Omron CX-Programmer project 新工程 (CX-Programmer 9.61)

# PLC 后氦检24L: CJ2M CPU33
I/O table (CPU CJ2M-CPU33): rack 0 slot 0 CJ1W-NC213; rack 0 slot 1 CJ1W-SCU21-V1; rack 0 slot 2 CJ1W-SCU21-V1; rack 0 slot 3 CJ1W-AD041-V1; rack 0 slot 4 CJ1W-ID261; rack 0 slot 5 CJ1W-ID261; rack 0 slot 6 CJ1W-OD261; rack 0 slot 7 CJ1W-MD231; rack 0 slot 11 CJ2M-EIP21

## Global symbols (name address type ; comment)
0 CHANNEL  ; 料盒#6电池屏蔽信号
0.00 BOOL  ; $?St$Bk?_#[1162] / 数字压力表 / $?St$Bk?_#[1162]
0.01 BOOL  ; 扫码位电池感应
0.02 BOOL  ; 抓料位有托盘感应
0.03 BOOL  ; 抓电池处有电池感应
0.04 BOOL  ; 腔体1有料感应
0.05 BOOL  ; 缺相保护信号
0.06 BOOL  ; 出料起始位有料感应
0.07 BOOL  ; 输送带有料感应
0.08 BOOL  ; NG放料位有料感应(常闭)
0.09 BOOL  ; NG通道料满感应
0.10 BOOL  ; 上料柔性报警
0.11 BOOL  ; 下料柔性报警延时
0.12 BOOL  ; 入盘升降柔性报警
0.13 BOOL  ; 料盒#12电池有料感应
0.14 BOOL  ; 料盒#11电池有料信号
0.15 BOOL  ; 料盒#10电池有料信号
10.00 BOOL  ; #2破真空阀
10.01 BOOL  ; #2吹气阀
10.02 BOOL  ; #2上顶升气缸
10.03 BOOL  ; #1上顶升气缸
10.04 BOOL  ; #2下顶升气缸
10.05 BOOL  ; #1下顶升气缸
10.06 BOOL  ; 料盒上阻挡气缸
10.07 BOOL  ; 料盒下阻挡气缸
10.08 BOOL  ; 料盒定位气缸
10.09 BOOL  ; 拉带左脱离气缸
10.10 BOOL  ; 拉带右脱离气缸
10.11 BOOL  ; 出料NG拨料气缸
10.12 BOOL  ; 上空料盘电机
10.13 BOOL  ; 下有料盘电机
10.14 BOOL  ; 有料盘缓存电机
10.15 BOOL  ; 出料输送带
11.01 BOOL  ; 真空泵
11.02 BOOL  ; 氦检仪启动
11.03 BOOL  ; 启动指示灯
11.04 BOOL  ; 停止指示灯
11.05 BOOL  ; 复位指示灯
11.06 BOOL  ; 蜂鸣器
11.07 BOOL  ; 三色红灯
11.08 BOOL  ; 三色绿灯
11.09 BOOL  ; 三色黄灯
11.10 BOOL  ; 料盒升降伺服Serv_ON
11.11 BOOL  ; 料盒升降伺服Alarm_Clr
11.12 BOOL  ; 入盘升降气缸
11.13 BOOL  ; 入盘夹爪气缸
11.14 BOOL  ; 龙门升降伺服刹车
11.15 BOOL  ; 料盒升降伺服刹车
12.03 BOOL  ; NG有料感应
12.07 BOOL  ; 腔体2有料感应
13.00 BOOL  ; 上料NG伸出位
13.01 BOOL  ; 上料NG缩回位
13.02 BOOL  ; 上料NG满感应
13.03 BOOL  ; 上料缓存NG有料感应
13.04 BOOL  ; 右按钮上气缸顶升请求（上料叉车到位）
13.05 BOOL  ; 左按钮气缸顶升请求（下料叉车到位）
13.07 BOOL  ; 腔体2有料感应
13.08 BOOL  ; 上料盒位有料盒感应
1534.15 BOOL  ; 单元1的串口1协议宏执行标志
1544.15 BOOL  ; 单元1的串口2协议宏执行标志
1559.15 BOOL  ; 单元2串口1协议宏执行标志
19.00 BOOL  ; 真空泵缺相报警
19.01 BOOL  ; PC系统异常
1.00 BOOL  ; 料盒#9电池有料信号
1.01 BOOL  ; 料盒#8电池有料信号
1.02 BOOL  ; 料盒#7电池有料信号
1.03 BOOL  ; 料盒#6电池有料信号
1.04 BOOL  ; 料盒#5电池有料信号
1.05 BOOL  ; 料盒#4电池有料信号
1.06 BOOL  ; 料盒#3电池有料信号
1.07 BOOL  ; 料盒#2电池有料信号
1.08 BOOL  ; 料盒#1电池有料信号
1.09 BOOL  ; 料盒#24电池有料信号
1.10 BOOL  ; 料盒#23电池有料信号
1.11 BOOL  ; 料盒#22电池有料信号
1.12 BOOL  ; 料盒#21电池有料信号
1.13 BOOL  ; 料盒#20电池有料信号
1.14 BOOL  ; 料盒#19电池有料信号
1.15 BOOL  ; 料盒#18电池有料信号
2000.03 BOOL  ; 绝对定位
2000.06 BOOL  ; 前后位回原
2000.09 BOOL  ; 龙门前后伺服脉冲
2000.10 BOOL  ; 龙门前后伺服方向
2000.12 BOOL  ; NC-X轴错误复位
2000.15 BOOL  ; 入盘Y轴停止
2002.03 BOOL  ; 料盘绝对运动
2002.06 BOOL  ; 料盘回原
2002.09 BOOL  ; 料盘升降脉冲
2002.10 BOOL  ; 料盘运动方向
2002.12 BOOL  ; NC-Y轴复位
2002.15 BOOL  ; 料盘伺服减速2停止
2004.06 BOOL  ; Y轴原点标志
2004.12 BOOL  ; NC
2004.13 BOOL  ; 伺服忙标志位
2007.06 BOOL  ; 料盘升降原点标志
2007.13 BOOL  ; 料盘伺服忙标志位
2010 CHANNEL  ; #1真空计度读出值CHO
2011 CHANNEL  ; #1真空计读出值CH1
2012 CHANNEL  ; #2真空计读出值CH2
20.01 BOOL  ; #2电池扫码信号
20.04 BOOL  ; 两扫码NG
20.09 BOOL  ; 放右NG缩回
21.00 BOOL  ; 上料机械手回左上料位
21.01 BOOL  ; 上料机械手回右上料位
21.05 BOOL  ; 上料右夹爪夹紧
21.09 BOOL  ; 上料右夹爪松开
21.10 BOOL  ; 上料提升气缸缩回
21.11 BOOL  ; 上料提升气缸/左夹爪升降气缸伸出
21.14 BOOL  ; 上料右夹爪夹紧
21.15 BOOL  ; 上料机械手去#1腔体放料
22.02 BOOL  ; 上料提升气缸取OK料后缩回(A)
22.10 BOOL  ; 上料提升气缸伸出(抓NG料)(A)
22.12 BOOL  ; 上料提升气缸伸出(放扫码NG料)(A)
22.13 BOOL  ; #1，#2夹爪张开(放扫码NG料)(A)
22.14 BOOL  ; 上料提升气缸缩回(放扫码NG料)(A)
22.15 BOOL  ; 扫码NG气缸缩回
25.13 BOOL  ; 出料机械手归零后回NG位置
25.15 BOOL  ; 机械手放料条件
26.00 BOOL  ; 出料旋转回#1待料位
26.02 BOOL  ; 下料升降气缸输出
26.06 BOOL  ; 下料升降/提升气缸输出
26.13 BOOL  ; 下料旋转回#2待料角度
26.14 BOOL  ; 下料旋转回出料角度
27.00 BOOL  ; 下料旋转归零后回下料角度
28.00 BOOL  ; 电池从扫码位到抓料超时
28.01 BOOL  ; 扫码阻挡气缸缩回位异常
28.02 BOOL  ; 扫码阻挡气缸伸出位异常
28.03 BOOL  ; 抓料阻挡气缸缩回位异常
28.04 BOOL  ; 抓料阻挡气缸伸出位异常
28.09 BOOL  ; 出料机械手回#1腔体位置
28.10 BOOL  ; 出料机械手回#2腔体位置
28.11 BOOL  ; 出料机械手回OK位置
28.12 BOOL  ; 出料机械手回放爪2位置
28.13 BOOL  ; 出料机械手回NG位置
2906.06 BOOL  ; 进料机械手左极限
2906.07 BOOL  ; 进料机械手右极限
2906.08 BOOL  ; 出料机械手左极限
2906.09 BOOL  ; 出料机械手右极限
2960.06 BOOL  ; 进料机械手左限位
2960.07 BOOL  ; 进料机械手右限位
2960.08 BOOL  ; 出料机械手左限位
2960.09 BOOL  ; 出料机械手右限位
2962.00 BOOL  ; 入盘升降原点
2962.06 BOOL  ; 龙门升降伺服上限位
2962.07 BOOL  ; 龙门升降伺服下限位
2962.08 BOOL  ; 龙门左右伺服左限位
2962.09 BOOL  ; 龙门左右伺服右限位
29.00 BOOL  ; 扫码NG拨料气缸缩回位报警
29.01 BOOL  ; 扫码NG拨料气缸伸出报警
29.02 BOOL  ; 上料提升气缸缩回报警
29.03 BOOL  ; 上料提升气缸伸出报警
29.04 BOOL  ; 上料左夹爪升降缩回报警
29.05 BOOL  ; 上料左夹爪升降气缸伸出报警
29.06 BOOL  ; 上料右夹爪升降气缸缩回报警
29.07 BOOL  ; 上料右夹爪升降气缸缩回报警
29.08 BOOL  ; 上料左夹爪张开位报警
29.09 BOOL  ; 上料左夹爪夹紧报警
29.10 BOOL  ; 上料夹爪2张开报警
29.11 BOOL  ; 上料夹爪2夹紧报警
29.12 BOOL  ; 上料机构柔性报警
29.13 BOOL  ; 进料机械手报警
2.00 BOOL  ; 料盒#17电池有料信号
2.01 BOOL  ; 料盒#16电池有料信号
2.02 BOOL  ; 料盒#15电池有料信号
2.03 BOOL  ; 料盒#14电池有料信号
2.04 BOOL  ; 料盒#13电池有料信号
2.05 BOOL  ; 扫码阻挡缩回位
2.06 BOOL  ; 扫码阻挡气缸伸出位
2.07 BOOL  ; 扫码定位气缸缩回位
2.08 BOOL  ; 扫码定位气缸伸出位
2.09 BOOL  ; 抓料阻挡气缸缩回位
2.10 BOOL  ; 抓料阻挡气缸伸出位
2.11 BOOL  ; 上料提升气缸缩回位
2.12 BOOL  ; 上料提升气缸伸出位
2.13 BOOL  ; 上料左夹爪升降气缸缩回位
2.14 BOOL  ; 上料左夹爪升降气缸伸出位
2.15 BOOL  ; 上料右夹爪升降气缸缩回位
32.00 BOOL  ; 读检漏仪状态
32.01 BOOL  ; 读氦检仪状态完成
32.02 BOOL  ; 读检漏口压力
32.03 BOOL  ; 读检漏口压力完成
32.05 BOOL  ; 读漏率
32.06 BOOL  ; 读漏率完成
32.07 BOOL  ; 读漏率失败
32.08 BOOL  ; 读氦检仪状态失败
32.09 BOOL  ; 读检漏口压力失败
3304.10 BOOL  ; 氦检仪报警
33.00 BOOL  ; #1腔体复位破真空
33.01 BOOL  ; #1合模气缸复位缩回
33.02 BOOL  ; 进料机械手有料
33.03 BOOL  ; 出料机械手有料
33.04 BOOL  ; #1合模气缸复位
33.05 BOOL  ; 下料夹爪有料
34.00 BOOL  ; 氦检仪当前为检漏状态
34.01 BOOL  ; 氦检仪当前为待机状态
34.02 BOOL  ; 氦检仪当前为启动状态
34.03 BOOL  ; 氦检仪当前为定标状态
34.04 BOOL  ; 氦检仪当前为错误状态
34.05 BOOL  ; 氦检仪当前为暂停状态
35.00 BOOL  ; #2腔体复位破真空
35.01 BOOL  ; #2合模气缸缩回
35.02 BOOL  ; #2合模气缸复位
35.05 BOOL  ; 扫码气缸自动伸出
39.00 BOOL  ; 合模气缸1缩回报警
39.01 BOOL  ; 合模气缸1伸出报警
39.02 BOOL  ; 合模气缸2缩回报警
39.03 BOOL  ; 合模气缸2伸出报警
39.04 BOOL  ; 氦检仪没启动
39.05 BOOL  ; 读氦漏率失败
39.06 BOOL  ; 读氦检仪状态失败
39.07 BOOL  ; 读检漏口压力失败
39.08 BOOL  ; 氦检仪通信异常
39.09 BOOL  ; 扫码枪通信异常
39.10 BOOL  ; #1真空计断线报警
39.11 BOOL  ; #2真空计断线报警
39.12 BOOL  ; （I：0.04）#1腔体有料感应异常
39.13 BOOL  ; （I：13.07）#2腔体有料感应异常
3.00 BOOL  ; 上料右夹爪升降气缸伸出位
3.01 BOOL  ; 上料左夹爪张开位
3.02 BOOL  ; 上料左夹爪夹紧位
3.03 BOOL  ; 上料右夹爪张开位
3.04 BOOL  ; 上料右夹爪夹紧位
3.05 BOOL  ; 下料提升气缸缩回位
3.06 BOOL  ; 下料提升气缸伸出位
3.07 BOOL  ; 下料夹爪升降气缸缩回位
3.08 BOOL  ; 下料夹爪升降气缸伸出位
3.09 BOOL  ; 下料左夹爪张开位
3.10 BOOL  ; 下料左夹爪夹紧位
3.11 BOOL  ; 下料右夹爪张开位
3.12 BOOL  ; 下料右夹爪夹紧位
3.13 BOOL  ; #1合模气缸缩回位
3.14 BOOL  ; #1合模气缸伸出位
3.15 BOOL  ; #2合模气缸缩回位
46.00 BOOL  ; #1夹爪放料完成
46.01 BOOL  ; #2夹爪放料完成
48.00 BOOL  ; 出料机械手位置异常
48.01 BOOL  ; 下料旋转托盘位置异常
48.02 BOOL  ; 下料缓存有料异常
48.03 BOOL  ; #1合模气缸不在缩回位
48.04 BOOL  ; #2合模气缸不在缩回位
48.05 BOOL  ; 出料夹爪不在张开位
48.06 BOOL  ; 出料提升气缸不在伸出位
48.07 BOOL  ; 出料提升气缸不在缩回位
48.08 BOOL  ; 出料机械手没归零
48.09 BOOL  ; 出料机械手到达左极限
48.10 BOOL  ; 出料机械手到达右极限
48.11 BOOL  ; 进料机械手位置避让异常
48.12 BOOL  ; 进料机械手位置避让异常
49.00 BOOL  ; 下料提升气缸缩回报警
49.01 BOOL  ; 下料提升气缸伸出报警
49.02 BOOL  ; 下料夹爪升降气缸缩回报警
49.03 BOOL  ; 下料夹爪升降气缸伸出报警
49.04 BOOL  ; 下料夹爪1张开报警
49.05 BOOL  ; 下料夹爪夹1紧报警
49.06 BOOL  ; 下料夹爪2张开位延时报警
49.07 BOOL  ; 下料夹爪2夹紧位报警
49.08 BOOL  ; 出料NG拨料气缸伸出位报警
49.09 BOOL  ; 出料NG拨料气缸缩回位报警
49.10 BOOL  ; 出料机械手报警
49.11 BOOL  ; 下料机构柔性报警
49.12 BOOL  ; （0.06）出料起始位有料感应异常
49.13 BOOL  ; （10.05）出料拉带运行异常
49.14 BOOL  ; （0.07）出料拉带末端感应异常
4.00 BOOL  ; #2合模气缸伸出位
4.01 BOOL  ; 出料NG拨料气缸缩回位
4.02 BOOL  ; 出料NG拨料气缸伸出位
4.03 BOOL  ; 料盒定位气缸缩回位
4.04 BOOL  ; 料盒定位气缸伸出位
4.05 BOOL  ; 料盒上阻挡气缸缩回位
4.06 BOOL  ; 料盒上阻挡气缸伸出位
4.07 BOOL  ; 料盒下阻挡气缸缩回位
4.08 BOOL  ; 料盒下阻挡气缸伸出位
4.09 BOOL  ; #2上顶升左气缸缩回位
4.10 BOOL  ; #2上顶升左气缸伸出位
4.11 BOOL  ; #2上顶升右气缸缩回位
4.12 BOOL  ; #2上顶升右气缸伸出位
4.13 BOOL  ; #1上顶升左气缸缩回位
4.14 BOOL  ; #1上顶升左气缸伸出位
4.15 BOOL  ; #1上顶升右气缸缩回位
54.00 BOOL  ; 放料准备-拉带对接测试按钮(T)
54.02 BOOL  ; 放料可移动-拉带对接测试按钮(T)
54.03 BOOL  ; 取料准备-拉带对接测试按钮(T)
54.05 BOOL  ; 取料可移动-拉带对接测试按钮(T)
54.06 BOOL  ; 设备故障-拉带对接测试按钮(T)
54.10 BOOL  ; 可取料-拉带对接测试按钮(T)
5.00 BOOL  ; #1上顶升右气缸伸出位
5.01 BOOL  ; #2下顶升左气缸缩回位
5.02 BOOL  ; #2下顶升左气缸伸出位
5.03 BOOL  ; #2下顶升右气缸缩回位
5.04 BOOL  ; #2下顶升右气缸伸出位
5.05 BOOL  ; #1下顶升左气缸缩回位
5.06 BOOL  ; #1下顶升左气缸伸出位
5.07 BOOL  ; #1下顶升右气缸缩回位
5.08 BOOL  ; #1下顶升右气缸伸出位
5.09 BOOL  ; 龙门左拉带脱离气缸缩回位
5.10 BOOL  ; 龙门左拉带脱离气缸伸出位
5.11 BOOL  ; 龙门右拉带脱离气缸缩回位
5.12 BOOL  ; 龙门右拉带脱离气缸伸出位
5.13 BOOL  ; 上料伺服Ready信号
5.14 BOOL  ; 上料伺服Alarm信号
5.15 BOOL  ; 下料伺服Ready信号
68.00 BOOL  ; 料盒定位气缸缩回位报警
68.01 BOOL  ; 料盒定位气缸伸出位报警
68.02 BOOL  ; 料盒上阻挡气缸缩回位报警
68.03 BOOL  ; 料盒上阻挡气缸伸出位报警
68.04 BOOL  ; #1上顶升左气缸缩回位报警
68.05 BOOL  ; #1上顶升左气缸伸出位报警
68.06 BOOL  ; #1上顶升右气缸缩回位报警
68.07 BOOL  ; #1上顶升右气缸伸出位报警
68.08 BOOL  ; #2上顶升左气缸缩回位报警
68.09 BOOL  ; #2上顶升左气缸伸出位报警
68.10 BOOL  ; #2上顶升右气缸缩回位报警
68.11 BOOL  ; #2上顶升右气缸伸出位报警
68.12 BOOL  ; #1下顶升左气缸缩回位报警
68.13 BOOL  ; #1下顶升左气缸伸出位报警
68.14 BOOL  ; #1下料顶升右气缸缩回位报警
68.15 BOOL  ; #1下顶升右气缸伸出位报警
69.00 BOOL  ; #2下顶升左气缸缩回位报警
69.01 BOOL  ; #2下顶升左气缸伸出位报警
69.02 BOOL  ; #2下料顶升右气缸缩回位报警
69.03 BOOL  ; #2下顶升右气缸伸出位报警
69.04 BOOL  ; 入盘左拉带脱离气缸缩回位报警
69.05 BOOL  ; 入盘左拉带脱离气缸伸出位报警
69.06 BOOL  ; 入盘右拉带脱离气缸缩回位报警
69.07 BOOL  ; 入盘右拉带脱离气缸伸出位报警
69.08 BOOL  ; 入盘升降气缸缩回位延时报警
69.09 BOOL  ; 入盘升降气缸伸出位延时报警
69.10 BOOL  ; 入盘夹爪气缸松开延时报警
69.11 BOOL  ; 入盘夹爪气缸夹紧延时报警
69.12 BOOL  ; 入盘机械手柔性报警
69.13 BOOL  ; 此位置有电池不能入盘
6.00 BOOL  ; 下料伺服Alarm信号
6.01 BOOL  ; 入盘升降伺服Ready信号
6.02 BOOL  ; 入盘升降伺服Alarm信号
6.03 BOOL  ; 龙门左右伺服Ready信号
6.04 BOOL  ; 龙门左右伺服Alarm信号
6.05 BOOL  ; 龙门前后伺服Ready信号
6.06 BOOL  ; 龙门前后伺服Alarm信号
6.07 BOOL  ; 氦检仪器报警
6.08 BOOL  ; 启动按钮
6.09 BOOL  ; 停止按钮
6.10 BOOL  ; 复位按钮
6.11 BOOL  ; 急停按钮
6.12 BOOL  ; 前门磁开关
6.13 BOOL  ; 后门磁开关
6.14 BOOL  ; 左门禁开关
6.15 BOOL  ; 右门禁开关
70.01 BOOL  ; I:7.01空托盘感应感应异常
70.02 BOOL  ; I:7.00空托盘感应感应异常
70.03 BOOL  ; （7.02）空托盘到位感应或拉带异常
70.04 BOOL  ; (7.05)#3空托盘感应或拉带异常
70.05 BOOL  ; 空托盘到位感应、#3空托盘感应或拉带异常
70.06 BOOL  ; 空托盘到位感应
70.07 BOOL  ; 空盘升降机架上有空托盘记忆异常
70.08 BOOL  ; （7.05）上空托盘位感应异常
70.09 BOOL  ; （7.14）下满料托盘感应1异常
70.10 BOOL  ; （7.04）下满料托盘到位感应#2异常
70.11 BOOL  ; （13.08）电池入盘位有托盘感应异常
70.12 BOOL  ; （7.03）缓存#1托盘到位感应异常
70.13 BOOL  ; （7.04）缓存#2托盘到位感应异常
71.00 BOOL  ; 上空托盘感应异常
7.00 BOOL  ; #2下感应有空料盒（外面）
7.01 BOOL  ; #1下感应有空料盒
7.02 BOOL  ; 料盒到位感应
7.03 BOOL  ; 缓存1有料到位感应
7.04 BOOL  ; 缓存2有料到位感应
7.05 BOOL  ; #3下料盒有料感应
7.06 BOOL  ; 料盒升降伺服Ready
7.07 BOOL  ; 料盒升降伺服Alarm
7.08 BOOL  ; $?St$Bk?_#[1163] / 龙门升降气缸缩回位 / $?St$Bk?_#[1163]
7.09 BOOL  ; $?St$Bk?_#[1164] / 龙门升降气缸伸出位 / $?St$Bk?_#[1164]
7.10 BOOL  ; $?St$Bk?_#[1165] / 龙门夹爪气缸张开位 / $?St$Bk?_#[1165]
7.11 BOOL  ; 龙门夹爪气缸夹紧
7.12 BOOL  ; $?St$Bk?_#[1166] / 上层货架叉车感应 / $?St$Bk?_#[1166]
7.13 BOOL  ; $?St$Bk?_#[1167] / 下层货架叉车感应 / $?St$Bk?_#[1167]
7.14 BOOL  ; 上有料盒感应1
7.15 BOOL  ; 缓存2有料感应
81.00 BOOL  ; 扫码NG缓存有料
82.02 BOOL  ; #3上料夹爪有料
82.03 BOOL  ; #4上料夹爪有料
83.02 BOOL  ; #3下料夹爪有料
83.03 BOOL  ; #4下料夹爪有料
84.11 BOOL  ; #2扫码失败
84.12 BOOL  ; #2扫码OK
8.00 BOOL  ; $?St$Bk?_#[1168] / 上料伺服Serv_On / $?St$Bk?_#[1168]
8.01 BOOL  ; $?St$Bk?_#[1169] / 上料伺服Alarm_Clr / $?St$Bk?_#[1169]
8.02 BOOL  ; $?St$Bk?_#[1170] / 下料伺服Serv_On / $?St$Bk?_#[1170]
8.03 BOOL  ; $?St$Bk?_#[1171] / 下料伺服Alarm_Clr / $?St$Bk?_#[1171]
8.04 BOOL  ; $?St$Bk?_#[1172] / 龙门升降伺服Serv_On / $?St$Bk?_#[1172]
8.05 BOOL  ; 龙门升降伺服Alarm_Clr
8.06 BOOL  ; 龙门左右伺服Serv_ON
8.07 BOOL  ; 龙门左右伺服Alarm_Clr
8.08 BOOL  ; 龙门前后伺服Serv_ON
8.09 BOOL  ; $?St$Bk?_#[1173] / 龙门前后伺服Alarm_Clr / $?St$Bk?_#[1173]
8.10 BOOL  ; 扫码阻挡气缸
8.11 BOOL  ; 抓料阻挡气缸
8.12 BOOL  ; 上料NG气缸
8.13 BOOL  ; 上料提升气缸
8.14 BOOL  ; 上料左夹爪升降气缸
8.15 BOOL  ; 上料右夹爪升降气缸
9.00 BOOL  ; $?St$Bk?_#[1174] / 上料左夹爪气缸 / $?St$Bk?_#[1174]
9.01 BOOL  ; 上料右夹爪
9.02 BOOL  ; 下料提升气缸
9.03 BOOL  ; 下料夹爪升降气缸
9.04 BOOL  ; 下料左夹爪气缸
9.05 BOOL  ; 下料右夹爪气缸
9.06 BOOL  ; #1合模气缸关闭
9.07 BOOL  ; #1合模气缸打开
9.08 BOOL  ; $?St$Bk?_#[1175] / #1腔体抽气阀 / $?St$Bk?_#[1175]
9.09 BOOL  ; $?St$Bk?_#[1176] / #1腔体氦检阀 / $?St$Bk?_#[1176]
9.10 BOOL  ; $?St$Bk?_#[1177] / #1腔体破真空阀 / $?St$Bk?_#[1177]
9.11 BOOL  ; $?St$Bk?_#[1178] / #1腔体吹气阀 / $?St$Bk?_#[1178]
9.12 BOOL  ; #2合模气缸关闭
9.13 BOOL  ; #2合模气缸打开
9.14 BOOL  ; #2抽气阀
9.15 BOOL  ; #2氦检阀
A202.01 BOOL  ; 通信端口1允许标志
A202.02 BOOL  ; 通信端口2允许标志
A276 CHANNEL  ; 前机械手当前脉冲
A278 CHANNEL  ; 后机械手当前脉冲
A280.04 BOOL  ; 上料机械手脉冲输出中
A280.05 BOOL  ; 上料机械手原点标志
A281.04 BOOL  ; 后机械手脉冲输出中
A281.05 BOOL  ; 下料机械手原点标志
A322 CHANNEL  ; 上料旋转当前位置脉冲
A324 CHANNEL  ; 下料旋转当前位置脉冲
A326.04 BOOL  ; 入盘升降脉冲输出中
A326.05 BOOL  ; 入盘升降原点标志
A327.04 BOOL  ; 入盘X轴脉冲标志
A327.05 BOOL  ; 入盘X轴原点标志
A351 CHANNEL  ; 系统时间(分秒)
A352 CHANNEL  ; 系统时间(日时)
A353 CHANNEL  ; 系统时间(年月)
A501.01 BOOL  ; #1通信模块复位
A501.02 BOOL  ; #2通信模块复位
A540.08 BOOL  ; 进料机械手CW
A540.09 BOOL  ; 进料机械手CCW
A541.08 BOOL  ; 出料机械手CW
A541.09 BOOL  ; 出料机械手CCW
A542.08 BOOL  ; 龙门升降伺服下限位
A542.09 BOOL  ; 龙门升降伺服上限位
A543.08 BOOL  ; 龙门左右伺服右限位
A543.09 BOOL  ; 龙门左右伺服左限位
D0.00 BOOL  ; CF113
D10 CHANNEL  ; 报警画面跳转
D100 CHANNEL  ; 扫码阻挡气缸缩回位延时
D1000 CHANNEL  ; #1腔体检漏口压力(浮点)
D1002 CHANNEL  ; #1腔体漏率(浮点)
D1004 CHANNEL  ; #1腔体测试完成时的检漏口压力
D1006 CHANNEL  ; #1腔体测试完成时的漏率
D1008 CHANNEL  ; #1腔抽残气压力
D101 CHANNEL  ; 扫码阻挡气缸伸出位延时
D102 CHANNEL  ; 扫码定位气缸缩回位延时
D1020 CHANNEL  ; #2腔体检漏口压力(浮点)
D1022 CHANNEL  ; #2腔体漏率(浮点)
D1024 CHANNEL  ; #2腔体测试完成时检漏口压力
D1026 CHANNEL  ; #2腔体测试完成时的漏率
D1028 CHANNEL  ; #2腔抽残气压力
D103 CHANNEL  ; 扫码定位气缸伸出位延时
D104 CHANNEL  ; 抓料阻挡气缸缩回位延时
D105 CHANNEL  ; 抓料阻挡气缸伸出位延时
D106 CHANNEL  ; 上料提升气缸缩回位延时
D107 CHANNEL  ; 上料提升气缩回位延时
D108 CHANNEL  ; 上料左夹爪升降气缸缩回位延时
D109 CHANNEL  ; 上料左夹爪升降气缸伸出位延时
D110 CHANNEL  ; 上料右夹爪升降气缸缩回位延时
D111 CHANNEL  ; 上料右夹爪升降气缸伸出位延时
D112 CHANNEL  ; 上料左夹爪张开位延时
D113 CHANNEL  ; 上料左夹爪夹紧位延时
D114 CHANNEL  ; 上料右夹爪张开位延时
D115 CHANNEL  ; 上料右夹爪夹紧位延时
D116 CHANNEL  ; 下料提升气缸缩回位延时
D1160 CHANNEL  ; 正向行程
D1164 CHANNEL  ; 反向行程（浮点）
D1168 CHANNEL  ; 反向行程
D117 CHANNEL  ; 下料提升气缸伸出位延时
D118 CHANNEL  ; 下料夹爪升降气缸缩回位延时
D119 CHANNEL  ; 下料夹爪升降气缸伸出位延时
D120 CHANNEL  ; 下料左夹爪张开位延时
D1204 CHANNEL  ; 检漏口压力设定值
D1206 CHANNEL  ; 漏率设定值
D121 CHANNEL  ; 下料左夹爪夹紧位延时
D122 CHANNEL  ; 下料右夹爪张开位延时
D123 CHANNEL  ; 下料右夹爪夹紧位延时
D124 CHANNEL  ; #1合模气缸缩回位延时
D125 CHANNEL  ; #1合模气缸伸出位延时
D126 CHANNEL  ; #2合模气缸缩回位延时
D1260 CHANNEL  ; 检漏口压力底数转换
D1264 CHANNEL  ; 漏率底数转换
D127 CHANNEL  ; #2合模气缸伸出位延时
D128 CHANNEL  ; 扫码NG拨料气缸缩回位延时
D129 CHANNEL  ; 扫码NG拨料气缸伸出位延时
D130 CHANNEL  ; 料盒定位气缸缩回位延时
D131 CHANNEL  ; 料盒定位气缸伸出位延时
D132 CHANNEL  ; 料盒上阻挡气缸缩回位延时
D133 CHANNEL  ; 料盒上阻挡气缸伸出位延时
D134 CHANNEL  ; 料盒下阻挡气缸缩回位延时
D135 CHANNEL  ; 料盒下阻挡气缸伸出位延时
D136 CHANNEL  ; #1上顶升左气缸缩回位延时
D137 CHANNEL  ; #1上顶升左气缸伸出位延时
D138 CHANNEL  ; #1上顶升右气缸缩回位延时
D139 CHANNEL  ; #1上顶升右气缸伸出位延时
D140 CHANNEL  ; #2上顶升左气缸缩回位延时
D141 CHANNEL  ; #2上顶升左气缸伸出位延时
D142 CHANNEL  ; #2上顶升右气缸缩回位延时
D143 CHANNEL  ; #2上顶升右气缸伸出位延时
D144 CHANNEL  ; #1下顶升左气缸缩回位延时
D145 CHANNEL  ; #1下顶升左气缸伸出位延时
D146 CHANNEL  ; #1下顶升右气缸缩回位延时
D147 CHANNEL  ; #1下顶升右气缸伸出位延时
D148 CHANNEL  ; #2下顶升左气缸延时缩回位
D149 CHANNEL  ; #2下顶升左气缸伸出位延时
D150 CHANNEL  ; #2下顶升右气缸缩回位延时
D151 CHANNEL  ; #2下顶升右气缸伸出位延时
D152 CHANNEL  ; 龙门左拉带脱离气缸缩回位延时
D153 CHANNEL  ; 龙门左拉带脱离气缸伸出位延时
D154 CHANNEL  ; 龙门右拉带脱离气缸缩回位延时
D155 CHANNEL  ; 龙门右拉带脱离气缸伸出位延时
D160 CHANNEL  ; 上料旋转步进当前脉冲
D1600 CHANNEL  ; #1条码下料机械手#1
D1606 CHANNEL  ; （龙门）抓料机械手当前位置(mm)
D1610 CHANNEL  ; #2条码下料机械手#2
D162 CHANNEL  ; 上料旋转步进当前脉冲(浮点）
D1620 CHANNEL  ; 产品检漏口压力在下料机械手#1
D1630 CHANNEL  ; 产品检漏口压力在下料机械手#2
D164 CHANNEL  ; 旋转脉冲当量(浮点)
D1640 CHANNEL  ; #1腔体测试完成时的漏率在下料机械手#1
D1650 CHANNEL  ; #1腔体测试完成时的漏率在下料机械手#2
D166 CHANNEL  ; 上料旋转步进当前位置(mm)
D1660 CHANNEL  ; 产品测试结果在下料机械手#1
D1670 CHANNEL  ; 产品测试结果在下料机械手#2
D168 CHANNEL  ; 旋转脉冲当量
D1690 CHANNEL  ; 1夹爪-1为腔体1-2为腔体2
D1692 CHANNEL  ; 2夹爪-1为腔体1-2为腔体2
D170 CHANNEL  ; 下料旋转步进当前脉冲
D1700 CHANNEL  ; 下料机械手#1条码
D1710 CHANNEL  ; 下料机械手#2条码
D172 CHANNEL  ; 下料旋转步进当前脉冲(浮点)
D1730 CHANNEL  ; OK拉带电池条码
D1750 CHANNEL  ; 龙门夹爪电池条码
D176 CHANNEL  ; 下料旋转步进当前角度(mm)
D1800 CHANNEL  ; 故障代码
D1802 CHANNEL  ; 设备状态
D1803 CHANNEL  ; 设备状态(存储)
D1804 CHANNEL  ; 设备状态变更
D181 CHANNEL  ; 入盘升降气缸缩回位延时
D1810 CHANNEL  ; #1爪电池抽真空时间
D1812 CHANNEL  ; #1爪电池真空达到阀值
D1814 CHANNEL  ; #1爪电池抽残气压力
D1816 CHANNEL  ; #1爪电池氦检消耗时长
D1818 CHANNEL  ; #1爪电池破真空阀值
D182 CHANNEL  ; 入盘升降气缸伸出位延时
D183 CHANNEL  ; 入盘夹爪气缸松开延时
D1830 CHANNEL  ; #2爪电池抽真空时间
D1832 CHANNEL  ; #2爪电池真空达到阀值
D1834 CHANNEL  ; #2爪电池抽残气压力
D1836 CHANNEL  ; #2爪电池氦检消耗时长
D1838 CHANNEL  ; #2爪电池破真空阀值
D184 CHANNEL  ; 龙门夹爪气缸夹紧延时
D185 CHANNEL  ; #1上料盒到位感应延时
D1856 CHANNEL  ; #1爪电池抽残气压力
D1858 CHANNEL  ; 下料机械手#1产品检漏口压力
D186 CHANNEL  ; #2上料盒到位感应延时
D1860 CHANNEL  ; 下料机械手#1产品漏率
D1862 CHANNEL  ; 产品测试结果在下料机械手#1
D1864 CHANNEL  ; #1爪电池抽真空时间
D1866 CHANNEL  ; #2爪电池抽残气压力
D1868 CHANNEL  ; 下料机械手#2产品检漏口压力
D187 CHANNEL  ; 料盒到位感应延时
D1870 CHANNEL  ; 下料机械手#2产品漏率
D1872 CHANNEL  ; 产品测试结果在下料机械手#2
D1874 CHANNEL  ; #2爪电池抽真空时间
D1876 CHANNEL  ; 托盘电池位置
D188 CHANNEL  ; #1下料盒到位感应延时
D1880 CHANNEL  ; 托盘放料信号--->PC
D189 CHANNEL  ; #2下料盒到位感应延时
D190 CHANNEL  ; #3下料盒到位感应延时
D1900 CHANNEL  ; 1为腔体1-2为腔体2
D1902 CHANNEL  ; 1为腔体1-2为腔体2
D1904 CHANNEL  ; PC返回夹1-OK
D1905 CHANNEL  ; PC返回夹2-OK
D1906 CHANNEL  ; 托盘扫码OK-->PC
D1908 CHANNEL  ; 托盘码注册OK PC-->PLC
D191 CHANNEL  ; 出料NG气伸出位屏蔽延时
D1910 CHANNEL  ; 出料夹爪电池时间
D192 CHANNEL  ; 出料NG气缩回位屏蔽延时
D1920 CHANNEL  ; 系统时间(年)
D1922 CHANNEL  ; 系统时间(日)
D1924 CHANNEL  ; 系统时间(分)
D1930 CHANNEL  ; #1腔体电池时间
D1940 CHANNEL  ; #2腔体电池时间
D196 CHANNEL  ; 传感器延迟时间
D197 CHANNEL  ; 报警信号延时
D198 CHANNEL  ; 上下料机械手距各自原点的总距离
D2000 CHANNEL  ; 进料机械手手动速度mm/s
D2002 CHANNEL  ; 进料机械手自动速度mm/s
D2004 CHANNEL  ; 异常报警状态2
D2006 CHANNEL  ; 异常报警状态3
D20068 CHANNEL  ; 运动位置
D20070 CHANNEL  ; NC-速度
D2008 CHANNEL  ; 异常报警状态4
D20080 CHANNEL  ; 运动位置
D20092 CHANNEL  ; 入盘（前后）机械手当前脉冲
D20096 CHANNEL  ; 料盘当前脉冲
D2010 CHANNEL  ; 进料机械手左进料位置(浮点)
D20100 CHANNEL  ; #1,#2路模拟量使用设置
D20101 CHANNEL  ; #1,#2路模拟量输入范围位0--10v
D20118 CHANNEL  ; #1,#2路模拟量分辨率8000，普通模式
D2012 CHANNEL  ; 进料机械手右进料位
D2014 CHANNEL  ; 进料机械手腔体1位置(浮点)
D2016 CHANNEL  ; 进料机械手腔体2位置(浮点)
D2018 CHANNEL  ; 进NG左位置-HMI
D20180 CHANNEL  ; 上料Z轴输出脉冲-读取值（二进制）
D2020 CHANNEL  ; 进NG右位置-HMI
D2104 CHANNEL  ; 伺服脉冲当量
D2106 CHANNEL  ; 伺服脉冲当量(浮点)
D2110 CHANNEL  ; 进料机械手当前脉冲
D2112 CHANNEL  ; 进料机械手当前脉冲(浮点)
D2116 CHANNEL  ; 进料机械手当前位置(mm)
D2200 CHANNEL  ; 进料机械手手动速度puls/s
D2202 CHANNEL  ; 进料机械手自动速度puls/s
D2300 CHANNEL  ; 上料机械手自动状态加速度
D2301 CHANNEL  ; 上料机械手自动状态减速度
D2302 CHANNEL  ; 进料机械手自动速度puls/s
D2304 CHANNEL  ; 进料机械手自动位移量
D2306 CHANNEL  ; 上料机械手自动状态起动速度
D2310 CHANNEL  ; 上料机械手手动状态加速度
D2311 CHANNEL  ; 上料机械手手动状态减速度
D2312 CHANNEL  ; 进料机械手手动速度puls/s
D2314 CHANNEL  ; 进料机械手手动位移量
D2316 CHANNEL  ; 上料机械手手动状态起动速度
D234 CHANNEL  ; #1腔体状态 0-停用；1-待料；2-测试中；3-测试完成
D236 CHANNEL  ; #1腔体状态 0-停用；1-待料；2-测试中；3-测试完成
D240 CHANNEL  ; 接收检漏仪状态的起始字
D241 CHANNEL  ; 接收的检漏口压力(ASCII)
D2450 CHANNEL  ; 氦捡仪稳定时间设定值(BCD)
D2452 CHANNEL  ; #1氦检阀打开抽气阀关闭延时
D2454 CHANNEL  ; #2氦检阀打开抽气阀关闭延时
D250 CHANNEL  ; 接收检漏口压力的起始字
D2500 CHANNEL  ; 出料结束手动速度(度/s)
D2502 CHANNEL  ; 出料机械手自动速度(度/s)
D251 CHANNEL  ; 接收的检漏口压力(ASCII)
D2510 CHANNEL  ; 出料机械手腔体1位置(浮点)
D2512 CHANNEL  ; 出料机械手腔体2位置(mm)
D2514 CHANNEL  ; 出料机械手OK左放料位置(mm)
D2516 CHANNEL  ; 出料机械手OK右位置(mm)
D2518 CHANNEL  ; 下料机械手NG位置(浮点)
D260 CHANNEL  ; 接收漏率起始字
D261 CHANNEL  ; 接收的漏率(ASCII)
D2610 CHANNEL  ; 出料机械手当前脉冲
D2612 CHANNEL  ; 出料机械手当前脉冲(浮点)
D2616 CHANNEL  ; 出料机械手当前位置(mm)
D2620 CHANNEL  ; 进、出料机械手正向行程脉冲
D2624 CHANNEL  ; 进、出料机械手反向行程
D2628 CHANNEL  ; 进、出料机械手反向行程脉冲
D270 CHANNEL  ; 进,出料机械手原点间距离
D2700 CHANNEL  ; 出料机械手手动速度puls/s
D2702 CHANNEL  ; 出料机械手自动速度puls/s
D272 CHANNEL  ; 机械手治具宽度
D274 CHANNEL  ; 进,出料机械手间的距离
D280 CHANNEL  ; 两轴原点间距离
D2810 CHANNEL  ; 出料机械手手动状态加速度
D2811 CHANNEL  ; 出料机械手手动状态减速度
D2812 CHANNEL  ; 出料机械手手动速度puls/s
D2814 CHANNEL  ; 出料机械手手动位移量
D2816 CHANNEL  ; 出料机械手手动状态起动速度
D282 CHANNEL  ; 最小间距
D2820 CHANNEL  ; 出料机械手自动状态加速度
D2821 CHANNEL  ; 出料机械手自动状态减速度
D2822 CHANNEL  ; 出料机械手自动速度puls/s
D2824 CHANNEL  ; 出料机械手自动位移量
D2826 CHANNEL  ; 出料机械手自动状体起动速度
D2998 CHANNEL  ; 轴控制预留
D30 CHANNEL  ; 一排有料状态
D300 CHANNEL  ; 扫码阻挡气缸缩回位延时
D3000 CHANNEL  ; 腔体真空达到阀值
D3002 CHANNEL  ; 腔体抽气时间
D3004 CHANNEL  ; 抽残气后压力设置值
D3008 CHANNEL  ; 腔体破真空设定值
D301 CHANNEL  ; 扫码阻挡气缸伸出位延时
D302 CHANNEL  ; 抓料阻挡气缸缩回位延时
D3020 CHANNEL  ; 腔体自检真空阀值
D3022 CHANNEL  ; 腔体自检抽气时间
D3024 CHANNEL  ; 腔体自检泄漏量设置值
D303 CHANNEL  ; 抓料阻挡气缸伸出位延时
D3030 CHANNEL  ; 腔体自检保压前设定时间
D3032 CHANNEL  ; 腔体自检保压设定时间
D3034 CHANNEL  ; 腔体自检破真空设定值
D304 CHANNEL  ; 抓料阻挡气缸缩回位延时
D305 CHANNEL  ; 抓料阻挡气缸伸出位延时
D306 CHANNEL  ; 上料提升气缸缩回位延时
D307 CHANNEL  ; 上料提升气缸伸出位延时
D308 CHANNEL  ; 上料左夹爪升降气缸缩回位延时
D309 CHANNEL  ; 上料左夹爪升降气缸伸出位延时
D31 CHANNEL  ; 二排有状态
D310 CHANNEL  ; 上料右夹爪升降气缸缩回位延时
D3100 CHANNEL  ; #1腔体真空值
D3104 CHANNEL  ; #1腔体抽气时间
D3108 CHANNEL  ; #1腔体测试结果
D311 CHANNEL  ; 上料右夹爪升降气缸伸出位延时
D3110 CHANNEL  ; #1腔体手动抽气时间
D3111 CHANNEL  ; #1腔体保压前时间
D3112 CHANNEL  ; #1腔体保压时间
D312 CHANNEL  ; 上料左夹爪张开位延时
D3120 CHANNEL  ; #1腔体保压前真空值
D3122 CHANNEL  ; #1腔体保压后真空值
D3124 CHANNEL  ; #1腔体自检泄漏量
D313 CHANNEL  ; 上料左夹爪夹紧位延时
D314 CHANNEL  ; 上料右夹爪张开位延时
D315 CHANNEL  ; 上料右夹爪夹紧位延时
D316 CHANNEL  ; 下料提升气缸缩回位延时
D317 CHANNEL  ; 下料提升气缸伸出位延时
D318 CHANNEL  ; 下料夹爪升降气缸缩回位延时
D319 CHANNEL  ; 下料夹爪升降气缸伸出位延时
D320 CHANNEL  ; 下料左夹爪张开位延时
D3200 CHANNEL  ; #2腔体真空值
D3204 CHANNEL  ; #2腔体抽气时间
D3208 CHANNEL  ; #2腔体测试结果
D321 CHANNEL  ; 下料左夹爪夹紧位延时
D3210 CHANNEL  ; #2腔体自检抽气时间
D3211 CHANNEL  ; #2腔体进入保压前时间
D3212 CHANNEL  ; #2腔体保压时间
D322 CHANNEL  ; 下料右夹爪张开位延时
D3220 CHANNEL  ; #2腔体保压前真空值
D3222 CHANNEL  ; #1腔体保压后真空值
D3224 CHANNEL  ; #1腔体自检泄漏量
D323 CHANNEL  ; 下料右夹爪夹紧位延时
D324 CHANNEL  ; #1合模气缸缩回位延时
D325 CHANNEL  ; #1合模气缸伸出位延时
D326 CHANNEL  ; #2合模气缸缩回位延时
D327 CHANNEL  ; #2合模气缸伸出位延时
D328 CHANNEL  ; 扫码NG拨料气缸缩回位延时
D329 CHANNEL  ; 扫码NG拨料气缸伸出位延时
D330 CHANNEL  ; 料盒定位气缸缩回位延时
D3300 CHANNEL  ; 真空值1转存
D3302 CHANNEL  ; #1真空值运算1
D3304 CHANNEL  ; #1真空值运算2
D3306 CHANNEL  ; #1真空值运算3
D3308 CHANNEL  ; #1真空值运算4
D331 CHANNEL  ; 料盒定位气缸伸出位延时
D332 CHANNEL  ; 料盒上阻挡气缸缩回位位延时
D333 CHANNEL  ; 料盒上阻挡气缸伸出位延时
D334 CHANNEL  ; 料盒下阻挡气缸缩回位延时
D335 CHANNEL  ; 料盒下阻挡气缸伸出位延时
D336 CHANNEL  ; #1上顶升左气缸缩回位延时
D337 CHANNEL  ; #2上顶升左气缸伸出位延时
D338 CHANNEL  ; #2上顶升右气缸缩回位延时
D339 CHANNEL  ; #2上顶升右气缸伸出位延时
D340 CHANNEL  ; #1上顶升左气缸缩回位延时
D3400 CHANNEL  ; 真空值2转存
D3402 CHANNEL  ; #2真空值运算1
D3404 CHANNEL  ; #2真空值运算2
D3406 CHANNEL  ; #2真空值运算3
D3408 CHANNEL  ; #2真空值运算4
D341 CHANNEL  ; #1上顶升左气缸伸出位延时
D342 CHANNEL  ; #1上顶升右气缸缩回位延时
D343 CHANNEL  ; #1上顶升右气缸伸出位延时
D344 CHANNEL  ; #2下顶升左气缸缩回位延时
D345 CHANNEL  ; #2下顶升左气缸伸出位延时
D346 CHANNEL  ; #2下顶升右气缸缩回位延时
D347 CHANNEL  ; #2下顶升右气缸伸出位延时
D348 CHANNEL  ; #2下顶升左气缸延时缩回位
D349 CHANNEL  ; #1下顶升左气缸伸出位延时
D35 CHANNEL  ; 入盘状态
D350 CHANNEL  ; #1下顶升右气缸缩回位延时
D351 CHANNEL  ; #1下顶升右气缸伸出位延时
D352 CHANNEL  ; 龙门左拉带脱离气缸缩回位延时
D353 CHANNEL  ; 龙门左拉带脱离气缸伸出位延时
D354 CHANNEL  ; 龙门右拉带脱离气缸缩回位延时
D355 CHANNEL  ; 龙门右拉带脱离气缸伸出位延时
D356 CHANNEL  ; 出料NG气伸出位延时
D357 CHANNEL  ; 出料NG气缩回位延时
D36 CHANNEL  ; #1排位置
D370 CHANNEL  ; 氦检仪状态
D4000 CHANNEL  ; （龙门）左右机械手手动速度
D4010 CHANNEL  ; 左右取料点位
D4030 CHANNEL  ; 入盘（左右）X轴手动速度puls/s（浮点）
D4032 CHANNEL  ; 入盘（左右）X轴自动速度（浮点）
D4100 CHANNEL  ; （龙门）左右#1号点位置
D4102 CHANNEL  ; #2号点位置
D4104 CHANNEL  ; #3点位置
D4106 CHANNEL  ; #4点位置
D4108 CHANNEL  ; #5点位置
D4110 CHANNEL  ; #6点位置
D4112 CHANNEL  ; #7点位置
D4114 CHANNEL  ; #8点位置
D4116 CHANNEL  ; #9点位置
D4118 CHANNEL  ; #10点位置
D4120 CHANNEL  ; #11点位置
D4122 CHANNEL  ; #12点位置
D4124 CHANNEL  ; （龙门）左右#13号点位置
D4126 CHANNEL  ; #14号点位置
D4128 CHANNEL  ; （龙门）左右#15号点位置
D4130 CHANNEL  ; （龙门）左右#16号点位置
D4132 CHANNEL  ; （龙门）左右#17号点位置
D4134 CHANNEL  ; #18点位置
D4136 CHANNEL  ; （龙门）左右#19号点位置
D4138 CHANNEL  ; （龙门）左右#20号点位置
D4140 CHANNEL  ; （龙门）左右#21号点位置
D4142 CHANNEL  ; （龙门）左右#22号点位置
D4144 CHANNEL  ; （龙门）左右#23号点位置
D4146 CHANNEL  ; （龙门）左右#24号点位置
D4200 CHANNEL  ; 入盘（左右）X轴#1号位置脉冲(浮点)
D4202 CHANNEL  ; 入盘（左右）X轴#2号位置脉冲(浮点)
D4204 CHANNEL  ; 入盘（左右）X轴#3号位置脉冲(浮点)
D4206 CHANNEL  ; 入盘（左右）X轴#4号位置脉冲(浮点)
D4208 CHANNEL  ; 入盘（左右）X轴#5号位置脉冲(浮点)
D4210 CHANNEL  ; 入盘（左右）X轴#6号位置脉冲(浮点)
D4212 CHANNEL  ; 入盘（左右）X轴#18号位置脉冲(浮点)
D4214 CHANNEL  ; 入盘（左右）X轴#8号位置脉冲(浮点)
D4216 CHANNEL  ; 入盘（左右）X轴#9号位置脉冲(浮点)
D4218 CHANNEL  ; 入盘（左右）X轴#10号位置脉冲(浮点)
D4220 CHANNEL  ; 入盘（左右）X轴#11号位置脉冲(浮点)
D4222 CHANNEL  ; 入盘（左右）X轴#12号位置脉冲(浮点)
D4250 CHANNEL  ; 入盘（左右）X轴#1号位置脉冲
D4252 CHANNEL  ; 入盘（左右）X轴#2号位置脉冲
D4254 CHANNEL  ; 入盘（左右）X轴#3号位置脉冲)
D4256 CHANNEL  ; 入盘（左右）X轴#4号位置脉冲
D4258 CHANNEL  ; 入盘（左右）X轴#5号位置脉冲
D4260 CHANNEL  ; 入盘（左右）X轴#6号位置脉冲
D4262 CHANNEL  ; 入盘（左右）X轴#7号位置脉冲
D4264 CHANNEL  ; 入盘（左右）X轴#8号位置脉冲
D4266 CHANNEL  ; 入盘（左右）X轴#9号位置脉冲
D4268 CHANNEL  ; 入盘（左右）X轴#10号位置脉冲
D4270 CHANNEL  ; 入盘（左右）X轴#11号位置脉冲
D4272 CHANNEL  ; 入盘（左右）X轴#12号位置脉冲
D4280 CHANNEL  ; 入盘（左右）X轴取料位置脉冲（浮点）
D4282 CHANNEL  ; 入盘（左右）X轴取料位置脉冲
D4300 CHANNEL  ; 入盘（左右）X轴#13号位置脉冲(浮点)
D4302 CHANNEL  ; 入盘（左右）X轴#14号位置脉冲(浮点)
D4304 CHANNEL  ; 入盘（左右）X轴#15号位置脉冲(浮点)
D4306 CHANNEL  ; 入盘（左右）X轴#16号位置脉冲(浮点)
D4308 CHANNEL  ; 入盘（左右）X轴#17号位置脉冲(浮点)
D4310 CHANNEL  ; 入盘（左右）X轴#18号位置脉冲(浮点)
D4312 CHANNEL  ; 入盘（左右）X轴#19号位置
D4314 CHANNEL  ; 入盘（左右）X轴#20号位置脉冲(浮点)
D4316 CHANNEL  ; 入盘（左右）X轴#21号位置脉冲(浮点)
D4318 CHANNEL  ; 入盘（左右）X轴#22号位置脉冲(浮点)
D4320 CHANNEL  ; 入盘（左右）X轴#23号位置脉冲(浮点)
D4322 CHANNEL  ; 入盘（左右）X轴#24号位置脉冲(浮点)
D4350 CHANNEL  ; 入盘（左右）X轴#13号位置脉冲
D4352 CHANNEL  ; 入盘（左右）X轴#14号位置脉冲
D4354 CHANNEL  ; 入盘（左右）X轴#15号位置
D4356 CHANNEL  ; 入盘（左右）X轴#16号位置
D4358 CHANNEL  ; 入盘（左右）X轴#17号位置脉冲
D4360 CHANNEL  ; 入盘（左右）X轴#18号位置
D4362 CHANNEL  ; 入盘（左右）X轴#19号位置
D4364 CHANNEL  ; 入盘（左右）X轴#20号位置
D4366 CHANNEL  ; 入盘（左右）X轴#21号位置
D4368 CHANNEL  ; 入盘（左右）X轴#22号位置
D4370 CHANNEL  ; 入盘（左右）X轴#23号位置
D4372 CHANNEL  ; 入盘（左右）X轴#24号位置
D440 CHANNEL  ; 上料旋转步进自动状态加速度
D441 CHANNEL  ; 上料旋转步进自动状体减速度
D4414 CHANNEL  ; 入盘X轴脉冲_距离转换系数（二进制）
D4416 CHANNEL  ; 入盘X轴脉冲_距离转换系数（浮点）
D442 CHANNEL  ; 上料旋转步进自动速度puls/s
D4424 CHANNEL  ; 入盘X轴脉冲_距离（二进制）
D4426 CHANNEL  ; 入盘X轴脉冲_距离（浮点）
D4428 CHANNEL  ; （龙门)左右料机械手位置(mm)
D444 CHANNEL  ; 上料旋转自动位移量
D4440 CHANNEL  ; 左右机械手正向行程脉冲
D4444 CHANNEL  ; 左右机械手反向行程
D4448 CHANNEL  ; 左右机械手反向行程脉冲
D446 CHANNEL  ; 上料旋转步进自动状态起动速度
D4480 CHANNEL  ; 入盘（左右）X轴手动状态加速度
D4481 CHANNEL  ; 入盘（左右）X轴手动状态减速度
D4482 CHANNEL  ; 入盘（左右）X轴手动速度脉冲puls/s
D4484 CHANNEL  ; 入盘（左右）X轴手动位移量
D4486 CHANNEL  ; 入盘（左右）X轴手动状态启动速度
D4490 CHANNEL  ; 入盘（左右）X轴自动状态加速度
D4491 CHANNEL  ; 入盘（左右）X轴自动状态减速度
D4492 CHANNEL  ; 入盘（左右）X轴自动速度脉冲puls/s
D4494 CHANNEL  ; 入盘（左右）X轴自动位移量
D4496 CHANNEL  ; 入盘（左右）X轴自动状态启动速度
D450 CHANNEL  ; 上料旋转步进手动状态加速度
D4500 CHANNEL  ; 入盘（前后）机械手手动速度mm/s
D4502 CHANNEL  ; 入盘（前后）机械手自动速度
D451 CHANNEL  ; 上料旋转步进手动状态减速度
D4510 CHANNEL  ; #1排位置
D4512 CHANNEL  ; #2排位置
D4514 CHANNEL  ; （龙门）前后机械手取料位置
D452 CHANNEL  ; 上料旋转步进手动速度puls/s
D4530 CHANNEL  ; 入盘（前后）Y轴手动速度puls/s（浮点）
D4532 CHANNEL  ; 入盘（前后）Y轴手动速度脉冲puls/s
D4534 CHANNEL  ; 入盘（前后）Y轴自动速度puls/s（浮点）
D4536 CHANNEL  ; 入盘（前后）Y轴自动速度脉冲puls/s
D454 CHANNEL  ; 进料旋转手动位移量
D4540 CHANNEL  ; （龙门）前后机械手#1排位置脉冲(浮点)
D4542 CHANNEL  ; （龙门）前后机械手#1排位置脉冲
D4544 CHANNEL  ; （龙门）前后机械手取料位置脉冲（浮点）
D4546 CHANNEL  ; （龙门）前后机械手#1排位置脉冲
D4550 CHANNEL  ; （龙门）前后机械手#2排位）前后机械手取料位(浮点)
D4552 CHANNEL  ; （龙门）前后机械手取料位置脉冲
D456 CHANNEL  ; 上料旋转步进手动状态起动速度
D46 CHANNEL  ; 氦检设定时间
D460 CHANNEL  ; 下料旋转步进自动状态加速度
D461 CHANNEL  ; 下料旋转步进自动状态减速度
D4614 CHANNEL  ; 入盘Y轴脉冲_距离（二进制）
D4616 CHANNEL  ; 入盘前后Y轴脉冲_距离转换系数（浮点）
D462 CHANNEL  ; 下料旋转步进自动速度puls/s
D4624 CHANNEL  ; 入盘（前后）Y轴当前脉冲
D4626 CHANNEL  ; 入盘（前后）Y轴当前脉冲（浮点）
D4628 CHANNEL  ; 入盘（前后）Y轴当前位置
D464 CHANNEL  ; 下料旋转自动位移量
D4640 CHANNEL  ; 前后料机械手行程
D4644 CHANNEL  ; 前后机械手反向行程
D4648 CHANNEL  ; 前后机械手反向行程
D466 CHANNEL  ; 下料旋转步进自动状态起动速度
D470 CHANNEL  ; 下料旋转步进手动状态加速度
D4700 CHANNEL  ; （龙门）上下料机械手上手动速度
D4702 CHANNEL  ; （龙门）上下料机械手自动速度
D471 CHANNEL  ; 下料旋转步进手动状态减速度
D4710 CHANNEL  ; （龙门）抓料机械手进料位置
D4712 CHANNEL  ; （龙门）抓料机械手OK位置
D472 CHANNEL  ; 下料旋转步进手动速度puls/s
D4730 CHANNEL  ; 入盘（升降）Z轴手动速度puls/s
D4734 CHANNEL  ; 入盘（升降）Z轴自动速度puls/s
D4736 CHANNEL  ; 入盘（升降）Z轴自动速度puls/s
D474 CHANNEL  ; 下料旋转手动位移量
D4740 CHANNEL  ; （龙门）抓料机械手进料位置脉冲(浮点)
D4742 CHANNEL  ; （龙门）抓料机械手进料位置脉冲
D4744 CHANNEL  ; （龙门）抓料机械手OK位置脉冲(浮点)
D4746 CHANNEL  ; （龙门）抓料机械手OK位置脉冲
D476 CHANNEL  ; 下料旋转步进手动状态起动速度
D4814 CHANNEL  ; 入盘升降轴脉冲_距离转换系数（二进制）
D4816 CHANNEL  ; 入盘升降轴脉冲_距离转换系数（浮点）
D4824 CHANNEL  ; 入盘升降脉冲
D4826 CHANNEL  ; （龙门）入盘升降脉冲当前脉冲(浮点)
D4828 CHANNEL  ; （龙门）入盘升降脉冲当前位置(mm)
D4840 CHANNEL  ; 抓料机械手正向行程脉冲
D4844 CHANNEL  ; 前后 抓料机械手反向行程
D4848 CHANNEL  ; 前后 抓料机械手反向行程脉冲
D4870 CHANNEL  ; 入盘（升降）Z轴手动状态加速度
D4871 CHANNEL  ; 入盘（升降）Z轴手动状态减速度
D4872 CHANNEL  ; 入盘（升降）Z轴手动速度脉冲puls/s
D4874 CHANNEL  ; 入盘（升降）Z轴手动行程脉冲
D4876 CHANNEL  ; 入盘（升降）Z轴手动状态启动速度
D4880 CHANNEL  ; 入盘（升降）Z轴自动状态加速度
D4881 CHANNEL  ; 入盘（升降）Z轴自动状态减速度
D4882 CHANNEL  ; 入盘（升降）Z轴自动速度脉冲puls/s
D4884 CHANNEL  ; 抓料机械手手动位移量
D4886 CHANNEL  ; 入盘（升降）Z轴自动状态启动速度
D4900 CHANNEL  ; 料盘手动速度
D4902 CHANNEL  ; 运行速度
D4910 CHANNEL  ; 上料盒位置
D4912 CHANNEL  ; 放料盒位置
D4924 CHANNEL  ; 料盘当前脉冲
D4926 CHANNEL  ; 料盘当前脉冲（浮点）
D4928 CHANNEL  ; 料盘当前位置
D4934 CHANNEL  ; 料盒升降轴脉冲_距离转换系数（二进制）
D4936 CHANNEL  ; 料盒升降轴脉冲_距离转换系数（浮点）
D4940 CHANNEL  ; 料盘手动速度puls/s（浮点）
D4942 CHANNEL  ; 料盘手动速度脉冲
D4944 CHANNEL  ; 料盘自动速度puls/s（浮点）
D4946 CHANNEL  ; 料盘自动速度脉冲
D4950 CHANNEL  ; （龙门）料盘机到上料位置脉冲(浮点)
D4952 CHANNEL  ; （龙门）料盘机到上料位置脉冲
D4954 CHANNEL  ; （龙门）料盘机到放料位置脉冲(浮点)
D4956 CHANNEL  ; （龙门）料盘机到放料位置脉冲
D50 CHANNEL  ; 检漏口压力指数
D502 CHANNEL  ; 进料机械手自动速度mm/s
D52 CHANNEL  ; 检漏口压力底数
D520 CHANNEL  ; 上料旋转步进自动速度puls/s
D524 CHANNEL  ; 上料旋转步进手动速度puls/s
D530 CHANNEL  ; 下料旋转步进自动速度puls/s
D534 CHANNEL  ; 下料旋转步进手动速度puls/s
D54 CHANNEL  ; 漏率指数
D540 CHANNEL  ; 下料机械手电池数量
D56 CHANNEL  ; 漏率底数
D600 CHANNEL  ; 进料机械手左进料位置脉冲(浮点)
D6000 CHANNEL  ; #1扫码长度
D604 CHANNEL  ; 上料机械手左取料位置脉冲
D610 CHANNEL  ; 进料机械手腔体1位置脉冲(浮点)
D614 CHANNEL  ; 上料机械手腔体1位置脉冲
D620 CHANNEL  ; 进料机械手腔体2位置(浮点)
D624 CHANNEL  ; 上料机械手腔体2位置脉冲
D640 CHANNEL  ; 进料机械手右进料位置(浮点)
D644 CHANNEL  ; 上料机械手右进料位置脉冲
D650 CHANNEL  ; 出料机械手腔体1位置(浮点)
D654 CHANNEL  ; 出料机械手腔体1位置脉冲
D66 CHANNEL  ; 条码设置长度
D660 CHANNEL  ; 出料机械手腔体2位置(浮点)
D664 CHANNEL  ; 出料机械手腔体2位置脉冲
D670 CHANNEL  ; 出料机械手OK左位置(浮点)
D674 CHANNEL  ; 出料机械手OK左位置脉冲
D680 CHANNEL  ; 出料机械手OK右位置(浮点)
D684 CHANNEL  ; 出料机械手OK右位置脉冲
D688 CHANNEL  ; 上料旋转进料反向位置脉冲
D690 CHANNEL  ; 下料机械手NG位置(浮点)
D692 CHANNEL  ; 上料升降轴输出脉冲-读取值（浮点数）
D694 CHANNEL  ; 下料机械手NG位置脉冲
D696 CHANNEL  ; 上料升降轴脉冲_距离转换系数（浮点）
D698 CHANNEL  ; 上料升降轴当前位置（浮点）
D7 CHANNEL  ; #2排位置
D700 CHANNEL  ; 下料旋转进料位置(浮点)
D7000 CHANNEL  ; 扫码长度
D7001 CHANNEL  ; 电池条码
D7020 CHANNEL  ; 条码在爪子1
D704 CHANNEL  ; 下料旋转进料位置脉冲
D7040 CHANNEL  ; 电池条码在爪子2
D7060 CHANNEL  ; #3条码缓存
D710 CHANNEL  ; 旋转步进正向行程脉冲
D7101 CHANNEL  ; #2电池条码
D7120 CHANNEL  ; #1腔体#1条码
D714 CHANNEL  ; 旋转步进反向行程
D7140 CHANNEL  ; #1腔体#2条码
D7160 CHANNEL  ; #1腔体#3条码
D718 CHANNEL  ; 旋转步进反向行程脉冲
D7180 CHANNEL  ; #1腔体#4条码
D72 CHANNEL  ; 托盘条码长度
D7200 CHANNEL  ; 托盘码长度
D7220 CHANNEL  ; #2腔体#1条码
D7240 CHANNEL  ; #2腔体#2条码
D7260 CHANNEL  ; #2腔体#3条码
D7280 CHANNEL  ; #2腔体#4条码
D7360 CHANNEL  ; 下料机械手#3条码
D7380 CHANNEL  ; 下料机械手#4条码
D74 CHANNEL  ; 托盘条码字节数
D76 CHANNEL  ; 托盘条码字符串字节数
D800 CHANNEL  ; 进NG左位置-HMI
D8000 CHANNEL  ; 检漏状态第一字节
D8001 CHANNEL  ; 检漏状态第二字节
D8002 CHANNEL  ; 检漏状态结束字节
D8010 CHANNEL  ; 待机状态第一字节
D8011 CHANNEL  ; 待机状态第二字节
D8012 CHANNEL  ; 待机状态结束字节
D802 CHANNEL  ; （龙门）上下料机械手手动速度mm/s
D8020 CHANNEL  ; 定标状态第一字节
D8021 CHANNEL  ; 定标状态第二字节
D8022 CHANNEL  ; 定标状态结束字节
D8030 CHANNEL  ; 启动状态第一字节
D8031 CHANNEL  ; 启动状态第二字节
D8032 CHANNEL  ; 启动状态结束字节
D804 CHANNEL  ; 进NG左位置-HMI
D8040 CHANNEL  ; 错误状态第一字节
D8041 CHANNEL  ; 错误状态第二字节
D8042 CHANNEL  ; 错误状态结束字节
D8050 CHANNEL  ; 暂停状态第一字节
D8051 CHANNEL  ; 暂停状态第二字节
D8052 CHANNEL  ; 暂停状态结束字节
D810 CHANNEL  ; 进NG右位置-HMI
D8100 CHANNEL  ; 氦检仪状态(1-检漏,2-待机,3-启动,4-定标,5-错误,6-暂停)
D814 CHANNEL  ; 进NG右位置-HMI
D9000 CHANNEL  ; PC通信标志
D9003 CHANNEL  ; PC交互
D9100 CHANNEL  ; MES进站结果 1-0K 2-NG
D9102 CHANNEL  ; #1腔体数据处理完成
D9103 CHANNEL  ; #3腔体数据处理完成
D9300 CHANNEL  ; 条码状态 0-EMS已读取 <>0 触发扫码
D9302 CHANNEL  ; 条码结果 0-OK，1-NG
D9303 CHANNEL  ; #2条码结果 0-OK, 1-NG
H0.00 BOOL  ; #1腔体屏蔽-HMI
H0.01 BOOL  ; #2腔体屏蔽-HMI
H0.02 BOOL  ; 扫码屏蔽-HMI
H0.03 BOOL  ; 电脑屏蔽-HMI
H0.04 BOOL  ; 门磁开关屏蔽-HMI
H0.05 BOOL  ; 空跑程序-HMI
H0.06 BOOL  ; MES屏蔽-HMI
H0.07 BOOL  ; 托盘扫码屏蔽-HMI
H0.08 BOOL  ; 氦检仪屏蔽
H0.09 BOOL  ; 入盘启用0ff/屏蔽on
H0.10 BOOL  ; 单个测试
H11.00 BOOL  ; 上料机械手归零完成
H11.01 BOOL  ; 下料机械手归零完成
H11.02 BOOL  ; 入盘升降归零完成
H11.03 BOOL  ; 入盘X轴归零完成
H11.04 BOOL  ; 入盘Y轴归零完成
H11.05 BOOL  ; 料盘升降归零完成
H16.04 BOOL  ; 下料夹爪3手动松开
H16.11 BOOL  ; 出料输送带手动
H1.00 BOOL  ; 扫码阻挡气缸缩回位-HMI
H1.01 BOOL  ; 扫码阻挡气缸伸出位-HMI
H1.02 BOOL  ; 扫码定位气缸缩回位-HMI
H1.03 BOOL  ; 扫码定位气缸伸出位-HMI
H1.04 BOOL  ; 抓料阻挡气缸缩回位-HMI
H1.05 BOOL  ; 抓料阻挡气缸伸出位-HMI
H1.06 BOOL  ; 上料提升气缸缩回位-HMI
H1.07 BOOL  ; 上料提升气缸伸出位-HMI
H1.08 BOOL  ; 上料左夹爪升降气缸缩回位-HMI
H1.09 BOOL  ; 上料左夹爪升降气缸伸出位-HMI
H1.10 BOOL  ; 上料右夹爪升降气缸缩回位-HMI
H1.11 BOOL  ; 上料右夹爪升降气缸伸出位-HMI
H1.12 BOOL  ; 上料左夹爪张开位-HMI
H1.13 BOOL  ; 上料左夹爪夹紧位-HMI
H1.14 BOOL  ; 上料右夹爪张开位-HMI
H1.15 BOOL  ; 上料右夹爪夹紧位-HMI
H20.00 BOOL  ; 扫码OK
H20.01 BOOL  ; 扫码OK在抓电池位
H20.05 BOOL  ; 在扫码位与抓料位有电池
H20.10 BOOL  ; 扫码NG
H20.11 BOOL  ; 扫码NG在抓电池位
H21.02 BOOL  ; 上料夹爪1手动夹紧
H21.03 BOOL  ; 上料夹爪2手动夹紧
H22 CHANNEL  ; 进料机械手状态
H22.00 BOOL  ; 左上料夹爪有料
H22.02 BOOL  ; 左夹爪有OK料
H22.03 BOOL  ; 右夹爪电池OK
H22.04 BOOL  ; 左夹爪有NG料
H22.05 BOOL  ; NG槽有料
H22.06 BOOL  ; 扫码NG拨料完成
H22.10 BOOL  ; 上料机械手夹爪1抓OK料完成
H22.11 BOOL  ; 夹爪1有NG料
H22.12 BOOL  ; 右上料夹爪有料_OK
H22.13 BOOL  ; 夹爪2有NG料
H22.14 BOOL  ; 上料机械手抓料完成
H23 CHANNEL  ; #3腔体保持状态
H23.01 BOOL  ; 1#上料夹爪夹紧(A)
H23.02 BOOL  ; 2#上料夹爪夹紧(A)
H23.03 BOOL  ; 上料机械手抓扫码NG料完成
H23.11 BOOL  ; #1上料夹爪有料
H23.12 BOOL  ; .#2上料夹爪有料
H24 CHANNEL  ; #4腔体保持状态
H25 CHANNEL  ; 出料机械手状态
H25.00 BOOL  ; 下料机械手有料
H25.01 BOOL  ; 下料夹爪产品NG
H25.02 BOOL  ; NG产品放料完成
H25.03 BOOL  ; OK产品放料完成
H25.04 BOOL  ; NG拨料完成
H25.05 BOOL  ; 机械手#1腔体取料
H25.06 BOOL  ; 机械手#2腔体取料
H25.12 BOOL  ; 出料托盘#3位置有料
H25.13 BOOL  ; 出料托盘#4位置有料
H26.00 BOOL  ; 下料夹爪夹紧
H26.01 BOOL  ; 1腔有料
H26.02 BOOL  ; 2腔有料
H26.05 BOOL  ; #1腔位置3有料
H26.06 BOOL  ; #1腔位置4有料
H26.09 BOOL  ; #2腔位置3有料
H26.10 BOOL  ; #2腔位置4有料
H2.00 BOOL  ; 下料提升气缸缩回位-HMI
H2.01 BOOL  ; 下料提升气缸伸出位-HMI
H2.02 BOOL  ; 下料夹爪升降气缸缩回位-HMI
H2.03 BOOL  ; 下料夹爪升降气缸伸出位-HMI
H2.04 BOOL  ; 下料左夹爪张开位-HMI
H2.05 BOOL  ; 下料左夹爪夹紧位-HMI
H2.06 BOOL  ; 下料右夹爪张开位-HMI
H2.07 BOOL  ; 下料右夹爪夹紧位-HMI
H2.08 BOOL  ; #1合模气缸缩回位-HMI
H2.09 BOOL  ; #1合模气缸伸出位-HMI
H2.10 BOOL  ; #2合模气缸缩回位-HMI
H2.11 BOOL  ; #2合模气缸伸出位-HMI
H2.12 BOOL  ; 扫码NG拨料气缸缩回位-HMI
H2.13 BOOL  ; 扫码NG拨料气缸伸出位-HMI
H2.14 BOOL  ; 料盒定位气缸缩回位-HMI
H2.15 BOOL  ; 料盒定位气缸伸出位-HMI
H31.01 BOOL  ; #1腔体自检OK
H31.02 BOOL  ; #2腔体自检OK
H31.03 BOOL  ; 4#下料夹爪夹紧(A)
H32.10 BOOL  ; 1#上料夹爪夹紧(NG料)(A)
H32.11 BOOL  ; 2#上料夹爪夹紧(NG料)(A)
H33.00 BOOL  ; #1腔体放料完成
H33.01 BOOL  ; #1腔体#1位有电池
H33.02 BOOL  ; #1腔体产品NG
H33.03 BOOL  ; #1腔体测试中
H33.04 BOOL  ; #1腔位置1有料
H33.05 BOOL  ; #1腔位置2有料
H34.00 BOOL  ; #2腔体放料完成
H34.01 BOOL  ; #2腔体#1位有电池
H34.02 BOOL  ; #2腔体产品NG
H34.03 BOOL  ; #2腔体测试中
H34.04 BOOL  ; #2腔位置1有料
H34.05 BOOL  ; #2腔位置2有料
H3.00 BOOL  ; 料盒上阻挡气缸缩回位-HMI
H3.01 BOOL  ; 料盒上阻挡气缸伸出位-HMI
H3.02 BOOL  ; 料盒下阻挡气缸缩回位-HMI
H3.03 BOOL  ; 料盒下阻挡气缸伸出位-HMI
H3.04 BOOL  ; #1上顶升左气缸缩回位-HMI
H3.05 BOOL  ; #2上顶升左气缸伸出位-HMI
H3.06 BOOL  ; #1上顶升右气缸缩回位-HMI
H3.07 BOOL  ; #2上顶升右气缸伸出位-HMI
H3.08 BOOL  ; #1上顶升左气缸缩回位-HMI
H3.09 BOOL  ; #1上顶升左气缸伸出位-HMI
H3.10 BOOL  ; #2上顶升右气缸缩回位-HMI
H3.11 BOOL  ; #1上顶升右气缸伸出位-HMI
H3.12 BOOL  ; #2下顶升左气缸缩回位-HMI
H3.13 BOOL  ; #2下顶升左气缸伸出位-HMI
H3.14 BOOL  ; #2下顶升右气缸缩回位-HMI
H3.15 BOOL  ; #2下顶升右气缸伸出位-HMI
H44.01 BOOL  ; 1#下料夹爪夹紧(A)
H44.02 BOOL  ; 2#下料夹爪夹紧(A)
H44.11 BOOL  ; #1下料夹爪有料
H44.12 BOOL  ; #2下料夹爪有料
H44.13 BOOL  ; #2下料夹爪无料
H45.01 BOOL  ; 下料夹爪1手动松开
H45.02 BOOL  ; 下料夹爪2手动松开
H4.00 BOOL  ; #2下顶升左气缸缩回位-HMI
H4.01 BOOL  ; #2下顶升左气缸伸出位-HMI
H4.02 BOOL  ; #2下顶升右气缸缩回位-HMI
H4.03 BOOL  ; #2下顶升右气缸伸出位-HMI
H4.04 BOOL  ; 龙门左拉带脱离气缸缩回位-HMI
H4.05 BOOL  ; 龙门左拉带脱离气缸伸出位-HMI
H4.06 BOOL  ; 龙门右拉带脱离气缸伸出位-HMI
H4.07 BOOL  ; 腔体有料信号-HMI
H4.08 BOOL  ; 料盒#1电池有料信号-HMI
H4.09 BOOL  ; 料盒#2电池有料信号-HMI
H4.10 BOOL  ; 料盒#3电池有料信号-HMI
H4.11 BOOL  ; 料盒#4电池有料屏蔽-HMI
H4.12 BOOL  ; 料盒#5电池有料屏蔽-HMI
H4.13 BOOL  ; 料盒#6电池有料屏蔽-HMI
H4.14 BOOL  ; 料盒#7电池有料屏蔽-HMI
H4.15 BOOL  ; 料盒#8电池有料信号屏蔽-HMI
H51.10 BOOL  ; 料盘有料感应屏蔽
H55.01 BOOL  ; 入盘夹爪气缸张开位
H55.02 BOOL  ; 入盘夹爪夹紧
H55.03 BOOL  ; 出料输出带有料
H55.10 BOOL  ; 输送带有#1-OK料
H55.11 BOOL  ; 输送带有#2-OK料
H55.12 BOOL  ; 龙门料抓有料
H55.13 BOOL  ; 放有料1
H55.14 BOOL  ; 放有料2
H58.01 BOOL  ; #1位有电池(记忆)
H58.02 BOOL  ; #2位有电池(记忆)
H58.03 BOOL  ; #3位有电池(记忆)
H58.04 BOOL  ; #4位有电池(记忆)
H58.05 BOOL  ; #5位有电池(记忆)
H58.06 BOOL  ; #6位有电池(记忆)
H58.07 BOOL  ; #7位有电池(记忆)
H58.08 BOOL  ; #8位有电池(记忆)
H58.09 BOOL  ; #9位有电池(记忆)
H58.10 BOOL  ; #10位有电池(记忆)
H58.11 BOOL  ; #11位有电池(记忆)
H58.12 BOOL  ; #12位有电池(记忆)
H59.01 BOOL  ; #13位有电池(记忆)
H59.02 BOOL  ; #14位有电池(记忆)
H59.03 BOOL  ; #15位有电池(记忆)
H59.04 BOOL  ; #16位有电池(记忆)
H59.05 BOOL  ; #17位有电池(记忆)
H59.06 BOOL  ; #18位有电池(记忆)
H59.07 BOOL  ; #19位有电池(记忆)
H59.08 BOOL  ; #20位有电池(记忆)
H59.09 BOOL  ; #21位有电池(记忆)
H59.10 BOOL  ; #22位有电池(记忆)
H59.11 BOOL  ; #23位有电池(记忆)
H59.12 BOOL  ; #24位有电池(记忆)
H5.01 BOOL  ; 拉带对接信号屏蔽
H5.02 BOOL  ; 料盒#11电池有料屏蔽-HMI
H5.03 BOOL  ; 料盒#12电池有料屏蔽-HMI
H5.04 BOOL  ; 料盒#13电池有料屏蔽-HMI
H5.06 BOOL  ; 料盒#15电池有料屏蔽-HMI
H5.07 BOOL  ; 料盒#16电池有料屏蔽-HMI
H5.08 BOOL  ; 料盒#17电池有料屏蔽-HMI
H5.09 BOOL  ; 料盒#18电池有料屏蔽-HMI
H5.10 BOOL  ; 料盒#19电池有料屏蔽-HMI
H5.11 BOOL  ; 料盒#20电池有料屏蔽-HMI
H5.12 BOOL  ; 料盒#21电池有料屏蔽-HMI
H5.13 BOOL  ; 料盒#22电池有料屏蔽
H5.14 BOOL  ; 料盒#23电池有料屏蔽-HMI
H5.15 BOOL  ; 料盒#24电池有料屏蔽-HMI
H6.00 BOOL  ; 机台方向选择(0:左进右出,1:右进左出)
H6.10 BOOL  ; 出料NG气伸出位屏蔽
H6.11 BOOL  ; 出料NG气缸缩回位屏蔽
H6.12 BOOL  ; 上料柔性报警屏蔽
H6.13 BOOL  ; 下料柔性报警屏蔽
H6.14 BOOL  ; 入盘柔性报警屏蔽
H73.01 BOOL  ; 下#1有空料盒
H73.02 BOOL  ; 下#2有空料盒
H73.03 BOOL  ; 下输送带有料
H73.04 BOOL  ; 料盒升降架上有空料盒
H73.05 BOOL  ; 料盒在入电池位
H73.06 BOOL  ; 下料输送带有满料
H73.07 BOOL  ; 满料在缓存输送带
H73.08 BOOL  ; 下#1位有料满电池
H73.09 BOOL  ; 下电池#2有满料盒
H8.00 BOOL  ; 龙门升降气缸缩回位 HIM屏蔽
H8.01 BOOL  ; 龙门升降气缸伸出位 HIM屏蔽
H8.02 BOOL  ; 龙门夹爪气缸夹紧HIM屏蔽
H8.03 BOOL  ; 龙门夹爪气缸松开HIM屏蔽
H8.04 BOOL  ; #1上料盒到位感应屏蔽HIM
H8.05 BOOL  ; #2上料盒到位感应 HIM
H8.06 BOOL  ; 料盒到位感应
H8.07 BOOL  ; #1下料盒到位感应HIM'
H8.08 BOOL  ; #2下料盒到位感应HIM'
H8.09 BOOL  ; #3下料盒到位感应HIM
T0000 BOOL  ; 扫码阻挡气缸缩回位延时
T0001 BOOL  ; 扫码阻挡气缸伸出位延时
T0002 BOOL  ; 抓料阻挡气缸缩回位延时
T0003 BOOL  ; 抓料阻挡气缸伸出位延时
T0004 BOOL  ; 下料提升气缸伸出位延时
T0005 BOOL  ; 上料提升气缸缩回位延时
T0006 BOOL  ; 上料提升气缸伸出位延时
T0007 BOOL  ; 上料左升降气缸缩回位
T0008 BOOL  ; 上料左夹爪升降气缸伸出位延时
T0009 BOOL  ; 上料右升降气缸缩回位
T0010 BOOL  ; 上料右夹爪升降气缸伸出位延时
T0011 BOOL  ; 上料夹爪1张开位延时
T0012 BOOL  ; 上料左夹爪夹紧位延时
T0013 BOOL  ; 上料右夹爪张开位延时
T0014 BOOL  ; 上料右夹爪夹紧位延时
T0015 BOOL  ; 扫码NG拨料气缸缩回位延时
T0016 BOOL  ; 扫码NG拨料气缸伸出位延时
T0017 BOOL  ; #1合模气缸缩回位延时
T0018 BOOL  ; #1合模气缸伸出位延时
T0019 BOOL  ; #2合模气缸缩回位延时
T0020 BOOL  ; #2合模气缸伸出位延时
T0021 BOOL  ; 下料提升气缸缩回位延时
T0022 BOOL  ; 下料提升气缸伸出位延时
T0023 BOOL  ; 下料升降气缸缩回位延时
T0024 BOOL  ; 下料夹爪升降气缸伸出位延时
T0025 BOOL  ; 下料夹爪1张开位延时
T0026 BOOL  ; 下料左夹爪夹紧位延时
T0027 BOOL  ; 下料夹爪2张开位延时
T0028 BOOL  ; 下料右夹爪夹紧位延时
T0029 BOOL  ; 出料NG拨料气缸缩回位延时
T0030 BOOL  ; 出料NG拨料气缸伸出位延时
T0031 BOOL  ; 料盒定位气缸缩回位延时
T0032 BOOL  ; 料盒定位气缸伸出位延时
T0033 BOOL  ; 料盒上阻挡气缸缩回位延时
T0034 BOOL  ; 料盒上阻挡气缸伸出位延时
T0035 BOOL  ; 料盒下阻挡气缸缩回位延时
T0036 BOOL  ; 料盒下阻挡气缸伸出位延时
T0037 BOOL  ; #1上顶升左气缸缩回位延时
T0038 BOOL  ; #2上顶升左气缸伸出位延时
T0039 BOOL  ; #2上顶升右气缸缩回位延时
T0040 BOOL  ; #2上顶升右气缸伸出位延时
T0041 BOOL  ; #1上顶升左气缸缩回位延时
T0042 BOOL  ; #1上顶升左气缸伸出位延时
T0043 BOOL  ; #1上顶升右气缸缩回位延时
T0044 BOOL  ; #1上顶升右气缸伸出位延时
T0045 BOOL  ; #2下顶升左气缸缩回位延时
T0046 BOOL  ; #2下顶升左气缸伸出位延时
T0047 BOOL  ; #2下料顶升右气缸缩回位延时
T0048 BOOL  ; #2下顶升右气缸伸出位延时
T0049 BOOL  ; #2下顶升左气缸缩回位延时
T0050 BOOL  ; #1下顶升左气缸伸出位延时
T0051 BOOL  ; #1下顶升右气缸缩回位延时
T0052 BOOL  ; #1下顶升右气缸伸出位延时
T0053 BOOL  ; 龙门左拉带脱离气缸缩回位延时
T0054 BOOL  ; 入盘左拉带脱离气缸伸出位
T0055 BOOL  ; 龙门右拉带脱离气缸缩回位延时
T0056 BOOL  ; 入盘右拉带脱离气缸伸出位延时
T0057 BOOL  ; 入盘升降气缸缩回位延时
T0058 BOOL  ; 入盘升降气缸伸出位延时
T0059 BOOL  ; 入盘夹爪气缸松开延时
T0060 BOOL  ; 龙门夹爪气缸夹紧延时
T0061 BOOL  ; #1上料盒到位感应延时报警
T0062 BOOL  ; #2上料盒有料感应报警
T0063 BOOL  ; 料盒到位感应延时
T0064 BOOL  ; #1下料盒到位感应延时
T0065 BOOL  ; #2下料盒到位感应延时
T0066 BOOL  ; #3下料盒有料感应
T0067 BOOL  ; 出料夹爪1张开报警
T0068 BOOL  ; 出料夹爪1夹紧报警
T0069 BOOL  ; 出料夹爪2张开报警
T0070 BOOL  ; 清料延时
T0107 BOOL  ; 延时关复位
T0110 BOOL  ; PC运行标志断开时间
T0111 BOOL  ; PC通信正常持续时间
T0112 BOOL  ; 氦检仪通信异常时间
T0113 BOOL  ; 扫码通信异常
T0114 BOOL  ; #1真空计断线延时
T0115 BOOL  ; #2真空计断线延时
T0116 BOOL  ; 报警延时关
T0118 BOOL  ; 系统运行延时
T0160 BOOL  ; 进料旋转回#1待料角度延时
T0161 BOOL  ; 进料旋转回#2待料位置延时
T0162 BOOL  ; 进料旋转回进料角度延时
T0200 BOOL  ; 扫码位有电感应延时
T0201 BOOL  ; 扫码位无电感应延时
T0202 BOOL  ; 抓料位有托盘感应延时
T0203 BOOL  ; 抓料位无托盘感应延时
T0204 BOOL  ; 抓料位有电池感应延时
T0205 BOOL  ; 抓料位无电池感应延时
T0207 BOOL  ; 空跑延时给信号
T0209 BOOL  ; 电池流出延时
T0210 BOOL  ; 扫码后判断延时
T0211 BOOL  ; 扫描缺料持续时间
T0212 BOOL  ; 隔离阻挡气缸延时放开
T0220 BOOL  ; 进料机械手左取料位置延时
T0221 BOOL  ; 进料机械手右取料位置延时
T0222 BOOL  ; 进料机械手回#1腔体位置
T0223 BOOL  ; 进料机械手回#2腔体位置
T0224 BOOL  ; 进料机械手手动回左NG位延时
T0225 BOOL  ; 进料机械手手动回右NG位延时
T0226 BOOL  ; 上料爪1打开延时时
T0227 BOOL  ; 上料爪2打开延时时
T0230 BOOL  ; #1合模气缸不在缩回位异常信息持续时间
T0231 BOOL  ; 进料夹爪不在张开位异常信息持续时间
T0232 BOOL  ; #2合模气缸不在缩回位异常信息持续时间
T0233 BOOL  ; 进料夹爪不在张开位异常信息持续时间
T0234 BOOL  ; 进料提升气缸不在缩回位异常信息持续时间
T0235 BOOL  ; 进料机械手没归零异常信息持续时间
T0236 BOOL  ; 进料机械手到达左极限信息持续时间
T0237 BOOL  ; 进料机械手到达右极限信息持续时间
T0238 BOOL  ; 出料机械手避让位置异常信息持续时间
T0239 BOOL  ; 出料机械手避让位置异常信息持续时间
T0250 BOOL  ; 进料机械手回进料位置延时
T0251 BOOL  ; 进料机械手回右进料位置延时
T0252 BOOL  ; 进料机械手回#1腔体位置延时
T0253 BOOL  ; 进料机械手回#2腔体位置延时
T0261 BOOL  ; 上料机械伺服复位时间
T0262 BOOL  ; 上料机械手报警信号持续时间
T0300 BOOL  ; 氦捡仪稳定时间
T0301 BOOL  ; 氦检仪状体判断延时
T0302 BOOL  ; 上料旋转回进料位置延时
T0303 BOOL  ; 检漏口压力判断延时
T0304 BOOL  ; 漏率判断延时
T0305 BOOL  ; 氦捡仪稳定时间
T0310 BOOL  ; 真空泵打开延时
T0311 BOOL  ; 真空泵断开延时
T0312 BOOL  ; #1腔体抽气时间
T0314 BOOL  ; #1腔体自检保压前延时
T0315 BOOL  ; #1腔体自检保压延时
T0316 BOOL  ; 破真空阀打开延时
T0320 BOOL  ; 进料提升气缸不在原位信息持续时间
T0321 BOOL  ; 出料提升气缸不在原位信息持续时间
T0322 BOOL  ; #1腔体真空值大于破真空设定值信息持续事假
T0323 BOOL  ; #1抽气阀打开异常信息持续时间
T0324 BOOL  ; #1氦检阀打开异常信息持续时间
T0325 BOOL  ; #1破真空阀打开异常信息持续时间
T0326 BOOL  ; #1吹气阀打开异常信息持续时间
T0327 BOOL  ; #1腔体复位破真空延时
T0328 BOOL  ; #1腔体达到破真空持续时间
T0330 BOOL  ; #1抽气阀打开延时(A)
T0331 BOOL  ; #1腔体抽气时间
T0332 BOOL  ; #1氦检阀打开延时
T0333 BOOL  ; 氦检持续时间
T0334 BOOL  ; #1氦检阀打开抽气阀关闭延时
T0335 BOOL  ; #1腔体数据传输延时
T0336 BOOL  ; 测试结束后抽残气延时
T0337 BOOL  ; 抽残气时间
T0338 BOOL  ; #1腔体破真空延时
T0339 BOOL  ; #1腔体破真空值到达
T0340 BOOL  ; #1腔氦检阀关闭延时
T0350 BOOL  ; #2腔体复位破真空延时
T0351 BOOL  ; #2腔体达到破真空持续时间
T0360 BOOL  ; #2腔体抽气时间
T0362 BOOL  ; #2腔体自检保压前延时
T0363 BOOL  ; #2腔体自检保压延时
T0364 BOOL  ; 破真空阀打开延时
T0370 BOOL  ; 进料提升气缸不在原位异常信息持续时间
T0371 BOOL  ; 出料提升气缸不在原位异常信息持续时间
T0372 BOOL  ; #2腔体真空值大于破真空设定值信息持续时间
T0373 BOOL  ; #2抽气阀异常信息持续时间
T0374 BOOL  ; #2氦检阀异常信息持续时间
T0375 BOOL  ; #2破真空阀异常信息持续时间
T0376 BOOL  ; #2吹气阀异常信息持续时间
T0380 BOOL  ; #2抽气阀打开延时(A)
T0381 BOOL  ; #2腔体抽气时间
T0382 BOOL  ; #2氦检阀打开延时
T0383 BOOL  ; 氦检持续时间
T0384 BOOL  ; #2氦检阀打开抽气阀关闭延时
T0385 BOOL  ; #2腔体数据传输延时
T0386 BOOL  ; 测试结束后抽残气延时
T0387 BOOL  ; 抽残气时间
T0388 BOOL  ; #2腔体破真空延时
T0389 BOOL  ; #2腔体破真空值到达
T0390 BOOL  ; #2腔氦检阀关闭延时
T0400 BOOL  ; 出料机械手回左OK位置延时
T0401 BOOL  ; 出料机械手回右OK位置延时
T0402 BOOL  ; 出料机械手回NG位置延时
T0403 BOOL  ; 出料机械手回#1腔体位置延时
T0404 BOOL  ; 出料机械手回#2腔体位置延时
T0407 BOOL  ; 下料机械手Alarm_Clr输出时间
T0410 BOOL  ; 出料机械手位置异常信息持续时间
T0411 BOOL  ; 下料旋转气缸位置异常信息持续时间
T0412 BOOL  ; 下料缓存有料异常信息持续时间
T0413 BOOL  ; #1合模气缸不在缩回位异常信息持续时间
T0414 BOOL  ; #2合模气缸不在缩回位异常信息持续时间
T0415 BOOL  ; 出料夹爪不在张开位异常信息持续时间
T0416 BOOL  ; 出料提升气缸不在伸出位异常信息持续时间
T0417 BOOL  ; 出料提升气缸不在缩回位异常信息持续时间
T0418 BOOL  ; 出料机械手没归零异常信息持续时间
T0419 BOOL  ; 出料机械手到达左极限异常信息持续时间
T0420 BOOL  ; 出料机械手到达右极限异常信息持续时间
T0421 BOOL  ; 进料机械手位置避让异常信息持续时间
T0422 BOOL  ; 进料机械手位置避让异常信息持续时间
T0425 BOOL  ; 出料机械手报警信号持续时间
T0426 BOOL  ; 出料爪1打开延时
T0427 BOOL  ; 出料爪2打开延时
T0430 BOOL  ; 出料机械手回#1腔体位置延时
T0431 BOOL  ; 出料机械手回#2腔体位置延时
T0432 BOOL  ; 出料机械手回OK位置延时
T0433 BOOL  ; 爪2-OK延时
T0434 BOOL  ; 出料机械手回NG位置延时
T0440 BOOL  ; （0.06）出料起始位有料感应异常延时
T0441 BOOL  ; （10.05）出料拉带运行异常延时
T0442 BOOL  ; （0.07）出料拉带末端感应异常延时
T0469 BOOL  ; $?St$Bk?_#[1179] / 上料伺服Alarm_Clr输出延时 / $?St$Bk?_#[1179]
T0501 BOOL  ; （龙门）左右机械手手动#1位置延时
T0502 BOOL  ; （龙门）左右机械手手动#2位置延时
T0503 BOOL  ; （龙门）左右机械手手动#3位置延时
T0504 BOOL  ; （龙门）左右机械手手动#4位置延时
T0505 BOOL  ; （龙门）左右机械手手动#5位置延时
T0506 BOOL  ; （龙门）左右机械手手动#6位置延时
T0507 BOOL  ; （龙门）左右机械手手动#7位置延时
T0508 BOOL  ; （龙门）左右机械手手动#8位置延时
T0509 BOOL  ; （龙门）左右机械手手动#9位置延时
T0510 BOOL  ; （龙门）左右机械手手动#10位置延时
T0511 BOOL  ; （龙门）左右机械手手动#11位置延时
T0512 BOOL  ; （龙门）左右机械手手动#12位置延时
T0513 BOOL  ; 取料点位延时
T0514 BOOL  ; 左右自动速度
T0520 BOOL  ; 到取料料位置延时
T0521 BOOL  ; （龙门）左右机械手手动#13位置延时
T0522 BOOL  ; （龙门）左右机械手手动#14位置延时
T0523 BOOL  ; （龙门）左右机械手手动#15位置延时
T0524 BOOL  ; （龙门）左右机械手手动#16位置延时
T0525 BOOL  ; （龙门）左右机械手手动#17位置延时
T0526 BOOL  ; （龙门）左右机械手手动#18位置延时
T0527 BOOL  ; （龙门）左右机械手手动#19位置延时
T0528 BOOL  ; （龙门）左右机械手手动#20位置延时
T0529 BOOL  ; （龙门）左右机械手手动#21位置延时
T0530 BOOL  ; （龙门）左右机械手手动#22位置延时
T0531 BOOL  ; （龙门）左右机械手手动#23位置延时
T0532 BOOL  ; （龙门）左右机械手手动#24位置延时
T0533 BOOL  ; 前后伺服正转脉冲
T0534 BOOL  ; 前后伺服反转脉冲
T0535 BOOL  ; 到#1排放料位置延时
T0536 BOOL  ; 到#2排放料位置延时
T0537 BOOL  ; 入盘爪打开延时
T0538 BOOL  ; 延时复位伺服
T0565 BOOL  ; 空跑延时
T0566 BOOL  ; 输送带有料感应延时
T0567 BOOL  ; 输送带无料感应延时
T0568 BOOL  ; 有料延时上升
T0569 BOOL  ; 去放料延时
T0570 BOOL  ; 延时松夹
T0571 BOOL  ; 入盘机械手延时上升
T0572 BOOL  ; 出料带电池取走持续时间
T0573 BOOL  ; 输送带没料持续时间
T0574 BOOL  ; 入盘延时复位
T0575 BOOL  ; 延时复位W66.10
T0576 BOOL  ; 出料带末端有料持续时间
T0577 BOOL  ; 出料末端料已取走持续时间
T0600 BOOL  ; 龙门升降机械手Alarm_Clr输出时间
T0601 BOOL  ; 龙门左右机械手Alarm_Clr输出时间
T0602 BOOL  ; 龙门前后机械手Alarm_Clr输出时间
T0603 BOOL  ; 抓料机械手手动到取料位
T0650 BOOL  ; 入盘机械手左右伺服没归零延时报警
T0651 BOOL  ; 入盘机械手前后伺服没归零延时报警
T0652 BOOL  ; 入盘机械手升降伺服没归零延时报警
T0653 BOOL  ; 入盘升降气缸只能在取料位升降延时
T0654 BOOL  ; 入盘夹爪气缸张开异常延时
T0655 BOOL  ; 入盘升降只能在入电池位下降
T0656 BOOL  ; 入盘放料时夹爪气缸张开异常延时
T0657 BOOL  ; 在取料位才能下降取料异常延时
T0661 BOOL  ; #1有空托盘感应异常延时
T0662 BOOL  ; #2有空托盘感应异常延时
T0663 BOOL  ; 空托盘到位感应或拉带异常延时
T0664 BOOL  ; #3空托盘感应或拉带异常延时
T0665 BOOL  ; 空托盘到位感应、#3空托盘感应或拉带异常延时
T0666 BOOL  ; 空托盘到位感应异常延时
T0667 BOOL  ; 空盘升降机架上有空托盘记忆异常延时
T0668 BOOL  ; （7.05）上空托盘位感应异常延时
T0669 BOOL  ; （7.14）下满料托盘感应1异常延时
T0670 BOOL  ; （7.04）下满料托盘到位感应#2异常延时
T0671 BOOL  ; （13.08）电池入盘位有托盘感应异常延时
T0672 BOOL  ; （7.03）缓存#1托盘到位感应异常延时
T0673 BOOL  ; （7.04）缓存#2托盘到位感应异常延时
T0701 BOOL  ; 料盘上升
T0702 BOOL  ; 料盘下降
T0703 BOOL  ; （龙门）料盘机到上料延时
T0704 BOOL  ; （龙门）料盘机到放料位置延时
T0710 BOOL  ; 料盘Alarm_Clr输出时间
T0711 BOOL  ; 刹车释放延时
T0720 BOOL  ; #1无料盒感应延时下降
T0721 BOOL  ; #2无料盒感应延时下降
T0722 BOOL  ; 下顶升气缸延时缩回
T0728 BOOL  ; 料盒定位气缸缩回延时
T0729 BOOL  ; 缓存电机延时停止
T0730 BOOL  ; 延时停下料电机
T0732 BOOL  ; 料盒定位气缸延时
T0733 BOOL  ; 缓存2有料顶升延时
T0734 BOOL  ; 缓存2有料延时
T0735 BOOL  ; 顶升气缸延时下降
T0736 BOOL  ; 顶升#2无料延时下
T0737 BOOL  ; 顶升#1无料延时下
T0738 BOOL  ; 料盒到位延时
T0750 BOOL  ; 料盒升降伺服没归零延时
T0751 BOOL  ; 有料盒脱离气缸没伸出不能上升延时
T0752 BOOL  ; 有料盒定位气缸没缩回不能上升延时
T0753 BOOL  ; 下面有料盒感应异常不下行延时
T0754 BOOL  ; 有料盒时定位气缸没缩回不能下降延时
T0800 BOOL  ; 腔体1有料感应延时
T0801 BOOL  ; 腔体1无料感应延时
T0802 BOOL  ; 上料柔性报警延时
T0803 BOOL  ; 下料柔性报警延时
T0804 BOOL  ; 入盘升降柔性报警
T0805 BOOL  ; 料盒#1电池有料屏蔽
T0806 BOOL  ; 料盒#2电池有料屏蔽
T0807 BOOL  ; 料盒#3电池有料信号屏蔽
T0808 BOOL  ; 料盒#4电池有料信号屏蔽
T0809 BOOL  ; 气源压力信号屏蔽
T0810 BOOL  ; 料盒#6电池屏蔽信号
T0811 BOOL  ; 进料缓存有料信号延时
T0812 BOOL  ; 出料缓存有料信号屏蔽
T0813 BOOL  ; 腔体有料信号
T0814 BOOL  ; 料盒#9电池有料信号屏蔽
T0815 BOOL  ; 料盒#10电池有料信号屏蔽
T0816 BOOL  ; 进料横移气缸缩回位延时
T0817 BOOL  ; 进料横移气缸伸出位延时
T0818 BOOL  ; 料盒#13电池有料信号屏蔽
T0819 BOOL  ; 料盒#14电池有料屏蔽
T0820 BOOL  ; 进料升降气缸缩回位时间
T0821 BOOL  ; 料盒#16电池有料信号屏蔽
T0822 BOOL  ; 进料夹爪1张开位延时
T0823 BOOL  ; 料盒#18电池有料信号屏蔽
T0824 BOOL  ; 进料夹爪2张开位延时
T0825 BOOL  ; 料盒#20电池有料信号屏蔽
T0826 BOOL  ; 进料移栽气缸缩回位时间
T0827 BOOL  ; 料盒#22电池有料信号屏蔽
T0828 BOOL  ; 上料夹爪1张开位时间
T0829 BOOL  ; 上料夹爪1夹紧位延时
T0830 BOOL  ; NG无料感应延时
T0831 BOOL  ; NG有料感应延时
T0832 BOOL  ; 腔体2无料感应延时
T0833 BOOL  ; 腔体2有料感应延时
T0900 BOOL  ; 扫码阻挡气缸缩回报警
T0901 BOOL  ; 扫码阻挡气缸伸出报警
T0902 BOOL  ; 抓料阻挡气缸缩回报警
T0903 BOOL  ; 抓料阻挡气缸伸出报警
T0904 BOOL  ; 扫码NG拨料气缸缩回位延时报警
T0905 BOOL  ; 扫码NG拨料气缸伸出报警
T0906 BOOL  ; 上料提升气缸缩回报警
T0907 BOOL  ; 上料提升气缸伸出报警
T0908 BOOL  ; 上料左夹爪升降气缸缩回报警
T0909 BOOL  ; 上料左夹爪升降气缸伸出报警
T0910 BOOL  ; 上料右夹爪升降气缸缩回报警
T0911 BOOL  ; 上料右夹爪升降气缸伸出报警
T0912 BOOL  ; 上料左夹爪张开位报警
T0913 BOOL  ; 上料左夹爪夹紧报警
T0914 BOOL  ; 上料夹爪2张开报警
T0915 BOOL  ; 上料夹爪2夹紧报警
T0916 BOOL  ; 下料提升气缸缩回报警
T0917 BOOL  ; 下料提升气缸伸出位延时报警
T0918 BOOL  ; 下料夹爪升降气缸缩回报警
T0919 BOOL  ; 下料夹爪升降气缸伸出报警
T0920 BOOL  ; 下料夹爪1张开报警
T0921 BOOL  ; 下料夹爪夹1紧报警
T0922 BOOL  ; 下料夹爪2张开位延时报警
T0923 BOOL  ; 下料夹爪2夹紧位延时报警
T0924 BOOL  ; 合模气缸1缩回延时报警
T0925 BOOL  ; #1合模气缸伸出位延时报警
T0926 BOOL  ; #2合模气缸缩回位延时报警
T0927 BOOL  ; #2合模气缸伸出位延时#2合模气缸伸出位延时报警
T0928 BOOL  ; 出料NG拨料气缸伸出位延时报警
T0929 BOOL  ; 出料NG拨料气缸缩回位延时报警
T0930 BOOL  ; 料盒定位气缸缩回位延时报警
T0931 BOOL  ; 料盒定位气缸伸出位延时报警
T0932 BOOL  ; 料盒上阻挡气缸缩回位延时报警
T0933 BOOL  ; 料盒上阻挡气缸伸出位延时报警
T0934 BOOL  ; 备份
T0935 BOOL  ; 备份
T0936 BOOL  ; #1上顶升左气缸缩回位延时报警
T0937 BOOL  ; #1上顶升左气缸伸出位延时报警
T0938 BOOL  ; #1上顶升右气缸缩回位延时报警
T0939 BOOL  ; #1上顶升右气缸伸出位延时报警
T0940 BOOL  ; #2上顶升左气缸缩回位延时报警
T0941 BOOL  ; #2上顶升左气缸伸出位延时
T0942 BOOL  ; #2上顶升右气缸缩回位延时报警
T0943 BOOL  ; #2上顶升右气缸伸出位延时报警
T0944 BOOL  ; #1下顶升左气缸缩回位延时报警
T0945 BOOL  ; #1下顶升左气缸伸出位延时报警
T0946 BOOL  ; #1下料顶升右气缸缩回位延时报警
T0947 BOOL  ; #1下顶升右气缸伸出位延时报警
T0948 BOOL  ; #2下顶升左气缸缩回位延时报警
T0949 BOOL  ; #2下顶升左气缸伸出位延时报警
T0950 BOOL  ; #2下料顶升右气缸缩回位延时报警
T0951 BOOL  ; #2下顶升右气缸伸出位延时报警
T0952 BOOL  ; 龙门左拉带脱离气缸缩回位延时
T0953 BOOL  ; 龙门左拉带脱离气缸伸出位
T0954 BOOL  ; 龙门右拉带脱离气缸缩回位延时
T0955 BOOL  ; 入盘右拉带脱离气缸伸出位延时
T0956 BOOL  ; 入盘升降气缸缩回位延时
T0957 BOOL  ; 入盘升降气缸伸出位延时
T0958 BOOL  ; 入盘夹爪气缸松开延时报警
T0959 BOOL  ; 龙门夹爪气缸夹紧延时报警
T0960 BOOL  ; 入盘扫码后判断
T0961 BOOL  ; 托盘重新扫码持续时间
T0962 BOOL  ; 托盘更新确认持续时间
T1099 BOOL  ; 出料夹爪2夹紧报警
T1287 BOOL  ; 料盘自动上
T1288 BOOL  ; 自动下
W0.00 BOOL  ; 自动状态-HMI
W0.01 BOOL  ; 启动按钮-HMI
W0.03 BOOL  ; 自动状态
W0.04 BOOL  ; 强制清零
W0.05 BOOL  ; 整机复位
W0.06 BOOL  ; 上料夹爪复位-HMI
W0.07 BOOL  ; 托盘重新扫码-HMI
W0.08 BOOL  ; 托盘更换确认-HMI
W0.09 BOOL  ; #1腔体复位-HMI
W0.10 BOOL  ; #2腔体复位-HMI
W0.11 BOOL  ; 出料机械手复位-HMI
W0.12 BOOL  ; 入盘机构复位
W0.13 BOOL  ; 出料夹爪复位-HMI
W0.14 BOOL  ; 复位按钮-HMI
W0.15 BOOL  ; 报警返回-HMI
W1 CHANNEL  ; 上料手动按钮-HMI
W10 CHANNEL  ; 上料手动气缸寄存器复位
W104.06 BOOL  ; 料盘定位气缸打开 HIM
W107.00 BOOL  ; 入盘（前后）Y轴取料位置
W107.01 BOOL  ; 入盘（前后）Y轴#1排位置
W107.02 BOOL  ; 入盘（前后）Y轴#2排位置
W107.03 BOOL  ; 料盘机到入电池位置
W107.04 BOOL  ; 料盘机上空料盒位置
W107.05 BOOL  ; 入盘（升降）Z轴取料位置
W107.06 BOOL  ; 入盘（升降）Z轴放料位置
W107.07 BOOL  ; 入盘（左右）X轴#1号点位置ok
W107.08 BOOL  ; 入盘（左右）X轴#2号点位置OK
W107.09 BOOL  ; 入盘（左右）X轴#3号点位置OK
W107.10 BOOL  ; 入盘（左右）X轴#4号点位置OK
W107.11 BOOL  ; 入盘（左右）X轴#5号点位置OK
W107.12 BOOL  ; 入盘（左右）X轴#6号点位置OK
W107.13 BOOL  ; 入盘（左右）X轴#7号点位置OK
W107.14 BOOL  ; 入盘（左右）X轴#8号点位置OK
W107.15 BOOL  ; 入盘（左右）X轴#9号点位置OK
W108.00 BOOL  ; 入盘（左右）X轴#10号点位置OK
W108.01 BOOL  ; 入盘（左右）X轴#11号点位置OK
W108.02 BOOL  ; 入盘（左右）X轴#12号点位置OK
W108.03 BOOL  ; 入盘（左右）X轴#13号点位置OK
W108.04 BOOL  ; 入盘（左右）X轴#14号点位置OK
W108.05 BOOL  ; 入盘（左右）X轴#15号点位置OK
W108.06 BOOL  ; 入盘（左右）X轴#16号点位置OK
W108.07 BOOL  ; 入盘（左右）X轴#17号点位置OK
W108.08 BOOL  ; 入盘（左右）X轴#18号点位置OK
W108.09 BOOL  ; 入盘（左右）X轴#19号点位置OK
W108.10 BOOL  ; 入盘（左右）X轴#20号点位置OK
W108.11 BOOL  ; 入盘（左右）X轴#21号点位置OK
W108.12 BOOL  ; 入盘（左右）X轴#22号点位置OK
W108.13 BOOL  ; 入盘（左右）X轴#23号点位置OK
W108.14 BOOL  ; 入盘（左右）X轴#24号点位置OK
W108.15 BOOL  ; 入盘（左右）X轴左右取料位
W109.00 BOOL  ; 入盘（左右）X轴前后左右到去料点位置
W10.00 BOOL  ; 机械手手动停止距离
W10.01 BOOL  ; 上料机械手到#1腔体安全条件
W10.02 BOOL  ; 上料机械手回#2腔体安全条件
W10.03 BOOL  ; 进料机械手回NG位时出料机械手条件
W10.04 BOOL  ; 出料机械手回#1腔体时进料机械手条件
W10.05 BOOL  ; 出料机械手回#2腔体时进料机械手条件
W10.06 BOOL  ; 手动可行走
W10.09 BOOL  ; 进料旋转手动归零
W10.10 BOOL  ; 进料旋转手动左转
W10.11 BOOL  ; 进料旋转手动右转
W10.12 BOOL  ; 进料手动旋转到#1待料角度
W10.13 BOOL  ; 进料手动旋转到#2待料角度
W10.14 BOOL  ; 进料手动旋转到进料角度
W11 CHANNEL  ; 下料手动气缸寄存器复位
W114.01 BOOL  ; 入盘机械手取料位
W11.09 BOOL  ; 上料机械手手动归零
W11.10 BOOL  ; 上料机械手手动左移
W11.11 BOOL  ; 上料机械手手动右移
W11.12 BOOL  ; 上料机械手手动左上料位
W11.13 BOOL  ; 上料机械手手动右上料位
W11.14 BOOL  ; 上料机械手手动#1腔体
W12 CHANNEL  ; 腔体手动寄存器复位1
W12.00 BOOL  ; 真空泵手动打开
W13 CHANNEL  ; 腔体手动寄存器复位2
W14 CHANNEL  ; 腔体手动寄存器复位3
W140.00 BOOL  ; 取料点位
W15 CHANNEL  ; 上料机械手手动寄存器复位
W151.06 BOOL  ; 入盘夹爪松开
W15.00 BOOL  ; 空跑程序-抓料
W15.01 BOOL  ; 重新扫码按钮(T)(A)
W15.02 BOOL  ; 电池扫码完成
W15.03 BOOL  ; 扫码失败
W15.04 BOOL  ; 扫码OK
W15.05 BOOL  ; 隔离阻挡气缸输出
W16 CHANNEL  ; 下料机械手手动寄存器复位
W166.10 BOOL  ; 上阻挡气缸
W16.08 BOOL  ; 下料NG手动拔料
W170.08 BOOL  ; .
W18.00 BOOL  ; 上料爪1打开
W18.01 BOOL  ; 上料爪2打开
W18.02 BOOL  ; 出料爪1打开
W18.03 BOOL  ; 出料爪2打开
W18.04 BOOL  ; 入盘夹爪打开-HMI
W19.00 BOOL  ; 门磁条件
W19.01 BOOL  ; PC系统条件
W19.02 BOOL  ; 自动状态不能进手动操作
W19.03 BOOL  ; 上料机构气缸状态
W19.04 BOOL  ; 出料机构气缸状态条件
W19.06 BOOL  ; 复位
W19.07 BOOL  ; 初始或复位后启动条件
W19.08 BOOL  ; 初始或复位后状态
W19.09 BOOL  ; 设备启动条件
W19.10 BOOL  ; 启动状态
W19.11 BOOL  ; 腔体真空泵启动
W19.13 BOOL  ; 手动转自动状态
W19.14 BOOL  ; 氦检仪启动条件
W19.15 BOOL  ; 氦检仪启动
W1.00 BOOL  ; 停止按钮-HMI
W1.01 BOOL  ; 启动按钮-HMI
W1.02 BOOL  ; 复位按钮-HMI
W1.03 BOOL  ; 清料按钮-HMI
W1.08 BOOL  ; HMI-蜂鸣器屏蔽
W2 CHANNEL  ; 下料手动按钮-HMI
W200.00 BOOL  ; 调试
W200.15 BOOL  ; 调试
W20.00 BOOL  ; 手动阻挡气缸
W20.01 BOOL  ; 手动阻挡气缸（抓料位）
W20.02 BOOL  ; 手动扫描-HMI
W20.05 BOOL  ; 扫码位阻挡气缸手动输出
W20.06 BOOL  ; 抓料位阻挡气缸手动输出
W20.09 BOOL  ; 电池扫码信号
W20.10 BOOL  ; 扫码阻挡气缸缩回
W20.11 BOOL  ; 电池已到抓紧料位
W20.12 BOOL  ; 抓紧料位阻挡气缸缩回
W21 CHANNEL  ; 上料机构寄存器
W21.00 BOOL  ; 机械手归零-HMI
W21.01 BOOL  ; 上料机械手左移按钮-HMI
W21.02 BOOL  ; 上料机械手机械手右移按钮-HMI
W21.03 BOOL  ; 上料左取料位-HMI
W21.04 BOOL  ; 上料右取料位-HMI
W21.05 BOOL  ; 腔体1位置-HMI
W21.06 BOOL  ; 腔体2位置-HMI
W21.07 BOOL  ; 左NG位
W21.08 BOOL  ; 右NG位
W21.09 BOOL  ; 进料提升气缸-HMI
W21.10 BOOL  ; 左爪升降
W21.11 BOOL  ; 右爪升降
W21.12 BOOL  ; #1进料夹爪-HMI
W21.13 BOOL  ; #2进料夹爪-HMI
W21.14 BOOL  ; NG手动拔料
W22 CHANNEL  ; 进料机械手寄存器
W23 CHANNEL  ; 上料机械手动作
W23.00 BOOL  ; 上料提升气缸伸出条件
W23.01 BOOL  ; 手动复位
W23.02 BOOL  ; 上料复位
W23.03 BOOL  ; 进料机械手回左取料位置
W23.04 BOOL  ; 进料机械手归回右取料位置
W23.05 BOOL  ; 上料提升气缸伸出
W23.06 BOOL  ; 升降1下
W23.07 BOOL  ; 上料夹爪2下
W23.08 BOOL  ; 进料机械手回#1腔体
W23.09 BOOL  ; 进料机械手回#2腔体
W23.10 BOOL  ; 上料提升气缸伸出
W23.11 BOOL  ; 上料夹爪松开
W23.12 BOOL  ; 进料提升气缸缩回
W24 CHANNEL  ; #4腔体状态1
W24.01 BOOL  ; 放左NG料
W24.02 BOOL  ; 放右NG料
W24.03 BOOL  ; 放NG缩回
W24.04 BOOL  ; 自动拔NG料
W24.05 BOOL  ; 清料了不去右取料
W24.06 BOOL  ; 自动扫码NG拨料缩回
W24.07 BOOL  ; 扫码NG拨料完成
W25.00 BOOL  ; 上料机械手手动归零
W25.01 BOOL  ; 上料机械手手动左移
W25.02 BOOL  ; 上料机械手手动右移
W25.03 BOOL  ; 上料机械手手动到上料左取料位
W25.04 BOOL  ; 手动到上料右取料位
W25.05 BOOL  ; 进料机械手手动到腔体1位置
W25.06 BOOL  ; 进料机械手手动到腔体2位置
W25.07 BOOL  ; 上料机械手手动回左NG位置
W25.08 BOOL  ; 上料机械手手动回右NG位置
W25.09 BOOL  ; 上料提升气缸手动伸出
W25.10 BOOL  ; 上料左爪升降手动伸出
W25.11 BOOL  ; 上料右爪升降手动伸出
W25.14 BOOL  ; NG手动拔料
W28.00 BOOL  ; #1合模气缸不在缩回位
W28.01 BOOL  ; 上料夹爪有料腔体有料不能下降
W28.02 BOOL  ; #2合模气缸不在缩回位
W28.03 BOOL  ; 进料夹爪不在张开位
W28.04 BOOL  ; 进料提升气缸不在缩回位
W28.05 BOOL  ; 进料机械手没归零
W28.06 BOOL  ; 进料机械手到达左极限
W28.07 BOOL  ; 进料机械手到达右极限
W28.08 BOOL  ; 出料机械手避让位置异常
W28.09 BOOL  ; 出料机械手避让位置异常
W28.10 BOOL  ; 上料提升气缸要先下到位才能操作
W29.00 BOOL  ; 上料机械手有报警输出
W3 CHANNEL  ; 腔体按钮-HMI
W303.00 BOOL  ; 异常
W303.01 BOOL  ; 设备暂停
W30.00 BOOL  ; #1合模气缸-HMI
W30.01 BOOL  ; #1抽气阀-HMI
W30.02 BOOL  ; #1氦检阀-HMI
W30.03 BOOL  ; #1破真空阀-HMI
W30.04 BOOL  ; #1吹气阀-HMI
W30.05 BOOL  ; #1腔体自检-HMI
W30.08 BOOL  ; #2合模气缸-HMI
W30.09 BOOL  ; #2抽气阀-HMI
W30.10 BOOL  ; #2氦检阀-HMI
W30.11 BOOL  ; #2破真空阀-HMI
W30.12 BOOL  ; #2吹气阀-HMI
W30.13 BOOL  ; #2腔体自检-HMI
W311.00 BOOL  ; 异常报警
W31.00 BOOL  ; #1合模气缸手动伸出
W31.01 BOOL  ; #1抽气阀手动打开
W31.02 BOOL  ; #1氦检阀手动打开
W31.03 BOOL  ; #1破真空阀手动打开
W31.04 BOOL  ; #1吹气阀手动打开
W31.06 BOOL  ; #1合模气缸手动缩回
W31.08 BOOL  ; #2合模气缸手动伸出
W31.09 BOOL  ; #2抽气阀手动打开
W31.10 BOOL  ; #2氦检阀手动打开
W31.11 BOOL  ; #2破真空阀手动打开
W31.12 BOOL  ; #2吹气阀手动打开
W31.14 BOOL  ; #2合模气缸手动缩回
W32.00 BOOL  ; 腔体1合模条件
W32.01 BOOL  ; #1腔体自检条件
W32.02 BOOL  ; #1腔体自检中
W32.03 BOOL  ; #1合模气缸自检伸出
W32.04 BOOL  ; #1抽气阀自检输出
W32.05 BOOL  ; #1腔体自检进入保压前状态
W32.06 BOOL  ; #1腔体自检进入保压状态
W32.07 BOOL  ; #1腔体保压结束
W32.08 BOOL  ; #1腔体自检破真空阀打开
W32.09 BOOL  ; #1腔体自检破真空结束
W32.10 BOOL  ; #1合模气缸缩回
W32.11 BOOL  ; #1腔体自检吹气阀打开
W32.12 BOOL  ; #1腔体自检结束
W33.00 BOOL  ; 合模气缸1伸出条件
W33.01 BOOL  ; 合模气缸1伸出
W33.02 BOOL  ; #1抽气阀打开
W33.03 BOOL  ; #1抽气结束
W33.04 BOOL  ; #1抽气阀关闭
W33.05 BOOL  ; #1氦检阀打开
W33.06 BOOL  ; #1氦检正常结束
W33.07 BOOL  ; #1抽气异常结束
W33.08 BOOL  ; #1抽气阀打开(抽残气)
W33.09 BOOL  ; #1抽残气结束
W33.10 BOOL  ; #1腔体破真空阀打开
W33.11 BOOL  ; #1腔体破真空结束
W33.12 BOOL  ; #1腔体吹气阀打开
W33.13 BOOL  ; #1合模气缸缩回
W34.00 BOOL  ; 腔体2合模条件
W34.01 BOOL  ; #2腔体自检条件
W34.02 BOOL  ; #2腔体自检中
W34.03 BOOL  ; #2合模气缸自检伸出
W34.04 BOOL  ; #2抽气阀自检输出
W34.05 BOOL  ; #2腔体自检进入保压前状体
W34.06 BOOL  ; #2腔体自检进入保压状态
W34.07 BOOL  ; #2腔体保压结束
W34.08 BOOL  ; #2腔体自检破真空阀打开
W34.09 BOOL  ; #2腔体自检破真空结束
W34.10 BOOL  ; #2合模气缸缩回
W34.11 BOOL  ; #2腔体自检吹气阀打开
W34.12 BOOL  ; #2腔体自检结束
W35.00 BOOL  ; 合模气缸2伸出条件
W35.01 BOOL  ; 合模气缸2伸出
W35.02 BOOL  ; #2抽气阀打开
W35.03 BOOL  ; #2抽气结束
W35.04 BOOL  ; #2抽气阀关闭
W35.05 BOOL  ; #2氦检阀打开
W35.06 BOOL  ; #2氦检正常结束
W35.07 BOOL  ; #2抽气异常结束
W35.08 BOOL  ; #2抽气阀打开(抽残气)
W35.09 BOOL  ; #2抽残气结束
W35.10 BOOL  ; #2腔体破真空阀打开
W35.11 BOOL  ; #2腔体破真空结束
W35.12 BOOL  ; #2腔体吹气阀打开
W35.13 BOOL  ; #2合模气缸缩回
W38.00 BOOL  ; 产品测试NG后蜂鸣器报警
W38.01 BOOL  ; 进料机械手要复位
W38.02 BOOL  ; 出料机械手要复位
W38.03 BOOL  ; #1腔体真空值大于破真空设定值异常
W38.04 BOOL  ; #1抽气阀打开异常
W38.05 BOOL  ; #1氦检阀打开异常
W38.06 BOOL  ; #1破真空阀打开异常
W38.07 BOOL  ; #1吹气阀打开异常
W38.08 BOOL  ; 上料机械手要复位
W38.09 BOOL  ; 出料机械手要复位
W38.10 BOOL  ; #2腔体真空值大于破真空设定值异常
W38.11 BOOL  ; #2抽气阀打开异常
W38.12 BOOL  ; #2氦检阀打开异常
W38.13 BOOL  ; #2破真空阀打开异常
W38.14 BOOL  ; #2吹气阀打开异常
W39.00 BOOL  ; 腔体有报警输出
W39.01 BOOL  ; 下料机械手在原点位
W4 CHANNEL  ; 上料机械手按钮-HMI
W400.00 BOOL  ; 料盘上
W400.01 BOOL  ; 料盘上方向
W400.02 BOOL  ; 料盘上
W400.03 BOOL  ; 料盘下方向
W400.04 BOOL  ; 前后伺服正转脉冲
W400.05 BOOL  ; 前后伺服正转方向
W400.06 BOOL  ; 前后伺服反转脉冲
W400.07 BOOL  ; 前后伺服反转方向
W40.00 BOOL  ; 机械手归零-HMI
W40.01 BOOL  ; 下料机械手左移按钮-HMI
W40.02 BOOL  ; 下料机械手右移按钮-HMI
W40.03 BOOL  ; 左OK下料位置-HMI
W40.04 BOOL  ; 右OK下料位置-HMI
W40.05 BOOL  ; NG下料位置-HMI
W40.06 BOOL  ; 腔体1位置-HMI
W40.07 BOOL  ; 腔体2位置-HMI
W40.08 BOOL  ; 出料输送带手动
W40.10 BOOL  ; 出料提升气缸-HMI
W40.11 BOOL  ; 出料升降气缸手动
W40.12 BOOL  ; #1出料夹爪-HMI
W40.13 BOOL  ; #2出料夹爪-HMI
W40.14 BOOL  ; 下料NG拔料
W42.00 BOOL  ; 出料提升气缸伸出条件
W42.01 BOOL  ; 左下料夹爪松开条件
W42.02 BOOL  ; 右下料夹爪松开条件
W43.01 BOOL  ; 腔体位出料提升缩回条件
W44.00 BOOL  ; 出料机械手回#1腔体位置
W44.01 BOOL  ; 出料机械手回#2腔体位置
W44.02 BOOL  ; 下料提升气缸伸出
W44.03 BOOL  ; 下料夹爪升降气缸伸出
W44.04 BOOL  ; 出料机械手回放爪1位置
W44.05 BOOL  ; 出料机械手回放爪2位置
W44.06 BOOL  ; 出料机械手回NG位置
W44.07 BOOL  ; 出料提升气缸伸出
W44.08 BOOL  ; 下料机械手放料完成
W44.09 BOOL  ; 出料NG拨料气缸输出
W44.10 BOOL  ; 出料自动运行
W44.11 BOOL  ; 出料自动停止
W44.12 BOOL  ; 强制清零电机运3秒
W44.13 BOOL  ; 下夹2无料
W44.14 BOOL  ; NG拨料气缸缩回
W44.15 BOOL  ; NG拨料完成
W450 CHANNEL  ; PLC交互
W450.00 BOOL  ; MES进站调用->PC
W450.01 BOOL  ; #1腔体放料->PC
W450.02 BOOL  ; #2腔体放料->PC
W450.03 BOOL  ; MES开启->PC
W450.04 BOOL  ; MES显示清除->PC
W450.09 BOOL  ; #1,#2条码OK
W450.10 BOOL  ; 条码OK
W450.11 BOOL  ; #1下料夹爪有料
W450.12 BOOL  ; #2下料夹爪有料
W450.14 BOOL  ; #3下料夹爪有料
W450.15 BOOL  ; #4下料夹爪有料
W45.00 BOOL  ; 出料机械手手动归零
W45.01 BOOL  ; 出料机械手手动左移
W45.02 BOOL  ; 出料机械手手动右移
W45.03 BOOL  ; 手动到左OK位置
W45.04 BOOL  ; 手动到右OK位置
W45.05 BOOL  ; 出料机械手手动到NG下料位
W45.06 BOOL  ; 出料机械手手动到腔体1位置
W45.07 BOOL  ; 出料机械手手动到腔体2位置
W45.10 BOOL  ; 下料提升气缸手动伸出
W45.11 BOOL  ; 出料升降手动
W45.14 BOOL  ; NG拨料气缸手动输出
W45.15 BOOL  ; 出料输送带手动
W47.01 BOOL  ; 去腔1
W47.02 BOOL  ; 到腔体步
W47.03 BOOL  ; 夹爪抓料步
W47.04 BOOL  ; 下料夹爪缩回d步
W47.05 BOOL  ; 去腔2
W47.08 BOOL  ; 出料提升气缸伸出放料步
W47.09 BOOL  ; 出料夹爪松开
W47.10 BOOL  ; 放料完成步
W49.00 BOOL  ; 下料机械有报警输出
W4.00 BOOL  ; 报警清除
W4.04 BOOL  ; 强制清零
W5 CHANNEL  ; 下料机械手按钮-HMI
W500.00 BOOL  ; #1号电池可放料
W500.01 BOOL  ; #2号电池可放料
W500.02 BOOL  ; #3号电池可放料
W500.03 BOOL  ; #4号电池可放料
W500.04 BOOL  ; #5号电池可放料
W500.05 BOOL  ; #6号电池可放料
W500.06 BOOL  ; #7号电池可放料
W500.07 BOOL  ; #8号电池可放料
W500.08 BOOL  ; #9号电池可放料
W500.09 BOOL  ; #10号电池可放料
W500.10 BOOL  ; #11号电池可放料
W500.11 BOOL  ; #12号电池可放料
W500.12 BOOL  ; #13号电池可放料
W500.13 BOOL  ; #14号电池可放料
W500.14 BOOL  ; #15号电池可放料
W500.15 BOOL  ; #16号电池可放料
W501.00 BOOL  ; #17号电池可放料
W501.01 BOOL  ; #18号电池可放料
W501.02 BOOL  ; #19号电池可放料
W501.03 BOOL  ; #20号电池可放料
W501.04 BOOL  ; #21号电池可放料
W501.05 BOOL  ; #22号电池可放料
W501.06 BOOL  ; #23号电池可放料
W501.07 BOOL  ; #24号电池可放料
W502.02 BOOL  ; 第二排料
W50.00 BOOL  ; 入盘（升降）X轴手动归零
W50.01 BOOL  ; 入盘（左右）X轴手动左移
W50.02 BOOL  ; 入盘（左右）X轴手动右移
W50.10 BOOL  ; （龙门）前后机械手回原
W50.11 BOOL  ; 入盘前进机械手前进
W50.12 BOOL  ; (龙门）前进机械手后退
W51.00 BOOL  ; 入盘机械手取料位
W51.01 BOOL  ; 入盘（左右）X轴手动#1位置
W51.02 BOOL  ; 入盘（左右）X轴手动#2位置
W51.03 BOOL  ; 入盘（左右）X轴手动#7位置
W51.04 BOOL  ; 入盘（左右）X轴手动#4位置
W51.05 BOOL  ; 入盘（左右）X轴手动#4位置
W51.06 BOOL  ; 入盘（左右）X轴手动#6位置
W51.07 BOOL  ; 入盘（左右）X轴手动#7位置
W51.08 BOOL  ; 入盘（左右）X轴手动#8位置
W51.09 BOOL  ; 入盘（左右）X轴手动#9位置
W51.10 BOOL  ; 入盘（左右）X轴手动#10位置
W51.11 BOOL  ; 入盘（左右）X轴手动#11位置
W51.12 BOOL  ; 入盘（左右）X轴手动#12位置
W51.13 BOOL  ; 入盘Y轴到#1排放料位置  HIM
W51.14 BOOL  ; 到#2排 放料位置  HIM
W51.15 BOOL  ; 到取料位置 HIM
W52.01 BOOL  ; 第#2排#13点
W52.02 BOOL  ; #2排#14点
W52.03 BOOL  ; #2排#15点
W52.04 BOOL  ; #2排#16点
W52.05 BOOL  ; #2排#17点
W52.06 BOOL  ; #2排#18点
W52.07 BOOL  ; #2排#19点
W52.08 BOOL  ; #2排#20点
W52.09 BOOL  ; #2排#21点
W52.10 BOOL  ; #2排#22点
W52.11 BOOL  ; #2排#23点
W52.12 BOOL  ; #2排#24点
W52.13 BOOL  ; 入盘（前后）Y轴#1排放料位置
W52.14 BOOL  ; #2排放料点
W53.00 BOOL  ; .入盘X轴取料位置 HIM
W53.01 BOOL  ; 入盘X轴#1机械点-HIM
W53.02 BOOL  ; 入盘X轴#2点位置 HIM
W53.03 BOOL  ; 入盘X轴#3点位置 HIM
W53.04 BOOL  ; 入盘X轴#4点位置 HIM
W53.05 BOOL  ; 入盘X轴#5点位置 HIM
W53.06 BOOL  ; 入盘X轴#6点位置 HIM
W53.07 BOOL  ; 入盘X轴#7点位置 HIM
W53.08 BOOL  ; 入盘X轴#8点位置 HIM
W53.09 BOOL  ; 入盘X轴#9点位置 HIM
W53.10 BOOL  ; 入盘X轴#10点位置 HIM
W53.11 BOOL  ; 入盘X轴#11点位置 HIM
W53.12 BOOL  ; 入盘X轴#12点位置 HIM
W53.13 BOOL  ; 入盘前后电机#1设置
W53.14 BOOL  ; 入盘前后机械手#2排位置
W53.15 BOOL  ; 入盘前后机械手取料位置
W54.01 BOOL  ; 入盘X轴#13机械点-HIM
W54.02 BOOL  ; 入盘X轴#14机械点-HIM
W54.03 BOOL  ; 入盘X轴#15点位置 HIM
W54.04 BOOL  ; 入盘X轴#16点位置 HIM
W54.05 BOOL  ; .入盘X轴#17点位置 HIM
W54.06 BOOL  ; .入盘X轴#18点位置 HIM
W54.07 BOOL  ; .入盘X轴#19点位置 HIM
W54.08 BOOL  ; .入盘X轴#20点位置 HIM
W54.09 BOOL  ; .入盘X轴#21点位置 HIM
W54.10 BOOL  ; .入盘X轴#22点位置 HIM
W54.11 BOOL  ; .入盘X轴#23点位置 HIM
W54.12 BOOL  ; .入盘X轴#24点位置 HIM
W55.00 BOOL  ; 升降轴复位
W55.03 BOOL  ; 抓料机械手手动到取料位
W55.04 BOOL  ; 龙门）抓料机械手手动回OK位
W55.05 BOOL  ; 升降回位
W55.06 BOOL  ; 抓料机械手下降到OK位置条件
W56 CHANNEL  ; 入盘机械手#1排位置
W56.01 BOOL  ; 入盘机械手在#1位置
W56.02 BOOL  ; 入盘机械手在#2位置
W56.03 BOOL  ; 入盘机械手在#3位置
W56.04 BOOL  ; 入盘机械手在#4位置
W56.05 BOOL  ; 入盘机械手在#5位置
W56.06 BOOL  ; 入盘机械手在#6位置
W56.07 BOOL  ; 入盘机械手在#7位置
W56.08 BOOL  ; 入盘机械手在#8位置
W56.09 BOOL  ; 入盘机械手在#9位置
W56.10 BOOL  ; 入盘机械手在#10位置
W56.11 BOOL  ; 入盘机械手在#11位置
W56.12 BOOL  ; 入盘机械手在#12位置
W57 CHANNEL  ; 入盘机械手#2排位置
W57.01 BOOL  ; 入盘机械手在#13位置
W57.02 BOOL  ; 入盘机械手在#14位置
W57.03 BOOL  ; 入盘机械手在#15位置
W57.04 BOOL  ; 入盘机械手在#16位置
W57.05 BOOL  ; 入盘机械手在#17位置
W57.06 BOOL  ; 入盘机械手在#18位置
W57.07 BOOL  ; 入盘机械手在#19位置
W57.08 BOOL  ; 入盘机械手在#20位置
W57.09 BOOL  ; 入盘机械手在#21位置
W57.10 BOOL  ; 入盘机械手在#22位置
W57.11 BOOL  ; 入盘机械手在#23位置
W57.12 BOOL  ; 入盘机械手在#24位置
W58.01 BOOL  ; #1位有电池
W58.02 BOOL  ; #2位有电池
W58.03 BOOL  ; #3位有电池
W58.04 BOOL  ; #4位有电池
W58.05 BOOL  ; #5位有电池
W58.06 BOOL  ; #6位有电池
W58.07 BOOL  ; #7位有电池
W58.08 BOOL  ; #8位有电池
W58.09 BOOL  ; #9位有电池
W58.10 BOOL  ; #10位有电池
W58.11 BOOL  ; #11位有电池
W58.12 BOOL  ; #12位有电池
W59.00 BOOL  ; 入盘机有报警输出
W59.01 BOOL  ; #13位有电池
W59.02 BOOL  ; #14位有电池
W59.03 BOOL  ; #15位有电池
W59.04 BOOL  ; #16位有电池
W59.05 BOOL  ; #17位有电池
W59.06 BOOL  ; #18位有电池
W59.07 BOOL  ; #19位有电池
W59.08 BOOL  ; #20位有电池
W59.09 BOOL  ; #21位有电池
W59.10 BOOL  ; #22位有电池
W59.11 BOOL  ; #23位有电池
W59.12 BOOL  ; #24位有电池
W5.00 BOOL  ; 真空泵-HMI
W5.13 BOOL  ; 蜂鸣器屏蔽可用
W5.14 BOOL  ; 蜂鸣器开
W60.00 BOOL  ; (龙门）升降轴归零
W60.01 BOOL  ; 入盘（升降）Z轴手动下降
W60.02 BOOL  ; 入盘（升降）Z轴手动上升
W60.03 BOOL  ; （龙门）抓料机械手手动取料位置
W60.04 BOOL  ; 入盘（升降）Z轴手动回下料位置
W60.05 BOOL  ; 升降回位
W60.10 BOOL  ; 入盘Z轴取料位-HMI
W60.11 BOOL  ; 入盘Z轴放料位置-HMI
W61.00 BOOL  ; 入盘升降气缸
W61.01 BOOL  ; 入盘夹爪气缸张开位
W62.00 BOOL  ; 入盘伺服升降条件
W62.01 BOOL  ; 入盘伺服升降下降条件
W62.02 BOOL  ; 入盘Y轴移动条件
W63.00 BOOL  ; 入盘机械手取料条件
W63.01 BOOL  ; 入盘机械运行条件
W63.02 BOOL  ; 入盘机械放料条件
W63.10 BOOL  ; X、Y轴在取料位
W63.11 BOOL  ; 第1排有电池
W63.12 BOOL  ; 第二排有电池
W64.15 BOOL  ; 到下降取料位置
W66.00 BOOL  ; 自动回取料位
W66.01 BOOL  ; 下取料
W66.02 BOOL  ; 气缸下降取料
W66.03 BOOL  ; 入盘夹爪夹料
W66.04 BOOL  ; 入机械手取料上升
W66.05 BOOL  ; 入盘机械手去放料
W66.06 BOOL  ; 升降电缸下放料
W66.07 BOOL  ; 入夹爪松夹
W66.08 BOOL  ; 入盘电缸上升
W66.09 BOOL  ; X、Y轴回取料位
W66.10 BOOL  ; 入盘复位
W67.00 BOOL  ; 入盘升降气缸伸出
W67.06 BOOL  ; 料不可上行
W67.07 BOOL  ; 料盒不可下行
W67.08 BOOL  ; 复位超限
W68.00 BOOL  ; 入盘机械手左右伺服没归零
W68.01 BOOL  ; 入盘机械手前后伺服没归零
W68.02 BOOL  ; 入盘机械手升降伺服没归零
W68.03 BOOL  ; 入盘升降气缸只能在取料位升降
W68.04 BOOL  ; 入盘夹爪气缸张开异常
W68.05 BOOL  ; 入盘升降只能在入盘位下降
W68.06 BOOL  ; 入盘放料时夹爪气缸张开异常
W68.07 BOOL  ; 在取料位才能下降取料
W68.10 BOOL  ; 入盘机械手异常
W69.00 BOOL  ; 出料末端有料
W6.00 BOOL  ; 进料机械手左进料位-HMI
W6.01 BOOL  ; 进料机械手右进料位置-HMI
W6.02 BOOL  ; 进料机械手腔体1位置-HMI
W6.03 BOOL  ; 进料机械手腔体2位置-HMI
W6.04 BOOL  ; 进NG左位置-HMI
W6.06 BOOL  ; 出料机械手腔体1位置-HMI
W6.07 BOOL  ; 出料机械手腔体2位置-HMI
W6.08 BOOL  ; 出料左OK放料位置-HMI
W6.09 BOOL  ; 出料机械手OK放料位置-HMI
W6.10 BOOL  ; 进料机械手NG放料位-HMI
W6.11 BOOL  ; 整机复位
W70.00 BOOL  ; 料盘回原
W70.01 BOOL  ; 料盘下降
W70.02 BOOL  ; 料盘上升
W70.03 BOOL  ; 电池入盘位 HIM
W70.04 BOOL  ; 料盘机到放料位置  HIM
W70.05 BOOL  ; 托盘扫码手动
W70.06 BOOL  ; 下有料盘电机
W70.07 BOOL  ; 有料盘缓存电机
W70.10 BOOL  ; 电池入盒位置 HIM
W70.11 BOOL  ; 上空料盒位置 HIM
W71.00 BOOL  ; 左脱离气缸手动 HIM
W71.01 BOOL  ; 右脱离气缸手动 HIM
W71.03 BOOL  ; 料盘下阻挡气缸打开  HIM
W71.04 BOOL  ; #1上顶气缸手动 HIM
W71.05 BOOL  ; #2上顶气缸手动 HIM
W71.06 BOOL  ; #2下顶气缸手动 HIM
W71.07 BOOL  ; #1下顶气缸手动 HIM
W72.00 BOOL  ; 料盘伺服上升条件
W72.01 BOOL  ; 料盘伺服下降条件
W73.00 BOOL  ; 料盒上升条件
W73.01 BOOL  ; 料盒下降条件
W73.02 BOOL  ; 下顶气缸1顶升
W73.03 BOOL  ; 下顶气缸2顶(外面）
W73.04 BOOL  ; 下顶升气缸1缩回
W73.05 BOOL  ; 下顶升气缸2下降
W73.06 BOOL  ; 上空盘电机运行
W73.07 BOOL  ; 上空盘电机停止
W73.08 BOOL  ; 料盘自动下行
W73.09 BOOL  ; 料盘自动上行
W73.10 BOOL  ; 下料电机运行
W73.11 BOOL  ; 缓存电机运行
W74.01 BOOL  ; 定位气缸伸出
W74.02 BOOL  ; 脱离气缸伸出
W74.03 BOOL  ; 脱离气缩回
W74.04 BOOL  ; 上顶升缸2上升
W74.05 BOOL  ; 上顶升缸1上升
W74.06 BOOL  ; 上阻挡气缸
W75.00 BOOL  ; 入盘扫码信号
W75.01 BOOL  ; 入盘扫码完成
W75.02 BOOL  ; 托盘扫码OK
W75.03 BOOL  ; 托盘扫码失败
W75.04 BOOL  ; 托盘注册OK
W75.05 BOOL  ; 托盘码注册NG
W75.06 BOOL  ; 托盘更换
W75.07 BOOL  ; 有料盘缓存电机
W76.03 BOOL  ; 料盘下阻挡气缸打开
W76.12 BOOL  ; 下有料盘电机
W76.13 BOOL  ; 上空料盘电机
W77.00 BOOL  ; 左脱离气缸手动
W77.01 BOOL  ; 右脱离气缸手动
W77.02 BOOL  ; 料盘定位气缸打开
W77.03 BOOL  ; 料盘上阻挡气缸打开
W77.04 BOOL  ; #1上顶气缸手动
W77.05 BOOL  ; #2上顶气缸手动
W77.06 BOOL  ; #2下顶气缸手动
W77.07 BOOL  ; #1下顶气缸手动
W78.00 BOOL  ; 料盒升降伺服没归零
W78.01 BOOL  ; 有料盒脱离气缸没伸出不能上升
W78.02 BOOL  ; 有料盒定位气缸没缩回不能上升
W78.03 BOOL  ; 下面有料盒感应异常不下行
W78.04 BOOL  ; 有料盒时定位气缸没缩回不能下降
W78.10 BOOL  ; 有异常料盒伺服不能操作
W7.01 BOOL  ; 上料机械手复位
W7.02 BOOL  ; 模组气缸状态条件
W7.03 BOOL  ; 下料机械手复位
W7.04 BOOL  ; 入盘机械手复位
W7.05 BOOL  ; 入盘物流原侠
W7.11 BOOL  ; 上料夹1有料
W7.12 BOOL  ; 上料夹2有料
W80.00 BOOL  ; 上料横移气缸复位
W80.01 BOOL  ; 上料移载气缸复位
W80.02 BOOL  ; 下料横移气缸复位
W80.03 BOOL  ; 下料移载气缸复位
W8.04 BOOL  ; 清尾料
W8.05 BOOL  ; 手动转自动提示
W8.13 BOOL  ; 上料旋转在进料反角度
W8.14 BOOL  ; 下料机械手到#1腔体安全条件
W8.15 BOOL  ; 下料机械手到#2腔体安全条件
W90 CHANNEL  ; 异常报警状态1
W91 CHANNEL  ; 异常报警状态2
W92 CHANNEL  ; 异常报警状态3
W93 CHANNEL  ; 异常报警状态4
W94 CHANNEL  ; 异常报警状态5
W94.07 BOOL  ; 进料机械手Sev_On信号异常
W94.09 BOOL  ; 出料机械手Sev_On信号异常
W94.10 BOOL  ; 急停报警
W95 CHANNEL  ; 暂停状态
W95.00 BOOL  ; 前门已打开
W95.01 BOOL  ; 后门已打开
W95.03 BOOL  ; 左侧门已打开
W95.04 BOOL  ; 右侧门已打开
W96.00 BOOL  ; 前门已打开
W96.01 BOOL  ; 后门已打开
W96.02 BOOL  ; 左侧门已打开
W96.03 BOOL  ; 右侧门已打开
W96.04 BOOL  ; 气压不足
W96.05 BOOL  ; 电脑没启动
W96.06 BOOL  ; 上料机械手没归零
W96.07 BOOL  ; 下料机械手没归零
W96.08 BOOL  ; 入盘机械手没归零
W96.09 BOOL  ; 料盘伺服没归零
W96.10 BOOL  ; 氦检仪没启动
W96.11 BOOL  ; 氦检仪通信异常
W96.12 BOOL  ; #1真空计断线
W96.13 BOOL  ; #2真空计断线
W96.14 BOOL  ; 氦检仪没稳定
W97.00 BOOL  ; 进料夹爪1没张开
W97.01 BOOL  ; 进料夹爪2没张开
W97.02 BOOL  ; 上料夹爪1没张开
W97.03 BOOL  ; 上料夹爪2没张开
W97.04 BOOL  ; 上料夹爪3没张开
W97.05 BOOL  ; 上料夹爪4没张开
W97.06 BOOL  ; 下料夹爪1没张开
W97.07 BOOL  ; 下料夹爪2没张开
W97.08 BOOL  ; 下料夹爪3没张开
W97.09 BOOL  ; 下料夹爪4没张开
W97.10 BOOL  ; 出料夹爪1没张开
W97.11 BOOL  ; 出料夹爪2没张开
W97.12 BOOL  ; 氦检仪还没有稳定
W98.00 BOOL  ; 上料横移气缸没缩回
W98.01 BOOL  ; 上料提升气缸没缩回
W98.02 BOOL  ; 上料升降气缸没缩回
W98.03 BOOL  ; 上料移栽气缸没缩回
W98.04 BOOL  ; #1合模气缸没缩回
W98.05 BOOL  ; #2合模气缸没缩回
W98.06 BOOL  ; 出料提升气缸没缩回
W98.07 BOOL  ; 下料横移气缸没缩回
W98.08 BOOL  ; 下料提升气缸没缩回
W98.09 BOOL  ; 下料升降气缸没缩回
W98.10 BOOL  ; 下料移栽气缸没缩回
W98.11 BOOL  ; NG拨料气缸没缩回
W98.12 BOOL  ; 进料提升气缸没缩回
W98.13 BOOL  ; 扫码NG缓存气缸没伸出
W98.14 BOOL  ; 扫码气缸没缩回
W99.00 BOOL  ; 上料机械手没归零
W99.01 BOOL  ; 模组气缸状态错误
W99.02 BOOL  ; 下料机械手没归零
W99.03 BOOL  ; 入盘机械手没归零
W99.04 BOOL  ; 料盘升降没归零
W99.05 BOOL  ; 电脑系统没开启
W9.00 BOOL  ; 上料机械手在左进料位置
W9.01 BOOL  ; 上料机械手在右进料位置
W9.02 BOOL  ; 上料机械手在腔体1位置
W9.03 BOOL  ; 上料机械手在腔体2位置
W9.04 BOOL  ; 上料机械手在左NG位置
W9.05 BOOL  ; 上料机械手在右NG位置
W9.06 BOOL  ; 出料机械手在腔体1位置
W9.07 BOOL  ; 出料机械手在腔体2位置
W9.08 BOOL  ; 出料机械手在OK左位置
W9.09 BOOL  ; 出料机械手在OK右位置
W9.10 BOOL  ; 出料机械手在NG右位置
W9.11 BOOL  ; 下料旋转在待料2位置
W9.12 BOOL  ; 下料旋转在下料位置
W9.13 BOOL  ; 机械手手动停止距离

## Program 主程序 (cyclic task 0)
Local symbols
D UINT
P_01s BOOL
P_10ms BOOL
P_1S BOOL

### Section 主程序

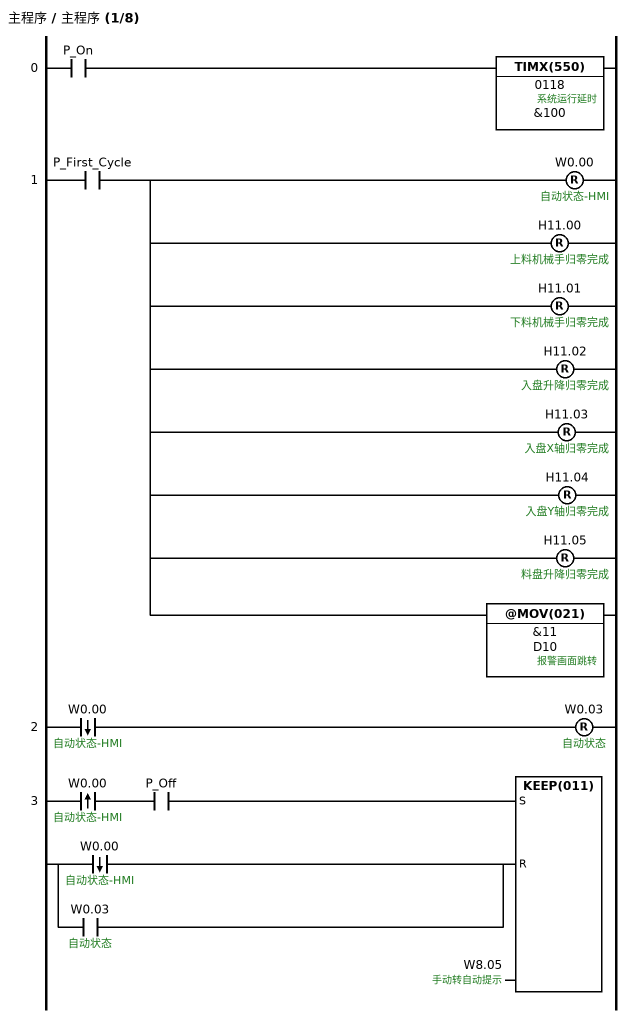
; rung 0
LD P_On
TIMX(550) 0118 &100  ; 系统运行延时
; rung 1
LD P_First_Cycle
RSET W0.00  ; 自动状态-HMI
RSET H11.00  ; 上料机械手归零完成
RSET H11.01  ; 下料机械手归零完成
RSET H11.02  ; 入盘升降归零完成
RSET H11.03  ; 入盘X轴归零完成
RSET H11.04  ; 入盘Y轴归零完成
RSET H11.05  ; 料盘升降归零完成
@MOV(021) &11 D10  ; 报警画面跳转
; rung 2
%LD W0.00  ; 自动状态-HMI
RSET W0.03  ; 自动状态
; rung 3
@LD W0.00  ; 自动状态-HMI
AND P_Off
%LD W0.00  ; 自动状态-HMI
OR W0.03  ; 自动状态
KEEP(011) W8.05  ; 手动转自动提示

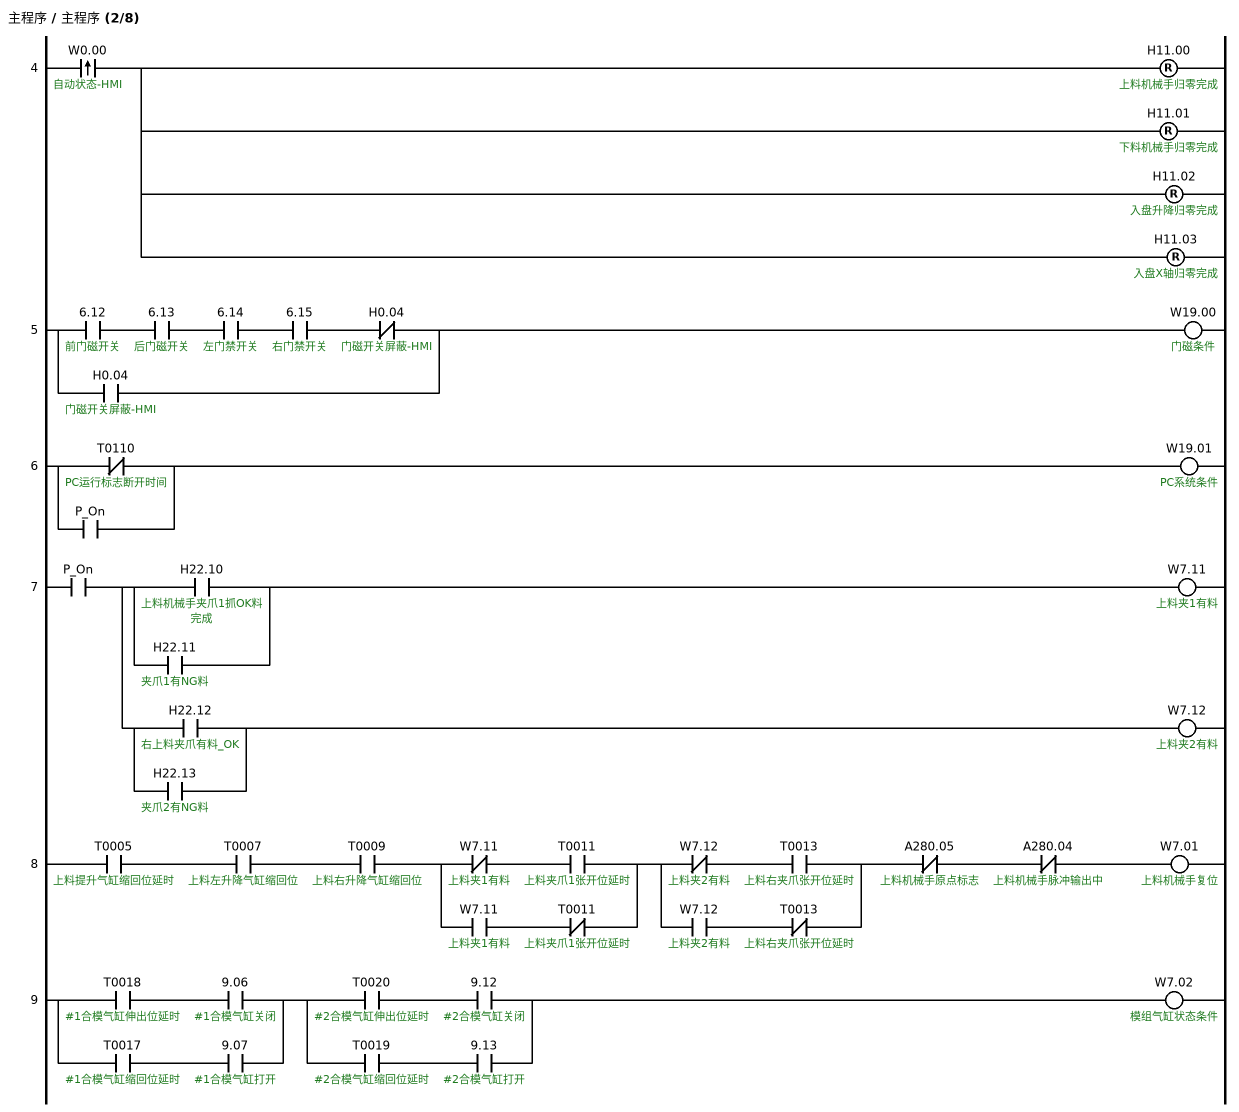
; rung 4
@LD W0.00  ; 自动状态-HMI
RSET H11.00  ; 上料机械手归零完成
RSET H11.01  ; 下料机械手归零完成
RSET H11.02  ; 入盘升降归零完成
RSET H11.03  ; 入盘X轴归零完成
; rung 5
LD 6.12  ; 前门磁开关
AND 6.13  ; 后门磁开关
AND 6.14  ; 左门禁开关
AND 6.15  ; 右门禁开关
ANDNOT H0.04  ; 门磁开关屏蔽-HMI
OR H0.04  ; 门磁开关屏蔽-HMI
OUT W19.00  ; 门磁条件
; rung 6
LDNOT T0110  ; PC运行标志断开时间
OR P_On
OUT W19.01  ; PC系统条件
; rung 7
LD P_On
OUT TR0
LD H22.10  ; 上料机械手夹爪1抓OK料完成
OR H22.11  ; 夹爪1有NG料
ANDLD
OUT W7.11  ; 上料夹1有料
LD TR0
LD H22.12  ; 右上料夹爪有料_OK
OR H22.13  ; 夹爪2有NG料
ANDLD
OUT W7.12  ; 上料夹2有料
; rung 8
LD T0005  ; 上料提升气缸缩回位延时
AND T0007  ; 上料左升降气缸缩回位
AND T0009  ; 上料右升降气缸缩回位
LDNOT W7.11  ; 上料夹1有料
AND T0011  ; 上料夹爪1张开位延时
LD W7.11  ; 上料夹1有料
ANDNOT T0011  ; 上料夹爪1张开位延时
ORLD
ANDLD
LDNOT W7.12  ; 上料夹2有料
AND T0013  ; 上料右夹爪张开位延时
LD W7.12  ; 上料夹2有料
ANDNOT T0013  ; 上料右夹爪张开位延时
ORLD
ANDLD
ANDNOT A280.05  ; 上料机械手原点标志
ANDNOT A280.04  ; 上料机械手脉冲输出中
OUT W7.01  ; 上料机械手复位
; rung 9
LD T0018  ; #1合模气缸伸出位延时
AND 9.06  ; #1合模气缸关闭
LD T0017  ; #1合模气缸缩回位延时
AND 9.07  ; #1合模气缸打开
ORLD
LD T0020  ; #2合模气缸伸出位延时
AND 9.12  ; #2合模气缸关闭
LD T0019  ; #2合模气缸缩回位延时
AND 9.13  ; #2合模气缸打开
ORLD
ANDLD
OUT W7.02  ; 模组气缸状态条件

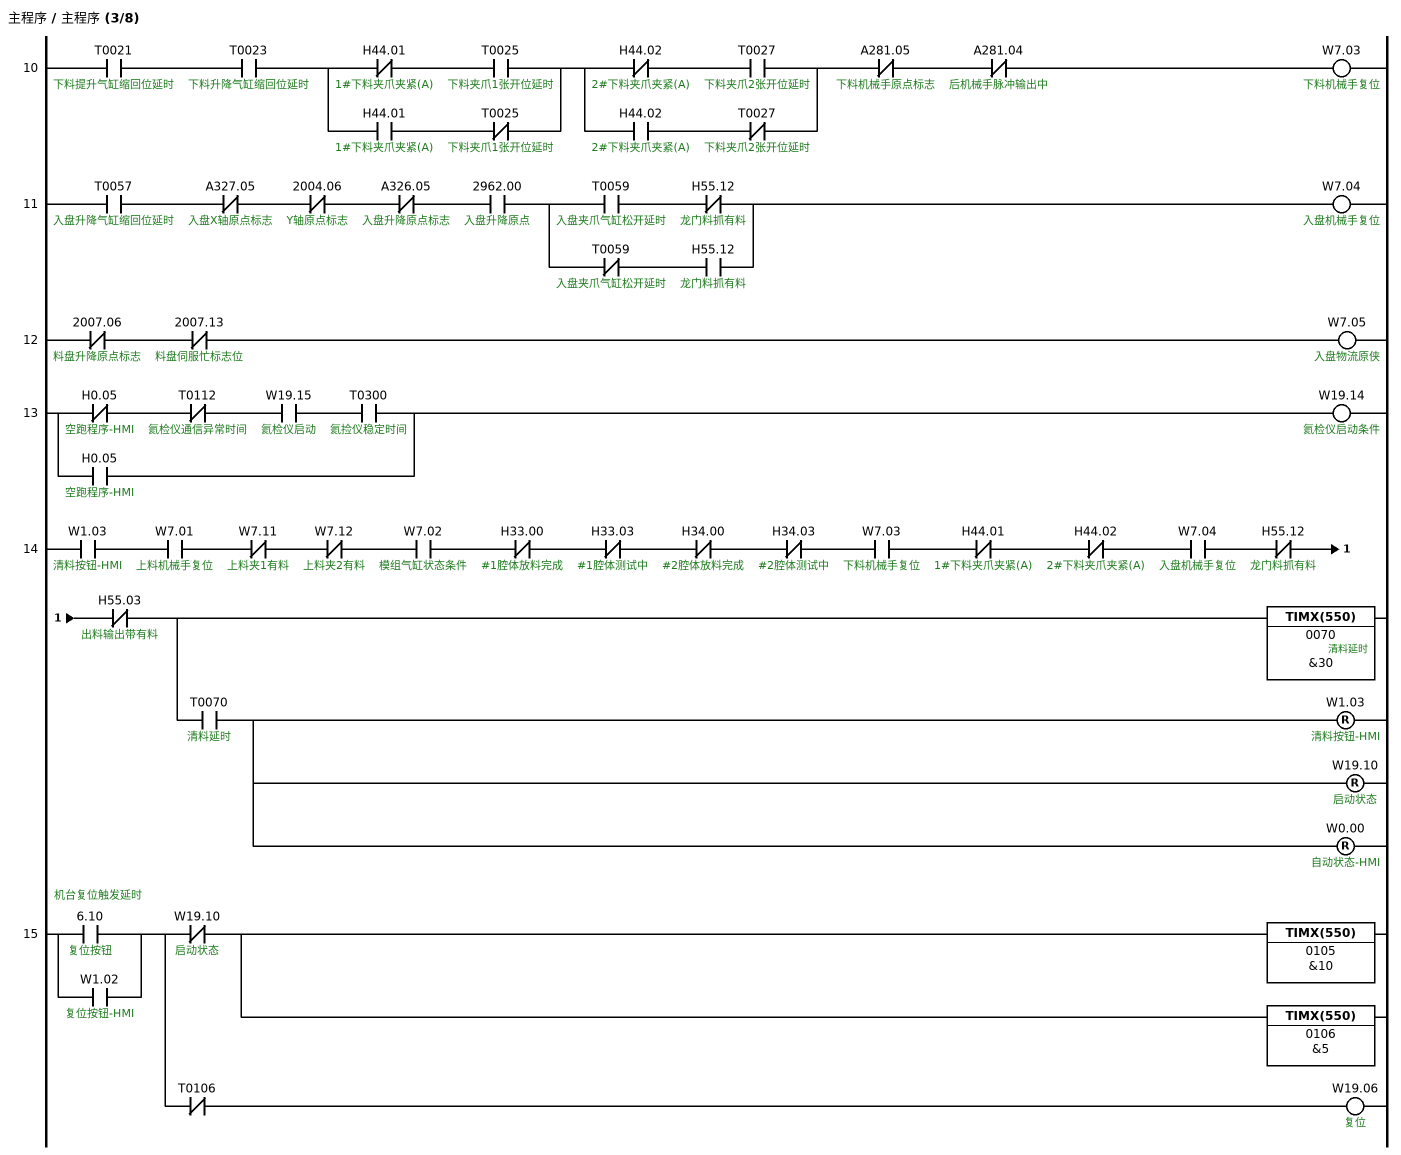
; rung 10
LD T0021  ; 下料提升气缸缩回位延时
AND T0023  ; 下料升降气缸缩回位延时
LDNOT H44.01  ; 1#下料夹爪夹紧(A)
AND T0025  ; 下料夹爪1张开位延时
LD H44.01  ; 1#下料夹爪夹紧(A)
ANDNOT T0025  ; 下料夹爪1张开位延时
ORLD
ANDLD
LDNOT H44.02  ; 2#下料夹爪夹紧(A)
AND T0027  ; 下料夹爪2张开位延时
LD H44.02  ; 2#下料夹爪夹紧(A)
ANDNOT T0027  ; 下料夹爪2张开位延时
ORLD
ANDLD
ANDNOT A281.05  ; 下料机械手原点标志
ANDNOT A281.04  ; 后机械手脉冲输出中
OUT W7.03  ; 下料机械手复位
; rung 11
LD T0057  ; 入盘升降气缸缩回位延时
ANDNOT A327.05  ; 入盘X轴原点标志
ANDNOT 2004.06  ; Y轴原点标志
ANDNOT A326.05  ; 入盘升降原点标志
AND 2962.00  ; 入盘升降原点
LD T0059  ; 入盘夹爪气缸松开延时
ANDNOT H55.12  ; 龙门料抓有料
LDNOT T0059  ; 入盘夹爪气缸松开延时
AND H55.12  ; 龙门料抓有料
ORLD
ANDLD
OUT W7.04  ; 入盘机械手复位
; rung 12
LDNOT 2007.06  ; 料盘升降原点标志
ANDNOT 2007.13  ; 料盘伺服忙标志位
OUT W7.05  ; 入盘物流原侠
; rung 13
LDNOT H0.05  ; 空跑程序-HMI
ANDNOT T0112  ; 氦检仪通信异常时间
AND W19.15  ; 氦检仪启动
AND T0300  ; 氦捡仪稳定时间
OR H0.05  ; 空跑程序-HMI
OUT W19.14  ; 氦检仪启动条件
; rung 14
LD W1.03  ; 清料按钮-HMI
AND W7.01  ; 上料机械手复位
ANDNOT W7.11  ; 上料夹1有料
ANDNOT W7.12  ; 上料夹2有料
AND W7.02  ; 模组气缸状态条件
ANDNOT H33.00  ; #1腔体放料完成
ANDNOT H33.03  ; #1腔体测试中
ANDNOT H34.00  ; #2腔体放料完成
ANDNOT H34.03  ; #2腔体测试中
AND W7.03  ; 下料机械手复位
ANDNOT H44.01  ; 1#下料夹爪夹紧(A)
ANDNOT H44.02  ; 2#下料夹爪夹紧(A)
AND W7.04  ; 入盘机械手复位
ANDNOT H55.12  ; 龙门料抓有料
ANDNOT H55.03  ; 出料输出带有料
TIMX(550) 0070 &30  ; 清料延时
AND T0070  ; 清料延时
RSET W1.03  ; 清料按钮-HMI
RSET W19.10  ; 启动状态
RSET W0.00  ; 自动状态-HMI
; rung 15: 机台复位触发延时
LD 6.10  ; 复位按钮
OR W1.02  ; 复位按钮-HMI
OUT TR0
ANDNOT W19.10  ; 启动状态
TIMX(550) 0105 &10
TIMX(550) 0106 &5
LD TR0
ANDNOT T0106
OUT W19.06  ; 复位

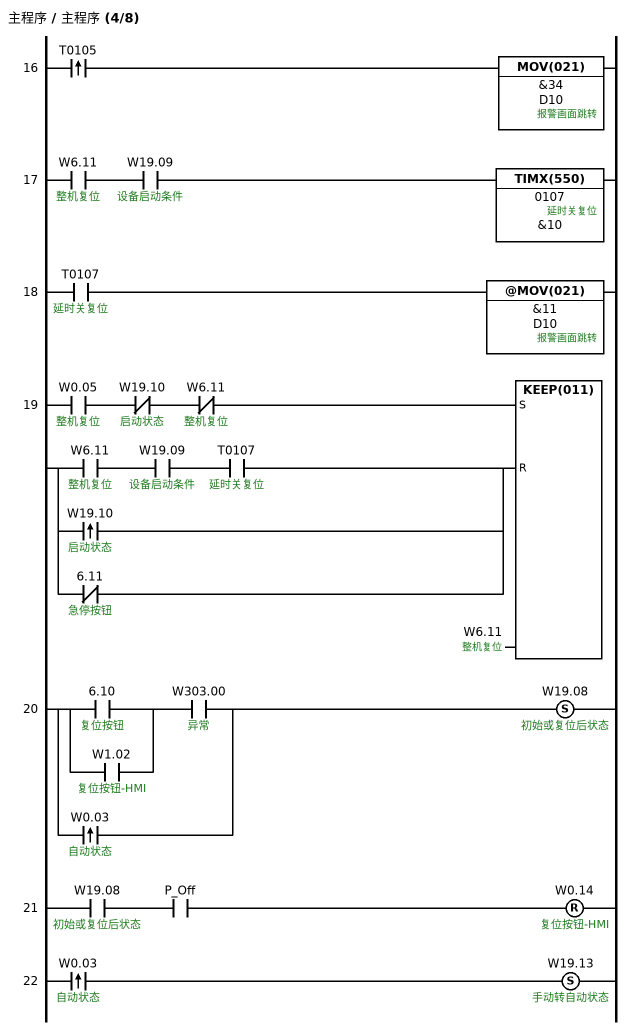
; rung 16
@LD T0105
MOV(021) &34 D10  ; 报警画面跳转
; rung 17
LD W6.11  ; 整机复位
AND W19.09  ; 设备启动条件
TIMX(550) 0107 &10  ; 延时关复位
; rung 18
LD T0107  ; 延时关复位
@MOV(021) &11 D10  ; 报警画面跳转
; rung 19
LD W0.05  ; 整机复位
ANDNOT W19.10  ; 启动状态
ANDNOT W6.11  ; 整机复位
LD W6.11  ; 整机复位
AND W19.09  ; 设备启动条件
AND T0107  ; 延时关复位
@OR W19.10  ; 启动状态
ORNOT 6.11  ; 急停按钮
KEEP(011) W6.11  ; 整机复位
; rung 20
LD 6.10  ; 复位按钮
OR W1.02  ; 复位按钮-HMI
AND W303.00  ; 异常
@OR W0.03  ; 自动状态
SET W19.08  ; 初始或复位后状态
; rung 21
LD W19.08  ; 初始或复位后状态
AND P_Off
RSET W0.14  ; 复位按钮-HMI
; rung 22
@LD W0.03  ; 自动状态
SET W19.13  ; 手动转自动状态

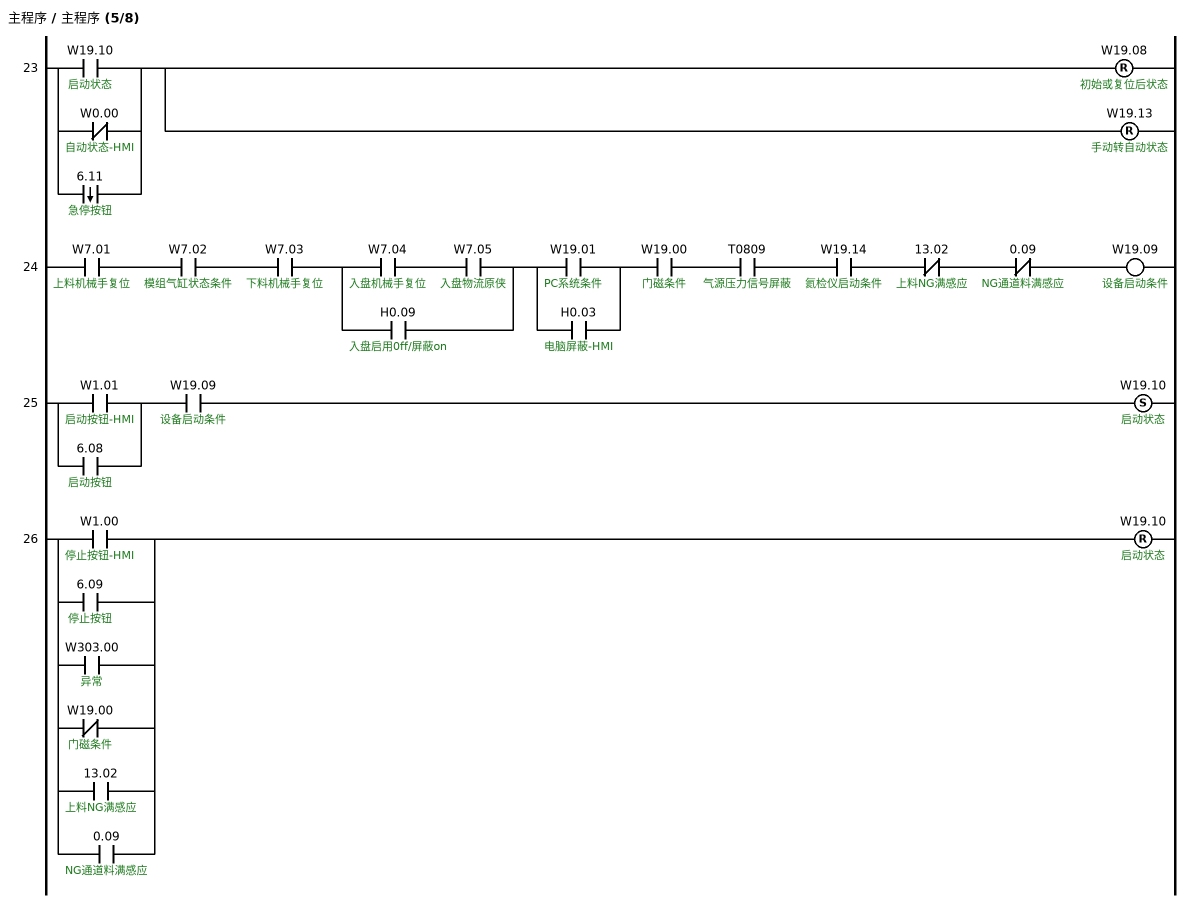
; rung 23
LD W19.10  ; 启动状态
ORNOT W0.00  ; 自动状态-HMI
%OR 6.11  ; 急停按钮
RSET W19.08  ; 初始或复位后状态
RSET W19.13  ; 手动转自动状态
; rung 24
LD W7.01  ; 上料机械手复位
AND W7.02  ; 模组气缸状态条件
AND W7.03  ; 下料机械手复位
LD W7.04  ; 入盘机械手复位
AND W7.05  ; 入盘物流原侠
OR H0.09  ; 入盘启用0ff/屏蔽on
ANDLD
LD W19.01  ; PC系统条件
OR H0.03  ; 电脑屏蔽-HMI
ANDLD
AND W19.00  ; 门磁条件
AND T0809  ; 气源压力信号屏蔽
AND W19.14  ; 氦检仪启动条件
ANDNOT 13.02  ; 上料NG满感应
ANDNOT 0.09  ; NG通道料满感应
OUT W19.09  ; 设备启动条件
; rung 25
LD W1.01  ; 启动按钮-HMI
OR 6.08  ; 启动按钮
AND W19.09  ; 设备启动条件
SET W19.10  ; 启动状态
; rung 26
LD W1.00  ; 停止按钮-HMI
OR 6.09  ; 停止按钮
OR W303.00  ; 异常
ORNOT W19.00  ; 门磁条件
OR 13.02  ; 上料NG满感应
OR 0.09  ; NG通道料满感应
RSET W19.10  ; 启动状态

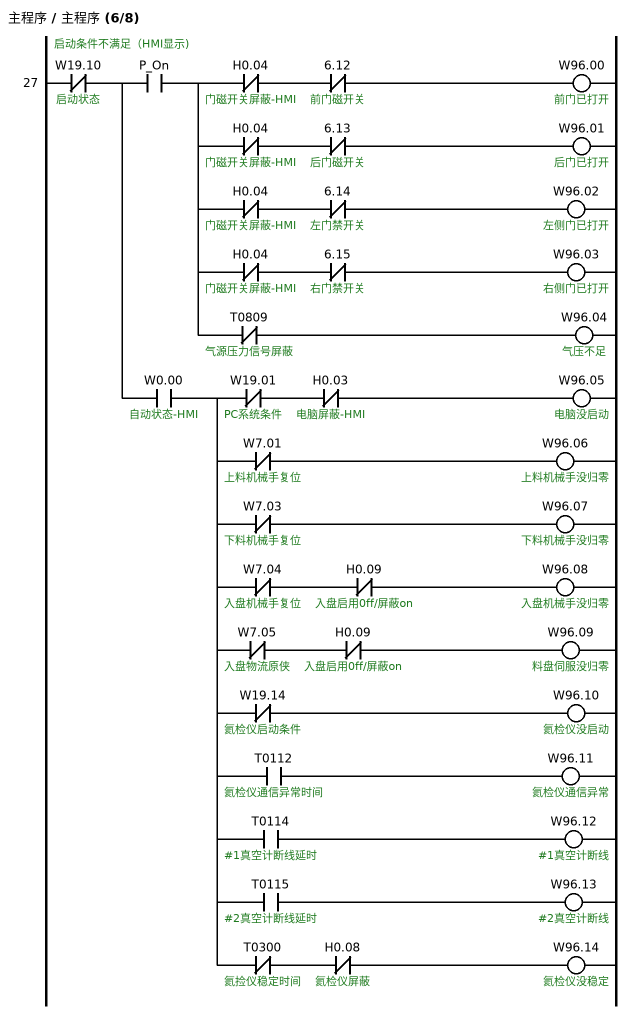
; rung 27: 启动条件不满足（HMI显示)
LDNOT W19.10  ; 启动状态
OUT TR0
AND P_On
OUT TR1
ANDNOT H0.04  ; 门磁开关屏蔽-HMI
ANDNOT 6.12  ; 前门磁开关
OUT W96.00  ; 前门已打开
LD TR1
ANDNOT H0.04  ; 门磁开关屏蔽-HMI
ANDNOT 6.13  ; 后门磁开关
OUT W96.01  ; 后门已打开
LD TR1
ANDNOT H0.04  ; 门磁开关屏蔽-HMI
ANDNOT 6.14  ; 左门禁开关
OUT W96.02  ; 左侧门已打开
LD TR1
ANDNOT H0.04  ; 门磁开关屏蔽-HMI
ANDNOT 6.15  ; 右门禁开关
OUT W96.03  ; 右侧门已打开
LD TR1
ANDNOT T0809  ; 气源压力信号屏蔽
OUT W96.04  ; 气压不足
LD TR0
AND W0.00  ; 自动状态-HMI
OUT TR0
ANDNOT W19.01  ; PC系统条件
ANDNOT H0.03  ; 电脑屏蔽-HMI
OUT W96.05  ; 电脑没启动
LD TR0
ANDNOT W7.01  ; 上料机械手复位
OUT W96.06  ; 上料机械手没归零
LD TR0
ANDNOT W7.03  ; 下料机械手复位
OUT W96.07  ; 下料机械手没归零
LD TR0
ANDNOT W7.04  ; 入盘机械手复位
ANDNOT H0.09  ; 入盘启用0ff/屏蔽on
OUT W96.08  ; 入盘机械手没归零
LD TR0
ANDNOT W7.05  ; 入盘物流原侠
ANDNOT H0.09  ; 入盘启用0ff/屏蔽on
OUT W96.09  ; 料盘伺服没归零
LD TR0
ANDNOT W19.14  ; 氦检仪启动条件
OUT W96.10  ; 氦检仪没启动
LD TR0
AND T0112  ; 氦检仪通信异常时间
OUT W96.11  ; 氦检仪通信异常
LD TR0
AND T0114  ; #1真空计断线延时
OUT W96.12  ; #1真空计断线
LD TR0
AND T0115  ; #2真空计断线延时
OUT W96.13  ; #2真空计断线
LD TR0
ANDNOT T0300  ; 氦捡仪稳定时间
ANDNOT H0.08  ; 氦检仪屏蔽
OUT W96.14  ; 氦检仪没稳定

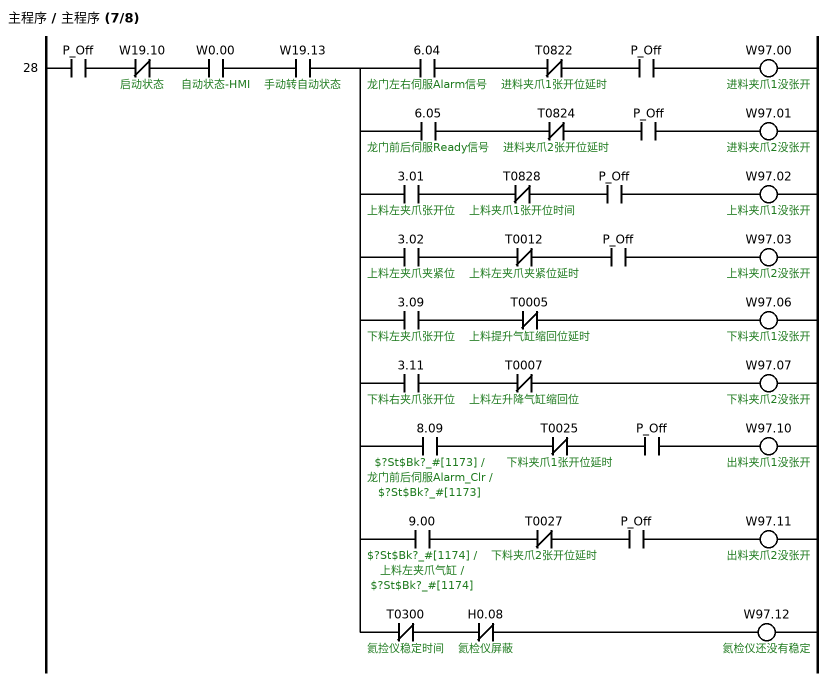
; rung 28
LD P_Off
ANDNOT W19.10  ; 启动状态
AND W0.00  ; 自动状态-HMI
AND W19.13  ; 手动转自动状态
OUT TR0
AND 6.04  ; 龙门左右伺服Alarm信号
ANDNOT T0822  ; 进料夹爪1张开位延时
AND P_Off
OUT W97.00  ; 进料夹爪1没张开
LD TR0
AND 6.05  ; 龙门前后伺服Ready信号
ANDNOT T0824  ; 进料夹爪2张开位延时
AND P_Off
OUT W97.01  ; 进料夹爪2没张开
LD TR0
AND 3.01  ; 上料左夹爪张开位
ANDNOT T0828  ; 上料夹爪1张开位时间
AND P_Off
OUT W97.02  ; 上料夹爪1没张开
LD TR0
AND 3.02  ; 上料左夹爪夹紧位
ANDNOT T0012  ; 上料左夹爪夹紧位延时
AND P_Off
OUT W97.03  ; 上料夹爪2没张开
LD TR0
AND 3.09  ; 下料左夹爪张开位
ANDNOT T0005  ; 上料提升气缸缩回位延时
OUT W97.06  ; 下料夹爪1没张开
LD TR0
AND 3.11  ; 下料右夹爪张开位
ANDNOT T0007  ; 上料左升降气缸缩回位
OUT W97.07  ; 下料夹爪2没张开
LD TR0
AND 8.09  ; $?St$Bk?_#[1173] / 龙门前后伺服Alarm_Clr / $?St$Bk?_#[1173]
ANDNOT T0025  ; 下料夹爪1张开位延时
AND P_Off
OUT W97.10  ; 出料夹爪1没张开
LD TR0
AND 9.00  ; $?St$Bk?_#[1174] / 上料左夹爪气缸 / $?St$Bk?_#[1174]
ANDNOT T0027  ; 下料夹爪2张开位延时
AND P_Off
OUT W97.11  ; 出料夹爪2没张开
LD TR0
ANDNOT T0300  ; 氦捡仪稳定时间
ANDNOT H0.08  ; 氦检仪屏蔽
OUT W97.12  ; 氦检仪还没有稳定

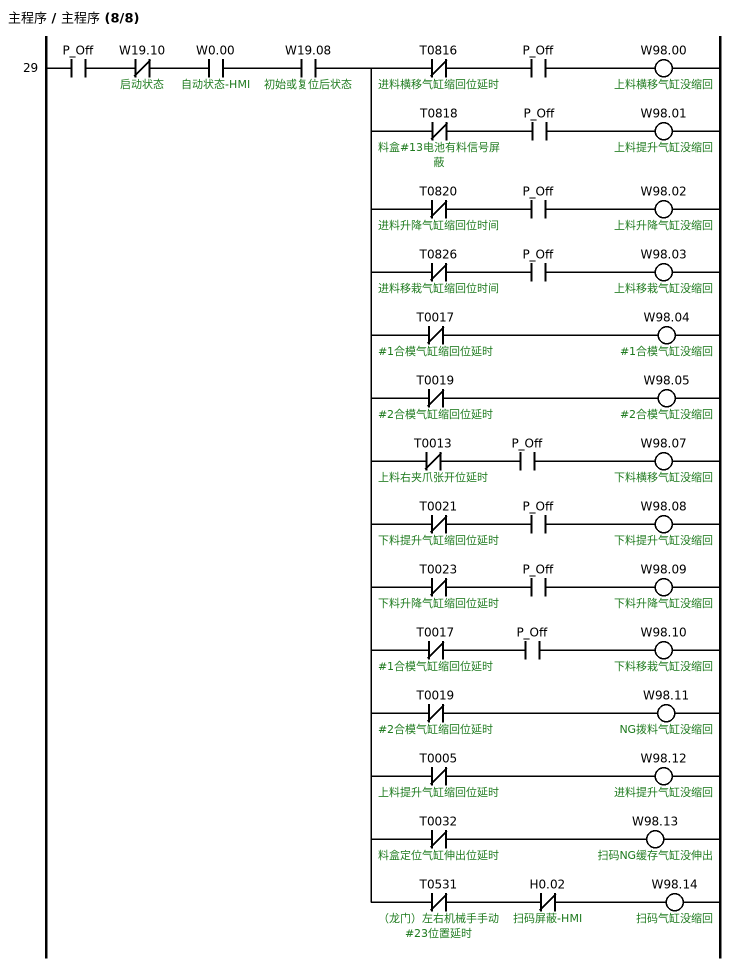
; rung 29
LD P_Off
ANDNOT W19.10  ; 启动状态
AND W0.00  ; 自动状态-HMI
AND W19.08  ; 初始或复位后状态
OUT TR0
ANDNOT T0816  ; 进料横移气缸缩回位延时
AND P_Off
OUT W98.00  ; 上料横移气缸没缩回
LD TR0
ANDNOT T0818  ; 料盒#13电池有料信号屏蔽
AND P_Off
OUT W98.01  ; 上料提升气缸没缩回
LD TR0
ANDNOT T0820  ; 进料升降气缸缩回位时间
AND P_Off
OUT W98.02  ; 上料升降气缸没缩回
LD TR0
ANDNOT T0826  ; 进料移栽气缸缩回位时间
AND P_Off
OUT W98.03  ; 上料移栽气缸没缩回
LD TR0
ANDNOT T0017  ; #1合模气缸缩回位延时
OUT W98.04  ; #1合模气缸没缩回
LD TR0
ANDNOT T0019  ; #2合模气缸缩回位延时
OUT W98.05  ; #2合模气缸没缩回
LD TR0
ANDNOT T0013  ; 上料右夹爪张开位延时
AND P_Off
OUT W98.07  ; 下料横移气缸没缩回
LD TR0
ANDNOT T0021  ; 下料提升气缸缩回位延时
AND P_Off
OUT W98.08  ; 下料提升气缸没缩回
LD TR0
ANDNOT T0023  ; 下料升降气缸缩回位延时
AND P_Off
OUT W98.09  ; 下料升降气缸没缩回
LD TR0
ANDNOT T0017  ; #1合模气缸缩回位延时
AND P_Off
OUT W98.10  ; 下料移栽气缸没缩回
LD TR0
ANDNOT T0019  ; #2合模气缸缩回位延时
OUT W98.11  ; NG拨料气缸没缩回
LD TR0
ANDNOT T0005  ; 上料提升气缸缩回位延时
OUT W98.12  ; 进料提升气缸没缩回
LD TR0
ANDNOT T0032  ; 料盒定位气缸伸出位延时
OUT W98.13  ; 扫码NG缓存气缸没伸出
LD TR0
ANDNOT T0531  ; （龙门）左右机械手手动#23位置延时
ANDNOT H0.02  ; 扫码屏蔽-HMI
OUT W98.14  ; 扫码气缸没缩回

### Section 传感器
; 气缸传感器屏蔽

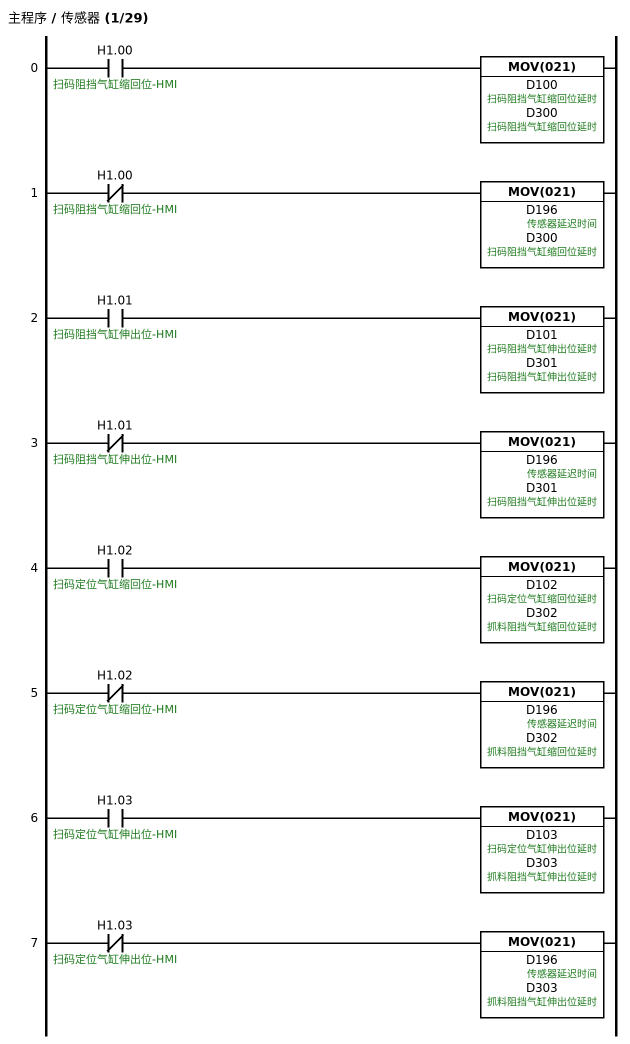
; rung 0
LD H1.00  ; 扫码阻挡气缸缩回位-HMI
MOV(021) D100 D300  ; 扫码阻挡气缸缩回位延时
; rung 1
LDNOT H1.00  ; 扫码阻挡气缸缩回位-HMI
MOV(021) D196 D300  ; 传感器延迟时间, 扫码阻挡气缸缩回位延时
; rung 2
LD H1.01  ; 扫码阻挡气缸伸出位-HMI
MOV(021) D101 D301  ; 扫码阻挡气缸伸出位延时
; rung 3
LDNOT H1.01  ; 扫码阻挡气缸伸出位-HMI
MOV(021) D196 D301  ; 传感器延迟时间, 扫码阻挡气缸伸出位延时
; rung 4
LD H1.02  ; 扫码定位气缸缩回位-HMI
MOV(021) D102 D302  ; 扫码定位气缸缩回位延时, 抓料阻挡气缸缩回位延时
; rung 5
LDNOT H1.02  ; 扫码定位气缸缩回位-HMI
MOV(021) D196 D302  ; 传感器延迟时间, 抓料阻挡气缸缩回位延时
; rung 6
LD H1.03  ; 扫码定位气缸伸出位-HMI
MOV(021) D103 D303  ; 扫码定位气缸伸出位延时, 抓料阻挡气缸伸出位延时
; rung 7
LDNOT H1.03  ; 扫码定位气缸伸出位-HMI
MOV(021) D196 D303  ; 传感器延迟时间, 抓料阻挡气缸伸出位延时

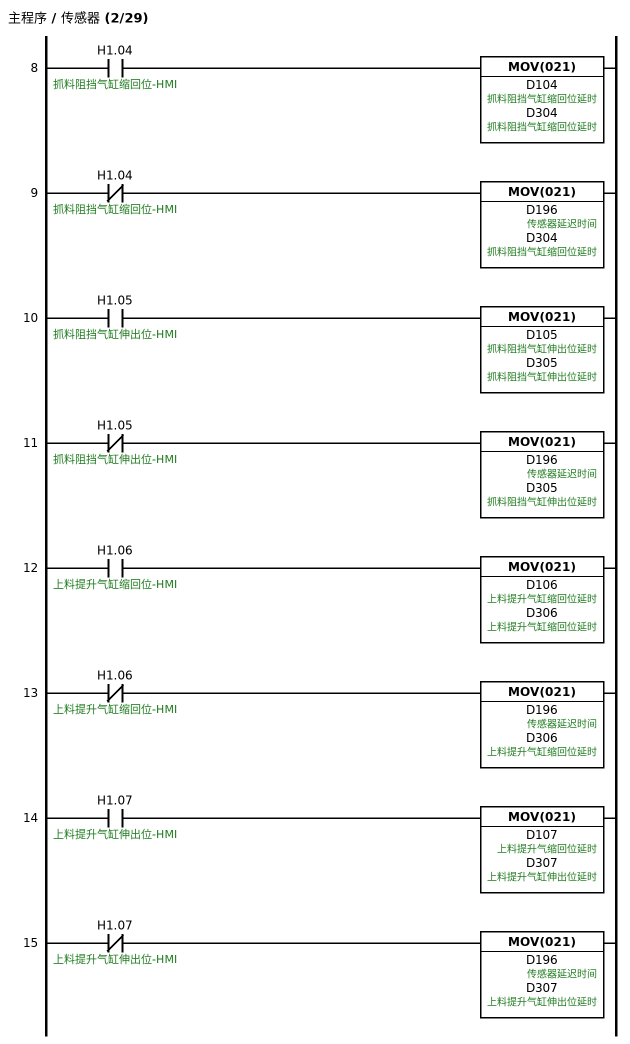
; rung 8
LD H1.04  ; 抓料阻挡气缸缩回位-HMI
MOV(021) D104 D304  ; 抓料阻挡气缸缩回位延时
; rung 9
LDNOT H1.04  ; 抓料阻挡气缸缩回位-HMI
MOV(021) D196 D304  ; 传感器延迟时间, 抓料阻挡气缸缩回位延时
; rung 10
LD H1.05  ; 抓料阻挡气缸伸出位-HMI
MOV(021) D105 D305  ; 抓料阻挡气缸伸出位延时
; rung 11
LDNOT H1.05  ; 抓料阻挡气缸伸出位-HMI
MOV(021) D196 D305  ; 传感器延迟时间, 抓料阻挡气缸伸出位延时
; rung 12
LD H1.06  ; 上料提升气缸缩回位-HMI
MOV(021) D106 D306  ; 上料提升气缸缩回位延时
; rung 13
LDNOT H1.06  ; 上料提升气缸缩回位-HMI
MOV(021) D196 D306  ; 传感器延迟时间, 上料提升气缸缩回位延时
; rung 14
LD H1.07  ; 上料提升气缸伸出位-HMI
MOV(021) D107 D307  ; 上料提升气缩回位延时, 上料提升气缸伸出位延时
; rung 15
LDNOT H1.07  ; 上料提升气缸伸出位-HMI
MOV(021) D196 D307  ; 传感器延迟时间, 上料提升气缸伸出位延时

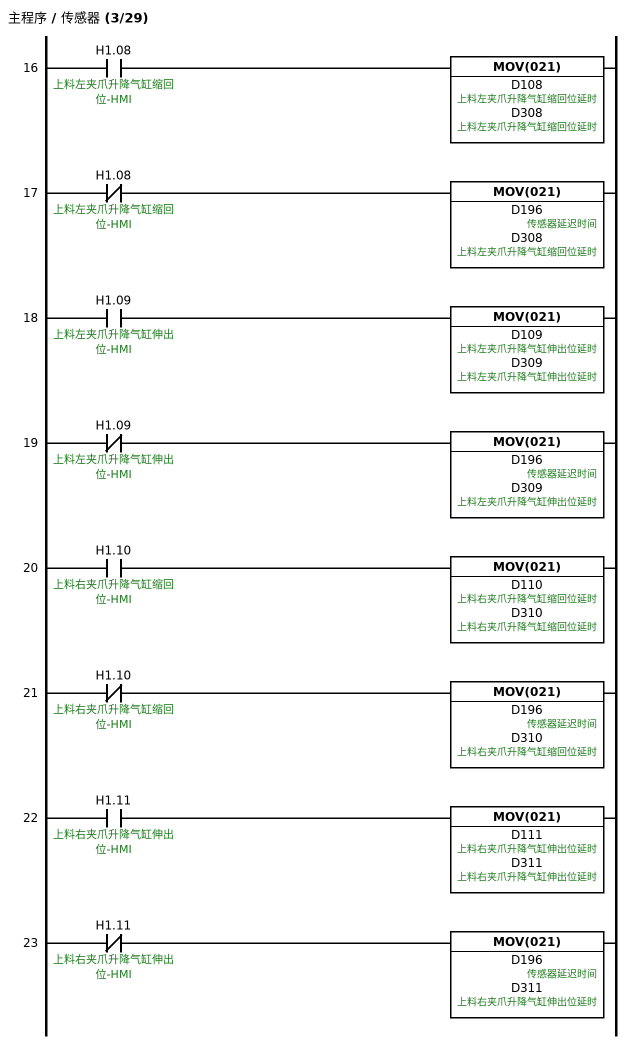
; rung 16
LD H1.08  ; 上料左夹爪升降气缸缩回位-HMI
MOV(021) D108 D308  ; 上料左夹爪升降气缸缩回位延时
; rung 17
LDNOT H1.08  ; 上料左夹爪升降气缸缩回位-HMI
MOV(021) D196 D308  ; 传感器延迟时间, 上料左夹爪升降气缸缩回位延时
; rung 18
LD H1.09  ; 上料左夹爪升降气缸伸出位-HMI
MOV(021) D109 D309  ; 上料左夹爪升降气缸伸出位延时
; rung 19
LDNOT H1.09  ; 上料左夹爪升降气缸伸出位-HMI
MOV(021) D196 D309  ; 传感器延迟时间, 上料左夹爪升降气缸伸出位延时
; rung 20
LD H1.10  ; 上料右夹爪升降气缸缩回位-HMI
MOV(021) D110 D310  ; 上料右夹爪升降气缸缩回位延时
; rung 21
LDNOT H1.10  ; 上料右夹爪升降气缸缩回位-HMI
MOV(021) D196 D310  ; 传感器延迟时间, 上料右夹爪升降气缸缩回位延时
; rung 22
LD H1.11  ; 上料右夹爪升降气缸伸出位-HMI
MOV(021) D111 D311  ; 上料右夹爪升降气缸伸出位延时
; rung 23
LDNOT H1.11  ; 上料右夹爪升降气缸伸出位-HMI
MOV(021) D196 D311  ; 传感器延迟时间, 上料右夹爪升降气缸伸出位延时

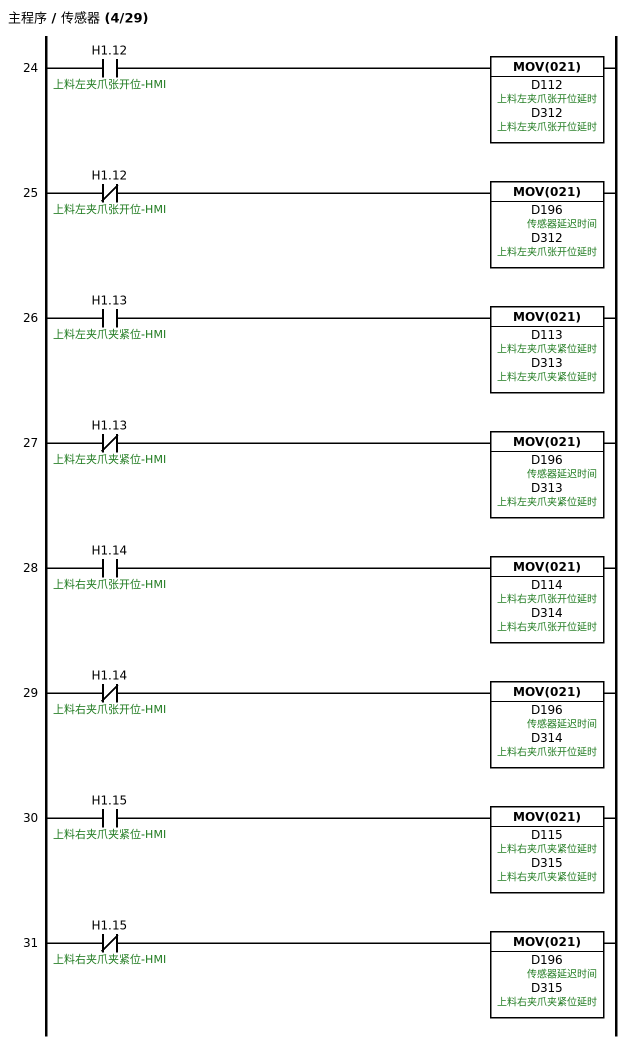
; rung 24
LD H1.12  ; 上料左夹爪张开位-HMI
MOV(021) D112 D312  ; 上料左夹爪张开位延时
; rung 25
LDNOT H1.12  ; 上料左夹爪张开位-HMI
MOV(021) D196 D312  ; 传感器延迟时间, 上料左夹爪张开位延时
; rung 26
LD H1.13  ; 上料左夹爪夹紧位-HMI
MOV(021) D113 D313  ; 上料左夹爪夹紧位延时
; rung 27
LDNOT H1.13  ; 上料左夹爪夹紧位-HMI
MOV(021) D196 D313  ; 传感器延迟时间, 上料左夹爪夹紧位延时
; rung 28
LD H1.14  ; 上料右夹爪张开位-HMI
MOV(021) D114 D314  ; 上料右夹爪张开位延时
; rung 29
LDNOT H1.14  ; 上料右夹爪张开位-HMI
MOV(021) D196 D314  ; 传感器延迟时间, 上料右夹爪张开位延时
; rung 30
LD H1.15  ; 上料右夹爪夹紧位-HMI
MOV(021) D115 D315  ; 上料右夹爪夹紧位延时
; rung 31
LDNOT H1.15  ; 上料右夹爪夹紧位-HMI
MOV(021) D196 D315  ; 传感器延迟时间, 上料右夹爪夹紧位延时

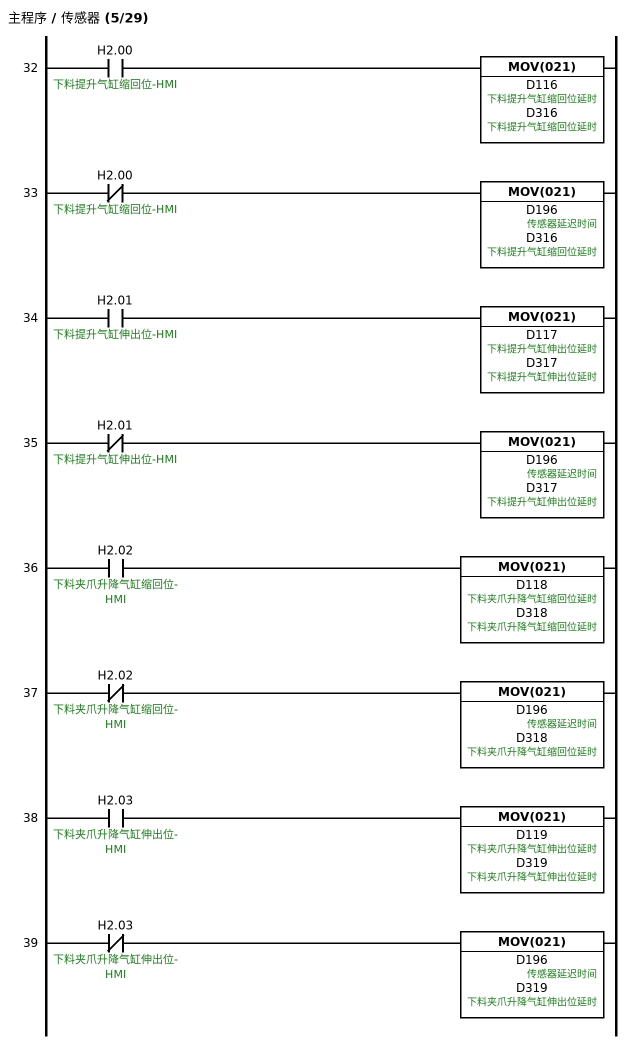
; rung 32
LD H2.00  ; 下料提升气缸缩回位-HMI
MOV(021) D116 D316  ; 下料提升气缸缩回位延时
; rung 33
LDNOT H2.00  ; 下料提升气缸缩回位-HMI
MOV(021) D196 D316  ; 传感器延迟时间, 下料提升气缸缩回位延时
; rung 34
LD H2.01  ; 下料提升气缸伸出位-HMI
MOV(021) D117 D317  ; 下料提升气缸伸出位延时
; rung 35
LDNOT H2.01  ; 下料提升气缸伸出位-HMI
MOV(021) D196 D317  ; 传感器延迟时间, 下料提升气缸伸出位延时
; rung 36
LD H2.02  ; 下料夹爪升降气缸缩回位-HMI
MOV(021) D118 D318  ; 下料夹爪升降气缸缩回位延时
; rung 37
LDNOT H2.02  ; 下料夹爪升降气缸缩回位-HMI
MOV(021) D196 D318  ; 传感器延迟时间, 下料夹爪升降气缸缩回位延时
; rung 38
LD H2.03  ; 下料夹爪升降气缸伸出位-HMI
MOV(021) D119 D319  ; 下料夹爪升降气缸伸出位延时
; rung 39
LDNOT H2.03  ; 下料夹爪升降气缸伸出位-HMI
MOV(021) D196 D319  ; 传感器延迟时间, 下料夹爪升降气缸伸出位延时

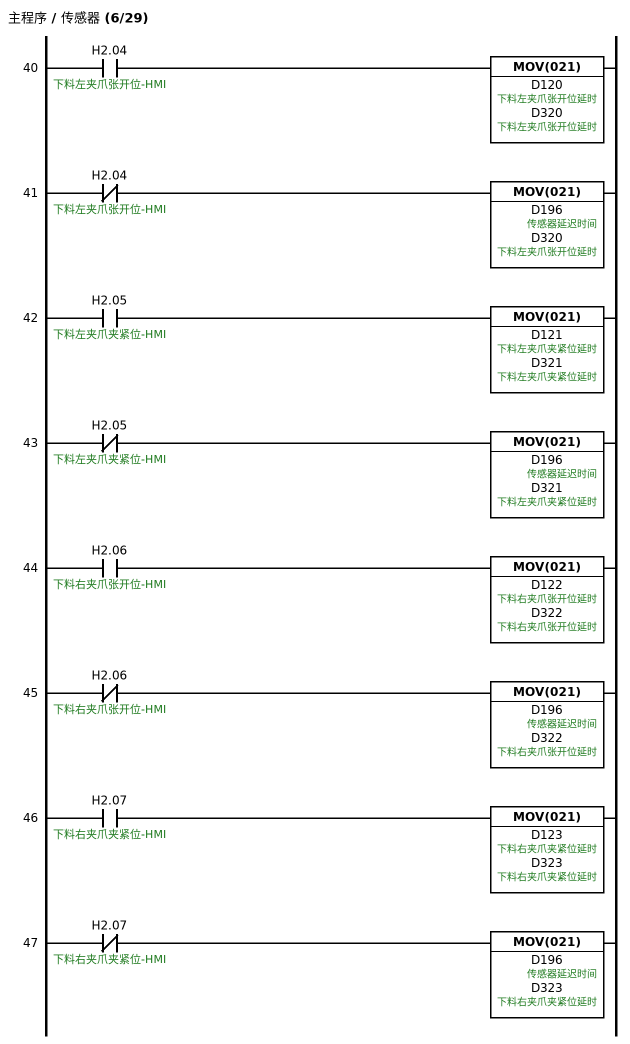
; rung 40
LD H2.04  ; 下料左夹爪张开位-HMI
MOV(021) D120 D320  ; 下料左夹爪张开位延时
; rung 41
LDNOT H2.04  ; 下料左夹爪张开位-HMI
MOV(021) D196 D320  ; 传感器延迟时间, 下料左夹爪张开位延时
; rung 42
LD H2.05  ; 下料左夹爪夹紧位-HMI
MOV(021) D121 D321  ; 下料左夹爪夹紧位延时
; rung 43
LDNOT H2.05  ; 下料左夹爪夹紧位-HMI
MOV(021) D196 D321  ; 传感器延迟时间, 下料左夹爪夹紧位延时
; rung 44
LD H2.06  ; 下料右夹爪张开位-HMI
MOV(021) D122 D322  ; 下料右夹爪张开位延时
; rung 45
LDNOT H2.06  ; 下料右夹爪张开位-HMI
MOV(021) D196 D322  ; 传感器延迟时间, 下料右夹爪张开位延时
; rung 46
LD H2.07  ; 下料右夹爪夹紧位-HMI
MOV(021) D123 D323  ; 下料右夹爪夹紧位延时
; rung 47
LDNOT H2.07  ; 下料右夹爪夹紧位-HMI
MOV(021) D196 D323  ; 传感器延迟时间, 下料右夹爪夹紧位延时

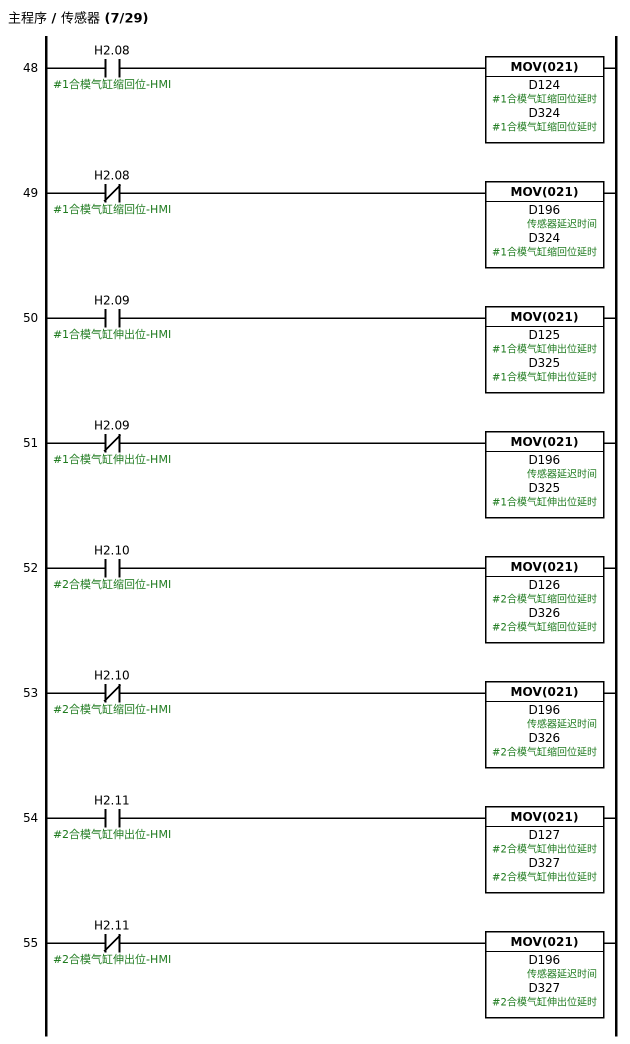
; rung 48
LD H2.08  ; #1合模气缸缩回位-HMI
MOV(021) D124 D324  ; #1合模气缸缩回位延时
; rung 49
LDNOT H2.08  ; #1合模气缸缩回位-HMI
MOV(021) D196 D324  ; 传感器延迟时间, #1合模气缸缩回位延时
; rung 50
LD H2.09  ; #1合模气缸伸出位-HMI
MOV(021) D125 D325  ; #1合模气缸伸出位延时
; rung 51
LDNOT H2.09  ; #1合模气缸伸出位-HMI
MOV(021) D196 D325  ; 传感器延迟时间, #1合模气缸伸出位延时
; rung 52
LD H2.10  ; #2合模气缸缩回位-HMI
MOV(021) D126 D326  ; #2合模气缸缩回位延时
; rung 53
LDNOT H2.10  ; #2合模气缸缩回位-HMI
MOV(021) D196 D326  ; 传感器延迟时间, #2合模气缸缩回位延时
; rung 54
LD H2.11  ; #2合模气缸伸出位-HMI
MOV(021) D127 D327  ; #2合模气缸伸出位延时
; rung 55
LDNOT H2.11  ; #2合模气缸伸出位-HMI
MOV(021) D196 D327  ; 传感器延迟时间, #2合模气缸伸出位延时

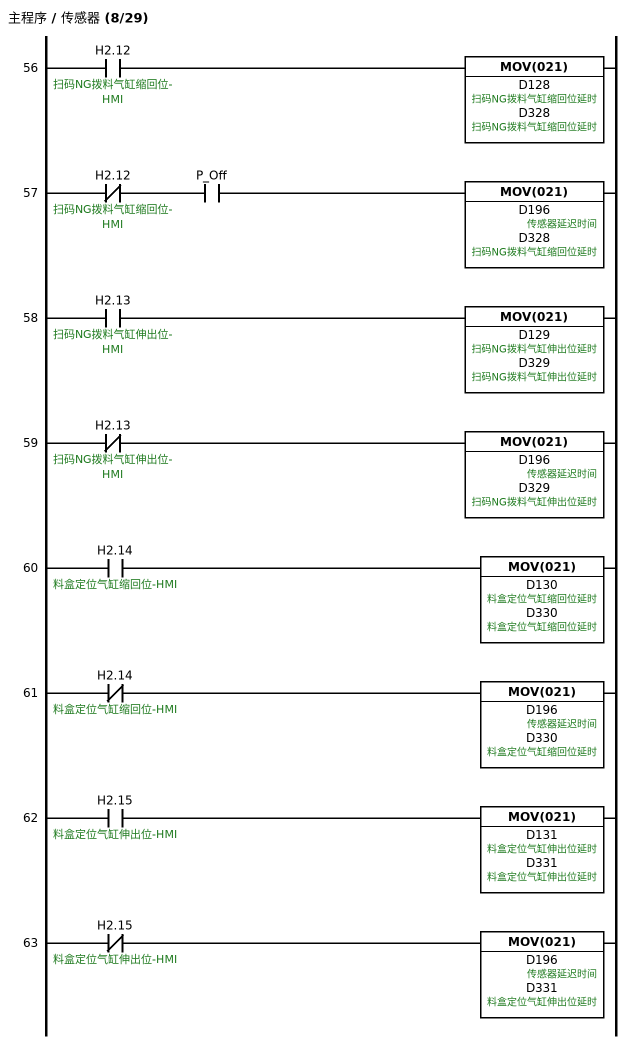
; rung 56
LD H2.12  ; 扫码NG拨料气缸缩回位-HMI
MOV(021) D128 D328  ; 扫码NG拨料气缸缩回位延时
; rung 57
LDNOT H2.12  ; 扫码NG拨料气缸缩回位-HMI
AND P_Off
MOV(021) D196 D328  ; 传感器延迟时间, 扫码NG拨料气缸缩回位延时
; rung 58
LD H2.13  ; 扫码NG拨料气缸伸出位-HMI
MOV(021) D129 D329  ; 扫码NG拨料气缸伸出位延时
; rung 59
LDNOT H2.13  ; 扫码NG拨料气缸伸出位-HMI
MOV(021) D196 D329  ; 传感器延迟时间, 扫码NG拨料气缸伸出位延时
; rung 60
LD H2.14  ; 料盒定位气缸缩回位-HMI
MOV(021) D130 D330  ; 料盒定位气缸缩回位延时
; rung 61
LDNOT H2.14  ; 料盒定位气缸缩回位-HMI
MOV(021) D196 D330  ; 传感器延迟时间, 料盒定位气缸缩回位延时
; rung 62
LD H2.15  ; 料盒定位气缸伸出位-HMI
MOV(021) D131 D331  ; 料盒定位气缸伸出位延时
; rung 63
LDNOT H2.15  ; 料盒定位气缸伸出位-HMI
MOV(021) D196 D331  ; 传感器延迟时间, 料盒定位气缸伸出位延时

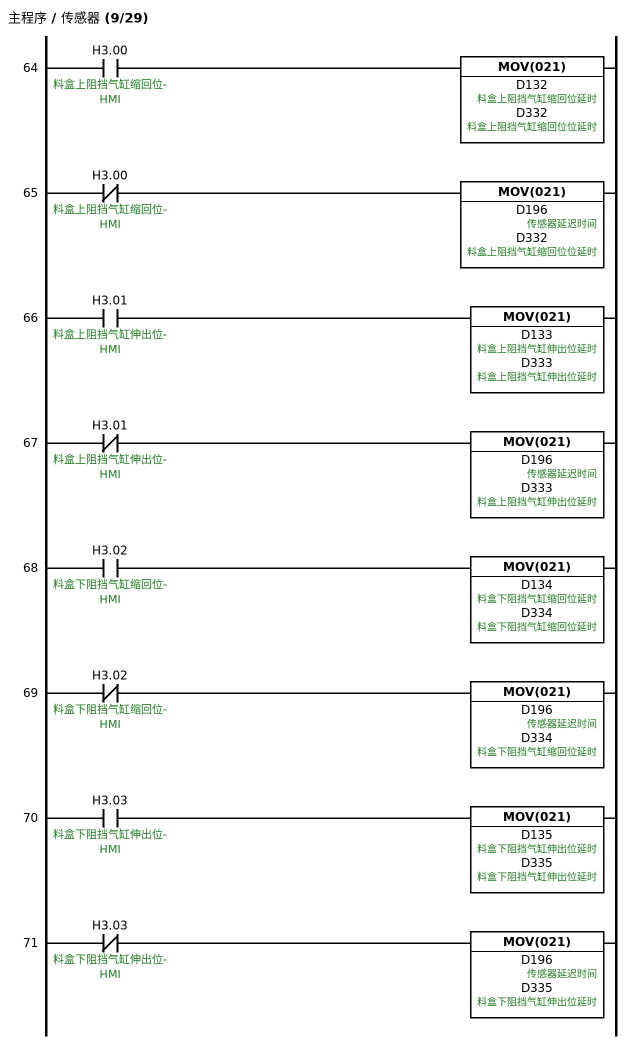
; rung 64
LD H3.00  ; 料盒上阻挡气缸缩回位-HMI
MOV(021) D132 D332  ; 料盒上阻挡气缸缩回位延时, 料盒上阻挡气缸缩回位位延时
; rung 65
LDNOT H3.00  ; 料盒上阻挡气缸缩回位-HMI
MOV(021) D196 D332  ; 传感器延迟时间, 料盒上阻挡气缸缩回位位延时
; rung 66
LD H3.01  ; 料盒上阻挡气缸伸出位-HMI
MOV(021) D133 D333  ; 料盒上阻挡气缸伸出位延时
; rung 67
LDNOT H3.01  ; 料盒上阻挡气缸伸出位-HMI
MOV(021) D196 D333  ; 传感器延迟时间, 料盒上阻挡气缸伸出位延时
; rung 68
LD H3.02  ; 料盒下阻挡气缸缩回位-HMI
MOV(021) D134 D334  ; 料盒下阻挡气缸缩回位延时
; rung 69
LDNOT H3.02  ; 料盒下阻挡气缸缩回位-HMI
MOV(021) D196 D334  ; 传感器延迟时间, 料盒下阻挡气缸缩回位延时
; rung 70
LD H3.03  ; 料盒下阻挡气缸伸出位-HMI
MOV(021) D135 D335  ; 料盒下阻挡气缸伸出位延时
; rung 71
LDNOT H3.03  ; 料盒下阻挡气缸伸出位-HMI
MOV(021) D196 D335  ; 传感器延迟时间, 料盒下阻挡气缸伸出位延时

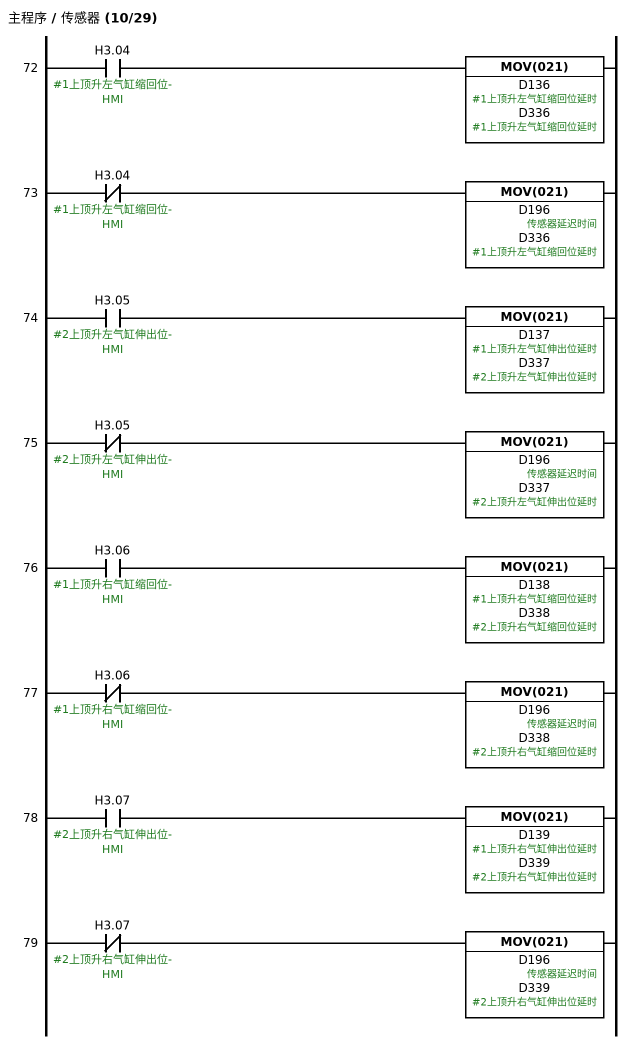
; rung 72
LD H3.04  ; #1上顶升左气缸缩回位-HMI
MOV(021) D136 D336  ; #1上顶升左气缸缩回位延时
; rung 73
LDNOT H3.04  ; #1上顶升左气缸缩回位-HMI
MOV(021) D196 D336  ; 传感器延迟时间, #1上顶升左气缸缩回位延时
; rung 74
LD H3.05  ; #2上顶升左气缸伸出位-HMI
MOV(021) D137 D337  ; #1上顶升左气缸伸出位延时, #2上顶升左气缸伸出位延时
; rung 75
LDNOT H3.05  ; #2上顶升左气缸伸出位-HMI
MOV(021) D196 D337  ; 传感器延迟时间, #2上顶升左气缸伸出位延时
; rung 76
LD H3.06  ; #1上顶升右气缸缩回位-HMI
MOV(021) D138 D338  ; #1上顶升右气缸缩回位延时, #2上顶升右气缸缩回位延时
; rung 77
LDNOT H3.06  ; #1上顶升右气缸缩回位-HMI
MOV(021) D196 D338  ; 传感器延迟时间, #2上顶升右气缸缩回位延时
; rung 78
LD H3.07  ; #2上顶升右气缸伸出位-HMI
MOV(021) D139 D339  ; #1上顶升右气缸伸出位延时, #2上顶升右气缸伸出位延时
; rung 79
LDNOT H3.07  ; #2上顶升右气缸伸出位-HMI
MOV(021) D196 D339  ; 传感器延迟时间, #2上顶升右气缸伸出位延时

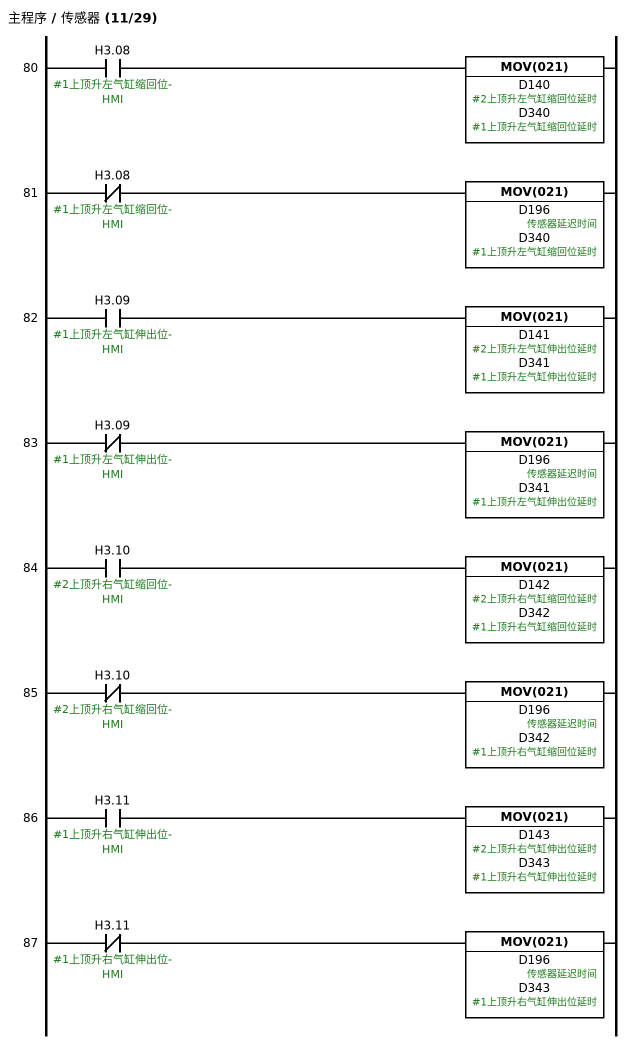
; rung 80
LD H3.08  ; #1上顶升左气缸缩回位-HMI
MOV(021) D140 D340  ; #2上顶升左气缸缩回位延时, #1上顶升左气缸缩回位延时
; rung 81
LDNOT H3.08  ; #1上顶升左气缸缩回位-HMI
MOV(021) D196 D340  ; 传感器延迟时间, #1上顶升左气缸缩回位延时
; rung 82
LD H3.09  ; #1上顶升左气缸伸出位-HMI
MOV(021) D141 D341  ; #2上顶升左气缸伸出位延时, #1上顶升左气缸伸出位延时
; rung 83
LDNOT H3.09  ; #1上顶升左气缸伸出位-HMI
MOV(021) D196 D341  ; 传感器延迟时间, #1上顶升左气缸伸出位延时
; rung 84
LD H3.10  ; #2上顶升右气缸缩回位-HMI
MOV(021) D142 D342  ; #2上顶升右气缸缩回位延时, #1上顶升右气缸缩回位延时
; rung 85
LDNOT H3.10  ; #2上顶升右气缸缩回位-HMI
MOV(021) D196 D342  ; 传感器延迟时间, #1上顶升右气缸缩回位延时
; rung 86
LD H3.11  ; #1上顶升右气缸伸出位-HMI
MOV(021) D143 D343  ; #2上顶升右气缸伸出位延时, #1上顶升右气缸伸出位延时
; rung 87
LDNOT H3.11  ; #1上顶升右气缸伸出位-HMI
MOV(021) D196 D343  ; 传感器延迟时间, #1上顶升右气缸伸出位延时

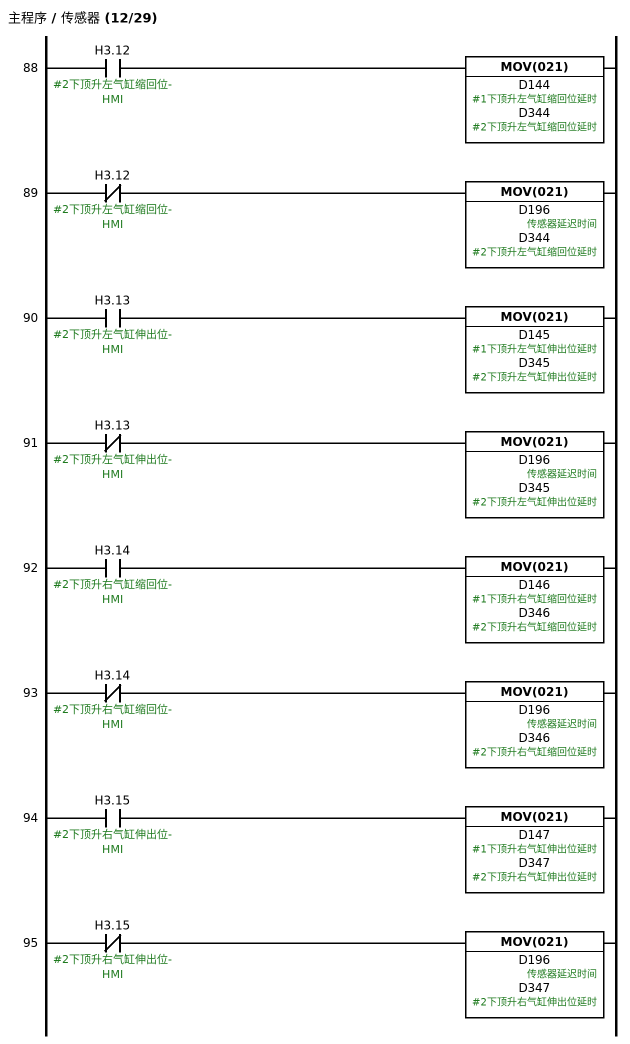
; rung 88
LD H3.12  ; #2下顶升左气缸缩回位-HMI
MOV(021) D144 D344  ; #1下顶升左气缸缩回位延时, #2下顶升左气缸缩回位延时
; rung 89
LDNOT H3.12  ; #2下顶升左气缸缩回位-HMI
MOV(021) D196 D344  ; 传感器延迟时间, #2下顶升左气缸缩回位延时
; rung 90
LD H3.13  ; #2下顶升左气缸伸出位-HMI
MOV(021) D145 D345  ; #1下顶升左气缸伸出位延时, #2下顶升左气缸伸出位延时
; rung 91
LDNOT H3.13  ; #2下顶升左气缸伸出位-HMI
MOV(021) D196 D345  ; 传感器延迟时间, #2下顶升左气缸伸出位延时
; rung 92
LD H3.14  ; #2下顶升右气缸缩回位-HMI
MOV(021) D146 D346  ; #1下顶升右气缸缩回位延时, #2下顶升右气缸缩回位延时
; rung 93
LDNOT H3.14  ; #2下顶升右气缸缩回位-HMI
MOV(021) D196 D346  ; 传感器延迟时间, #2下顶升右气缸缩回位延时
; rung 94
LD H3.15  ; #2下顶升右气缸伸出位-HMI
MOV(021) D147 D347  ; #1下顶升右气缸伸出位延时, #2下顶升右气缸伸出位延时
; rung 95
LDNOT H3.15  ; #2下顶升右气缸伸出位-HMI
MOV(021) D196 D347  ; 传感器延迟时间, #2下顶升右气缸伸出位延时

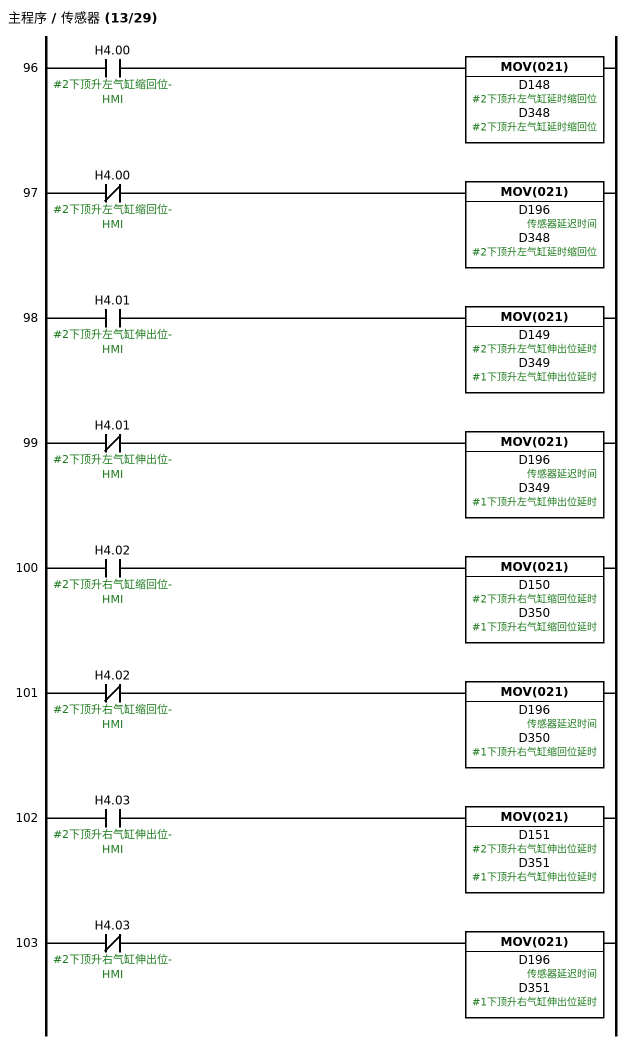
; rung 96
LD H4.00  ; #2下顶升左气缸缩回位-HMI
MOV(021) D148 D348  ; #2下顶升左气缸延时缩回位
; rung 97
LDNOT H4.00  ; #2下顶升左气缸缩回位-HMI
MOV(021) D196 D348  ; 传感器延迟时间, #2下顶升左气缸延时缩回位
; rung 98
LD H4.01  ; #2下顶升左气缸伸出位-HMI
MOV(021) D149 D349  ; #2下顶升左气缸伸出位延时, #1下顶升左气缸伸出位延时
; rung 99
LDNOT H4.01  ; #2下顶升左气缸伸出位-HMI
MOV(021) D196 D349  ; 传感器延迟时间, #1下顶升左气缸伸出位延时
; rung 100
LD H4.02  ; #2下顶升右气缸缩回位-HMI
MOV(021) D150 D350  ; #2下顶升右气缸缩回位延时, #1下顶升右气缸缩回位延时
; rung 101
LDNOT H4.02  ; #2下顶升右气缸缩回位-HMI
MOV(021) D196 D350  ; 传感器延迟时间, #1下顶升右气缸缩回位延时
; rung 102
LD H4.03  ; #2下顶升右气缸伸出位-HMI
MOV(021) D151 D351  ; #2下顶升右气缸伸出位延时, #1下顶升右气缸伸出位延时
; rung 103
LDNOT H4.03  ; #2下顶升右气缸伸出位-HMI
MOV(021) D196 D351  ; 传感器延迟时间, #1下顶升右气缸伸出位延时

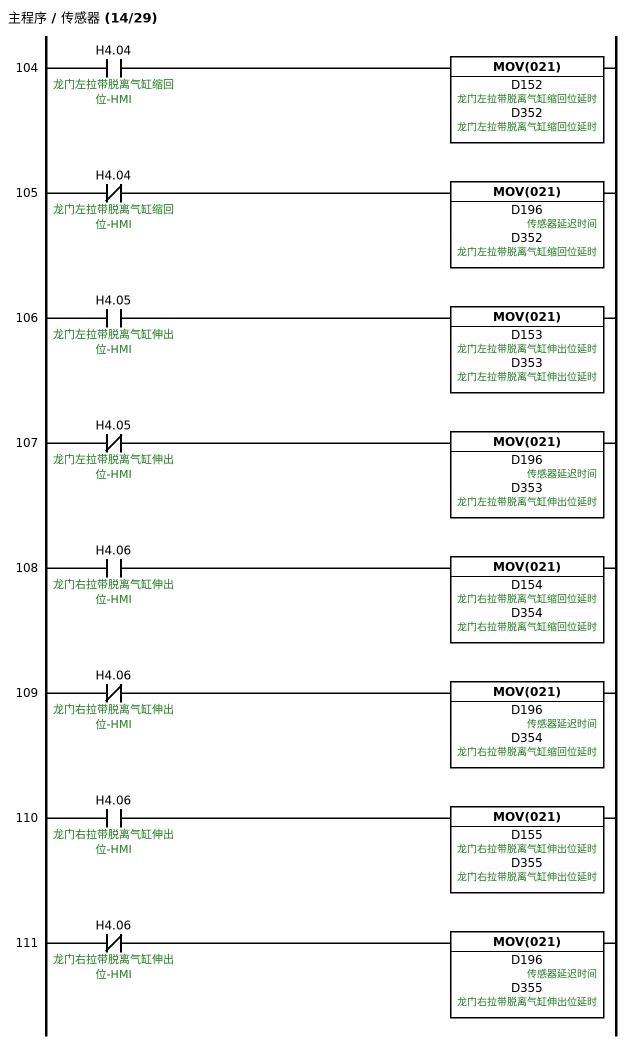
; rung 104
LD H4.04  ; 龙门左拉带脱离气缸缩回位-HMI
MOV(021) D152 D352  ; 龙门左拉带脱离气缸缩回位延时
; rung 105
LDNOT H4.04  ; 龙门左拉带脱离气缸缩回位-HMI
MOV(021) D196 D352  ; 传感器延迟时间, 龙门左拉带脱离气缸缩回位延时
; rung 106
LD H4.05  ; 龙门左拉带脱离气缸伸出位-HMI
MOV(021) D153 D353  ; 龙门左拉带脱离气缸伸出位延时
; rung 107
LDNOT H4.05  ; 龙门左拉带脱离气缸伸出位-HMI
MOV(021) D196 D353  ; 传感器延迟时间, 龙门左拉带脱离气缸伸出位延时
; rung 108
LD H4.06  ; 龙门右拉带脱离气缸伸出位-HMI
MOV(021) D154 D354  ; 龙门右拉带脱离气缸缩回位延时
; rung 109
LDNOT H4.06  ; 龙门右拉带脱离气缸伸出位-HMI
MOV(021) D196 D354  ; 传感器延迟时间, 龙门右拉带脱离气缸缩回位延时
; rung 110
LD H4.06  ; 龙门右拉带脱离气缸伸出位-HMI
MOV(021) D155 D355  ; 龙门右拉带脱离气缸伸出位延时
; rung 111
LDNOT H4.06  ; 龙门右拉带脱离气缸伸出位-HMI
MOV(021) D196 D355  ; 传感器延迟时间, 龙门右拉带脱离气缸伸出位延时

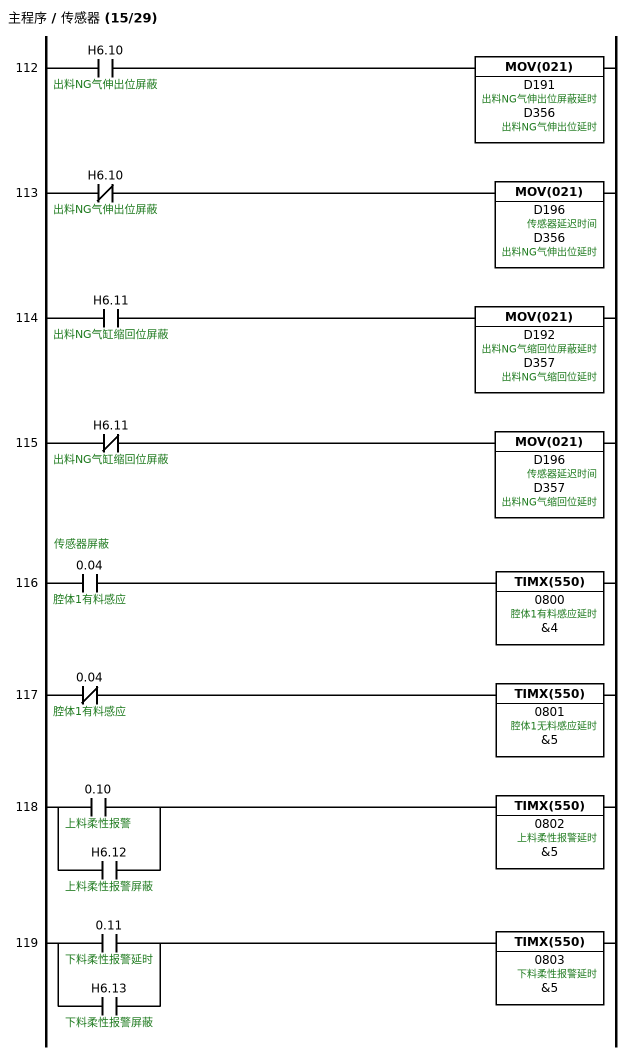
; rung 112
LD H6.10  ; 出料NG气伸出位屏蔽
MOV(021) D191 D356  ; 出料NG气伸出位屏蔽延时, 出料NG气伸出位延时
; rung 113
LDNOT H6.10  ; 出料NG气伸出位屏蔽
MOV(021) D196 D356  ; 传感器延迟时间, 出料NG气伸出位延时
; rung 114
LD H6.11  ; 出料NG气缸缩回位屏蔽
MOV(021) D192 D357  ; 出料NG气缩回位屏蔽延时, 出料NG气缩回位延时
; rung 115
LDNOT H6.11  ; 出料NG气缸缩回位屏蔽
MOV(021) D196 D357  ; 传感器延迟时间, 出料NG气缩回位延时
; rung 116: 传感器屏蔽
LD 0.04  ; 腔体1有料感应
TIMX(550) 0800 &4  ; 腔体1有料感应延时
; rung 117
LDNOT 0.04  ; 腔体1有料感应
TIMX(550) 0801 &5  ; 腔体1无料感应延时
; rung 118
LD 0.10  ; 上料柔性报警
OR H6.12  ; 上料柔性报警屏蔽
TIMX(550) 0802 &5  ; 上料柔性报警延时
; rung 119
LD 0.11  ; 下料柔性报警延时
OR H6.13  ; 下料柔性报警屏蔽
TIMX(550) 0803 &5  ; 下料柔性报警延时

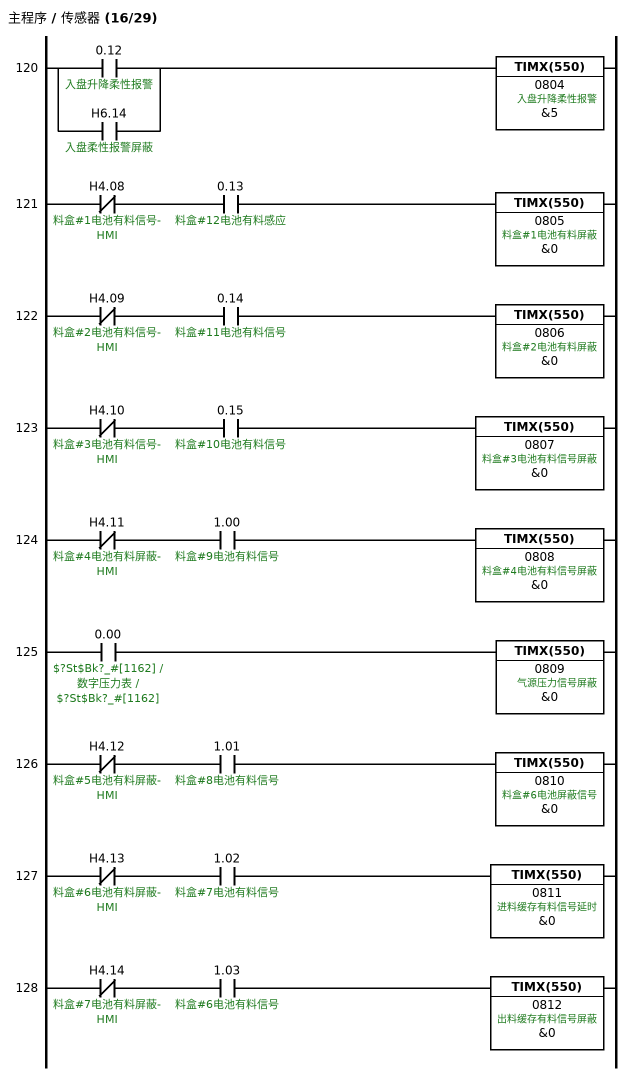
; rung 120
LD 0.12  ; 入盘升降柔性报警
OR H6.14  ; 入盘柔性报警屏蔽
TIMX(550) 0804 &5  ; 入盘升降柔性报警
; rung 121
LDNOT H4.08  ; 料盒#1电池有料信号-HMI
AND 0.13  ; 料盒#12电池有料感应
TIMX(550) 0805 &0  ; 料盒#1电池有料屏蔽
; rung 122
LDNOT H4.09  ; 料盒#2电池有料信号-HMI
AND 0.14  ; 料盒#11电池有料信号
TIMX(550) 0806 &0  ; 料盒#2电池有料屏蔽
; rung 123
LDNOT H4.10  ; 料盒#3电池有料信号-HMI
AND 0.15  ; 料盒#10电池有料信号
TIMX(550) 0807 &0  ; 料盒#3电池有料信号屏蔽
; rung 124
LDNOT H4.11  ; 料盒#4电池有料屏蔽-HMI
AND 1.00  ; 料盒#9电池有料信号
TIMX(550) 0808 &0  ; 料盒#4电池有料信号屏蔽
; rung 125
LD 0.00  ; $?St$Bk?_#[1162] / 数字压力表 / $?St$Bk?_#[1162]
TIMX(550) 0809 &0  ; 气源压力信号屏蔽
; rung 126
LDNOT H4.12  ; 料盒#5电池有料屏蔽-HMI
AND 1.01  ; 料盒#8电池有料信号
TIMX(550) 0810 &0  ; 料盒#6电池屏蔽信号
; rung 127
LDNOT H4.13  ; 料盒#6电池有料屏蔽-HMI
AND 1.02  ; 料盒#7电池有料信号
TIMX(550) 0811 &0  ; 进料缓存有料信号延时
; rung 128
LDNOT H4.14  ; 料盒#7电池有料屏蔽-HMI
AND 1.03  ; 料盒#6电池有料信号
TIMX(550) 0812 &0  ; 出料缓存有料信号屏蔽

